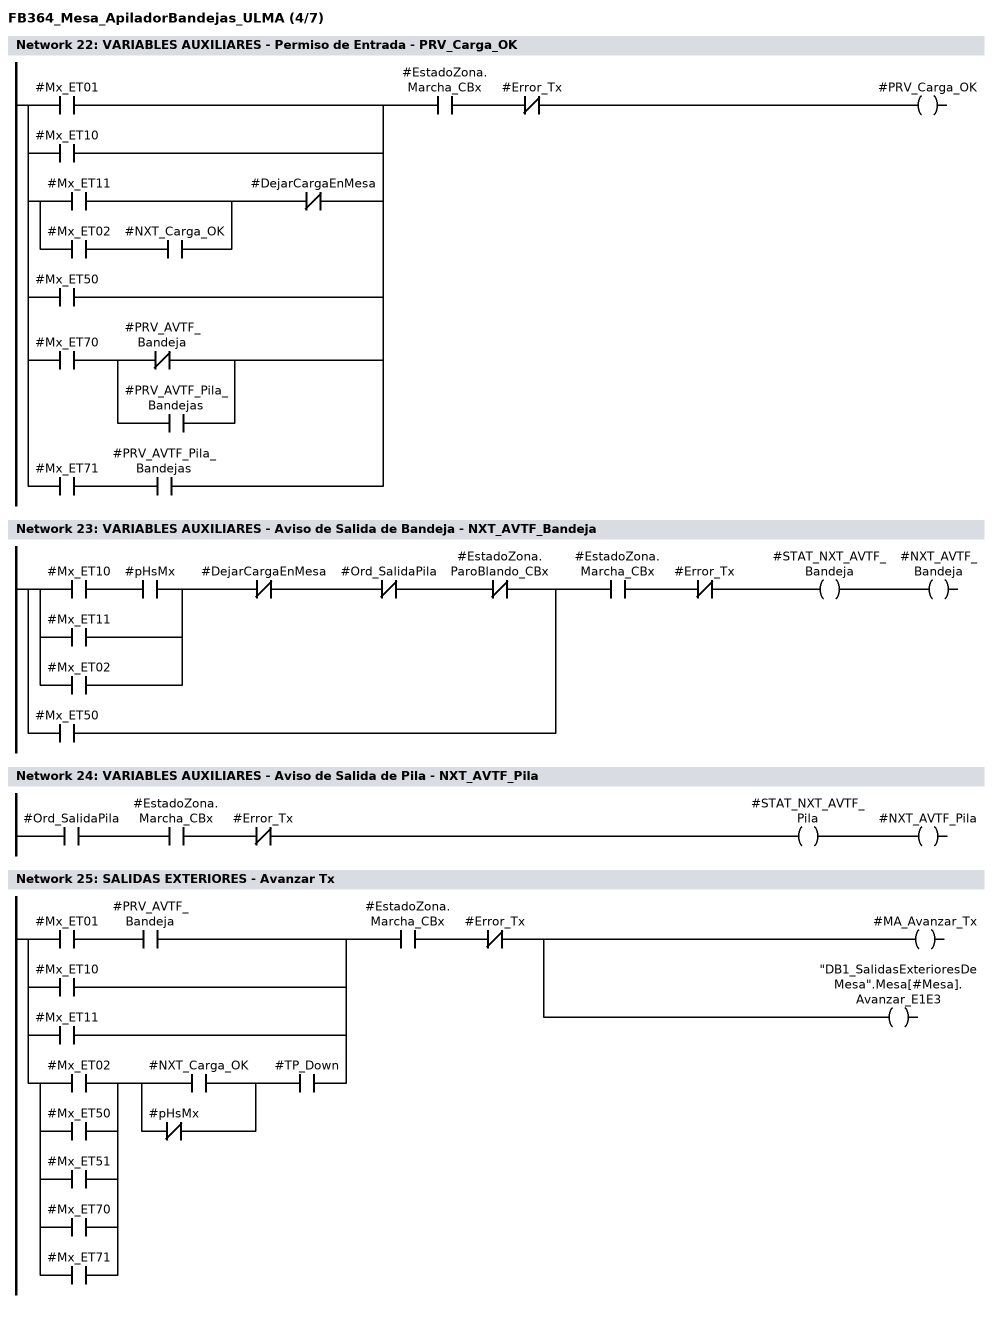
   RUNG wire#powerrail
      Contact( #Mx_ET01 )
      wire#w1
      Contact( #EstadoZona.Marcha_CBx )
      I_Contact( #Error_Tx )
      Coil( #PRV_Carga_OK )
   END_RUNG
   RUNG wire#powerrail
      Contact( #Mx_ET10 )
   END_RUNG wire#w1
   RUNG wire#powerrail
      Contact( #Mx_ET11 )
      wire#w2
      I_Contact( #DejarCargaEnMesa )
   END_RUNG wire#w1
   RUNG wire#powerrail
      Contact( #Mx_ET02 )
      Contact( #NXT_Carga_OK )
   END_RUNG wire#w2
   RUNG wire#powerrail
      Contact( #Mx_ET50 )
   END_RUNG wire#w1
   RUNG wire#powerrail
      Contact( #Mx_ET70 )
      wire#w3
      I_Contact( #PRV_AVTF_Bandeja )
   END_RUNG wire#w1
   RUNG wire#w3
      Contact( #PRV_AVTF_Pila_Bandejas )
   END_RUNG wire#w1
   RUNG wire#powerrail
      Contact( #Mx_ET71 )
      Contact( #PRV_AVTF_Pila_Bandejas )
   END_RUNG wire#w1
   // the same network as SCL:
   #PRV_Carga_OK := (#Mx_ET01 OR #Mx_ET10 OR ((#Mx_ET11 OR (#Mx_ET02 AND #NXT_Carga_OK)) AND NOT #DejarCargaEnMesa) OR #Mx_ET50 OR (#Mx_ET70 AND (NOT #PRV_AVTF_Bandeja OR #PRV_AVTF_Pila_Bandejas)) OR (#Mx_ET71 AND #PRV_AVTF_Pila_Bandejas)) AND #EstadoZona.Marcha_CBx AND NOT #Error_Tx;
END_REGION

REGION Network 23: VARIABLES AUXILIARES - Aviso de Salida de Bandeja - NXT_AVTF_Bandeja
   RUNG wire#powerrail
      Contact( #Mx_ET10 )
      Contact( #pHsMx )
      wire#w1
      I_Contact( #DejarCargaEnMesa )
      I_Contact( #Ord_SalidaPila )
      I_Contact( #EstadoZona.ParoBlando_CBx )
      wire#w2
      Contact( #EstadoZona.Marcha_CBx )
      I_Contact( #Error_Tx )
      Coil( #STAT_NXT_AVTF_Bandeja )
      Coil( #NXT_AVTF_Bandeja )
   END_RUNG
   RUNG wire#powerrail
      Contact( #Mx_ET11 )
   END_RUNG wire#w1
   RUNG wire#powerrail
      Contact( #Mx_ET02 )
   END_RUNG wire#w1
   RUNG wire#powerrail
      Contact( #Mx_ET50 )
   END_RUNG wire#w2
   // the same network as SCL:
   #STAT_NXT_AVTF_Bandeja := ((((#Mx_ET10 AND #pHsMx) OR #Mx_ET11 OR #Mx_ET02) AND NOT #DejarCargaEnMesa AND NOT #Ord_SalidaPila AND NOT #EstadoZona.ParoBlando_CBx) OR #Mx_ET50) AND #EstadoZona.Marcha_CBx AND NOT #Error_Tx;
   #NXT_AVTF_Bandeja := #STAT_NXT_AVTF_Bandeja;
END_REGION

REGION Network 24: VARIABLES AUXILIARES - Aviso de Salida de Pila - NXT_AVTF_Pila
   RUNG wire#powerrail
      Contact( #Ord_SalidaPila )
      Contact( #EstadoZona.Marcha_CBx )
      I_Contact( #Error_Tx )
      Coil( #STAT_NXT_AVTF_Pila )
      Coil( #NXT_AVTF_Pila )
   END_RUNG
   // the same network as SCL:
   #STAT_NXT_AVTF_Pila := #Ord_SalidaPila AND #EstadoZona.Marcha_CBx AND NOT #Error_Tx;
   #NXT_AVTF_Pila := #STAT_NXT_AVTF_Pila;
END_REGION

REGION Network 25: SALIDAS EXTERIORES - Avanzar Tx
   RUNG wire#powerrail
      Contact( #Mx_ET01 )
      Contact( #PRV_AVTF_Bandeja )
      wire#w1
      Contact( #EstadoZona.Marcha_CBx )
      I_Contact( #Error_Tx )
      wire#w4
      Coil( #MA_Avanzar_Tx )
   END_RUNG
   RUNG wire#powerrail
      Contact( #Mx_ET10 )
   END_RUNG wire#w1
   RUNG wire#powerrail
      Contact( #Mx_ET11 )
   END_RUNG wire#w1
   RUNG wire#powerrail
      Contact( #Mx_ET02 )
      wire#w2
      Contact( #NXT_Carga_OK )
      wire#w3
      Contact( #TP_Down )
   END_RUNG wire#w1
   RUNG wire#powerrail
      Contact( #Mx_ET50 )
   END_RUNG wire#w2
   RUNG wire#powerrail
      Contact( #Mx_ET51 )
   END_RUNG wire#w2
   RUNG wire#powerrail
      Contact( #Mx_ET70 )
   END_RUNG wire#w2
   RUNG wire#powerrail
      Contact( #Mx_ET71 )
   END_RUNG wire#w2
   RUNG wire#w2
      I_Contact( #pHsMx )
   END_RUNG wire#w3
   RUNG wire#w4
      Coil( "DB1_SalidasExterioresDeMesa".Mesa[#Mesa].Avanzar_E1E3 )
   END_RUNG
   // the same network as SCL:
   #MA_Avanzar_Tx := ((#Mx_ET01 AND #PRV_AVTF_Bandeja) OR #Mx_ET10 OR #Mx_ET11 OR ((#Mx_ET02 OR #Mx_ET50 OR #Mx_ET51 OR #Mx_ET70 OR #Mx_ET71) AND (#NXT_Carga_OK OR NOT #pHsMx) AND #TP_Down)) AND #EstadoZona.Marcha_CBx AND NOT #Error_Tx;
   "DB1_SalidasExterioresDeMesa".Mesa[#Mesa].Avanzar_E1E3 := #MA_Avanzar_Tx;
END_REGION

REGION Network 26: SALIDAS EXTERIORES - Parar Tx
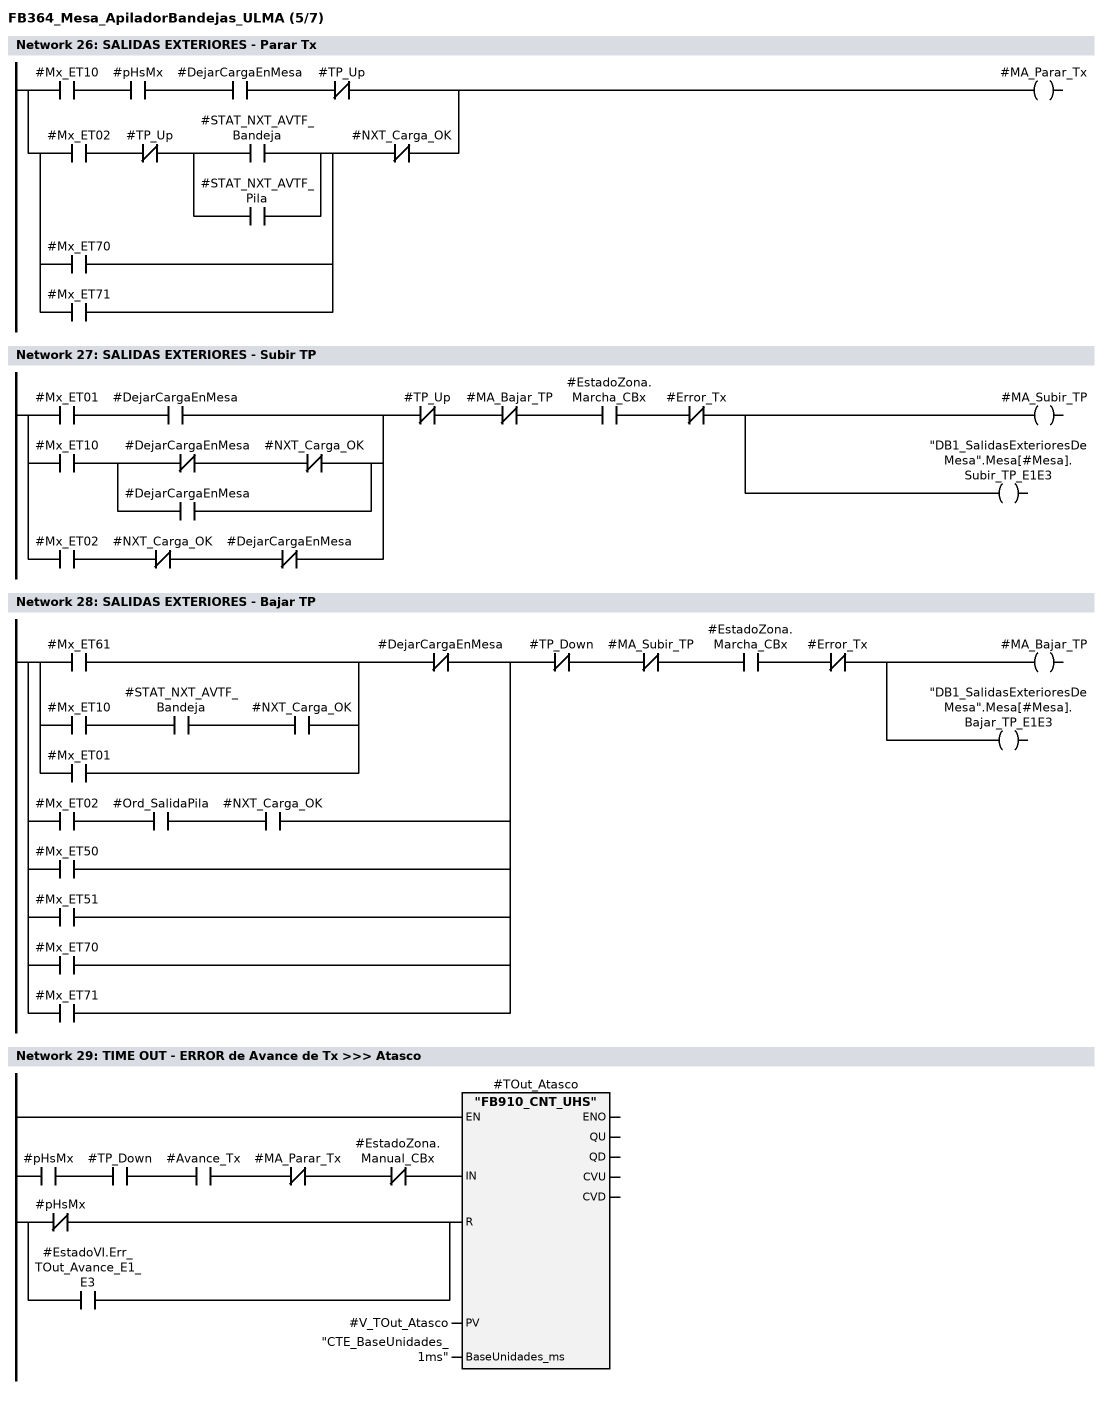
   RUNG wire#powerrail
      Contact( #Mx_ET10 )
      Contact( #pHsMx )
      Contact( #DejarCargaEnMesa )
      I_Contact( #TP_Up )
      wire#w1
      Coil( #MA_Parar_Tx )
   END_RUNG
   RUNG wire#powerrail
      Contact( #Mx_ET02 )
      I_Contact( #TP_Up )
      wire#w2
      Contact( #STAT_NXT_AVTF_Bandeja )
      wire#w3
      I_Contact( #NXT_Carga_OK )
   END_RUNG wire#w1
   RUNG wire#w2
      Contact( #STAT_NXT_AVTF_Pila )
   END_RUNG wire#w3
   RUNG wire#powerrail
      Contact( #Mx_ET70 )
   END_RUNG wire#w3
   RUNG wire#powerrail
      Contact( #Mx_ET71 )
   END_RUNG wire#w3
   // the same network as SCL:
   #MA_Parar_Tx := (#Mx_ET10 AND #pHsMx AND #DejarCargaEnMesa AND NOT #TP_Up) OR (((#Mx_ET02 AND NOT #TP_Up AND (#STAT_NXT_AVTF_Bandeja OR #STAT_NXT_AVTF_Pila)) OR #Mx_ET70 OR #Mx_ET71) AND NOT #NXT_Carga_OK);
END_REGION

REGION Network 27: SALIDAS EXTERIORES - Subir TP
   RUNG wire#powerrail
      Contact( #Mx_ET01 )
      Contact( #DejarCargaEnMesa )
      wire#w1
      I_Contact( #TP_Up )
      I_Contact( #MA_Bajar_TP )
      Contact( #EstadoZona.Marcha_CBx )
      I_Contact( #Error_Tx )
      wire#w3
      Coil( #MA_Subir_TP )
   END_RUNG
   RUNG wire#powerrail
      Contact( #Mx_ET10 )
      wire#w2
      I_Contact( #DejarCargaEnMesa )
      I_Contact( #NXT_Carga_OK )
   END_RUNG wire#w1
   RUNG wire#w2
      Contact( #DejarCargaEnMesa )
   END_RUNG wire#w1
   RUNG wire#powerrail
      Contact( #Mx_ET02 )
      I_Contact( #NXT_Carga_OK )
      I_Contact( #DejarCargaEnMesa )
   END_RUNG wire#w1
   RUNG wire#w3
      Coil( "DB1_SalidasExterioresDeMesa".Mesa[#Mesa].Subir_TP_E1E3 )
   END_RUNG
   // the same network as SCL:
   #MA_Subir_TP := ((#Mx_ET01 AND #DejarCargaEnMesa) OR (#Mx_ET10 AND ((NOT #DejarCargaEnMesa AND NOT #NXT_Carga_OK) OR #DejarCargaEnMesa)) OR (#Mx_ET02 AND NOT #NXT_Carga_OK AND NOT #DejarCargaEnMesa)) AND NOT #TP_Up AND NOT #MA_Bajar_TP AND #EstadoZona.Marcha_CBx AND NOT #Error_Tx;
   "DB1_SalidasExterioresDeMesa".Mesa[#Mesa].Subir_TP_E1E3 := #MA_Subir_TP;
END_REGION

REGION Network 28: SALIDAS EXTERIORES - Bajar TP
   RUNG wire#powerrail
      Contact( #Mx_ET61 )
      wire#w1
      I_Contact( #DejarCargaEnMesa )
      wire#w2
      I_Contact( #TP_Down )
      I_Contact( #MA_Subir_TP )
      Contact( #EstadoZona.Marcha_CBx )
      I_Contact( #Error_Tx )
      wire#w3
      Coil( #MA_Bajar_TP )
   END_RUNG
   RUNG wire#powerrail
      Contact( #Mx_ET10 )
      Contact( #STAT_NXT_AVTF_Bandeja )
      Contact( #NXT_Carga_OK )
   END_RUNG wire#w1
   RUNG wire#powerrail
      Contact( #Mx_ET01 )
   END_RUNG wire#w1
   RUNG wire#powerrail
      Contact( #Mx_ET02 )
      Contact( #Ord_SalidaPila )
      Contact( #NXT_Carga_OK )
   END_RUNG wire#w2
   RUNG wire#powerrail
      Contact( #Mx_ET50 )
   END_RUNG wire#w2
   RUNG wire#powerrail
      Contact( #Mx_ET51 )
   END_RUNG wire#w2
   RUNG wire#powerrail
      Contact( #Mx_ET70 )
   END_RUNG wire#w2
   RUNG wire#powerrail
      Contact( #Mx_ET71 )
   END_RUNG wire#w2
   RUNG wire#w3
      Coil( "DB1_SalidasExterioresDeMesa".Mesa[#Mesa].Bajar_TP_E1E3 )
   END_RUNG
   // the same network as SCL:
   #MA_Bajar_TP := (((#Mx_ET61 OR (#Mx_ET10 AND #STAT_NXT_AVTF_Bandeja AND #NXT_Carga_OK) OR #Mx_ET01) AND NOT #DejarCargaEnMesa) OR (#Mx_ET02 AND #Ord_SalidaPila AND #NXT_Carga_OK) OR #Mx_ET50 OR #Mx_ET51 OR #Mx_ET70 OR #Mx_ET71) AND NOT #TP_Down AND NOT #MA_Subir_TP AND #EstadoZona.Marcha_CBx AND NOT #Error_Tx;
   "DB1_SalidasExterioresDeMesa".Mesa[#Mesa].Bajar_TP_E1E3 := #MA_Bajar_TP;
END_REGION

REGION Network 29: TIME OUT - ERROR de Avance de Tx >>> Atasco
   RUNG wire#powerrail
      #TOut_Atasco(IN := wire#w1, R := wire#w2, PV := #V_TOut_Atasco, BaseUnidades_ms := "CTE_BaseUnidades_1ms", QU =>, QD =>, CVU =>, CVD =>)
   END_RUNG
   RUNG wire#powerrail
      Contact( #pHsMx )
      Contact( #TP_Down )
      Contact( #Avance_Tx )
      I_Contact( #MA_Parar_Tx )
      I_Contact( #EstadoZona.Manual_CBx )
   END_RUNG wire#w1
   RUNG wire#powerrail
      I_Contact( #pHsMx )
   END_RUNG wire#w2
   RUNG wire#powerrail
      Contact( #EstadoVI.Err_TOut_Avance_E1_E3 )
   END_RUNG wire#w2
   // the same network as SCL:
   #TOut_Atasco(IN := #pHsMx AND #TP_Down AND #Avance_Tx AND NOT #MA_Parar_Tx AND NOT #EstadoZona.Manual_CBx,   // "FB910_CNT_UHS"
                R := NOT #pHsMx OR #EstadoVI.Err_TOut_Avance_E1_E3,
                PV := #V_TOut_Atasco,
                BaseUnidades_ms := "CTE_BaseUnidades_1ms");
END_REGION

REGION Network 30: ERROR de Avance de Tx >>> Atasco
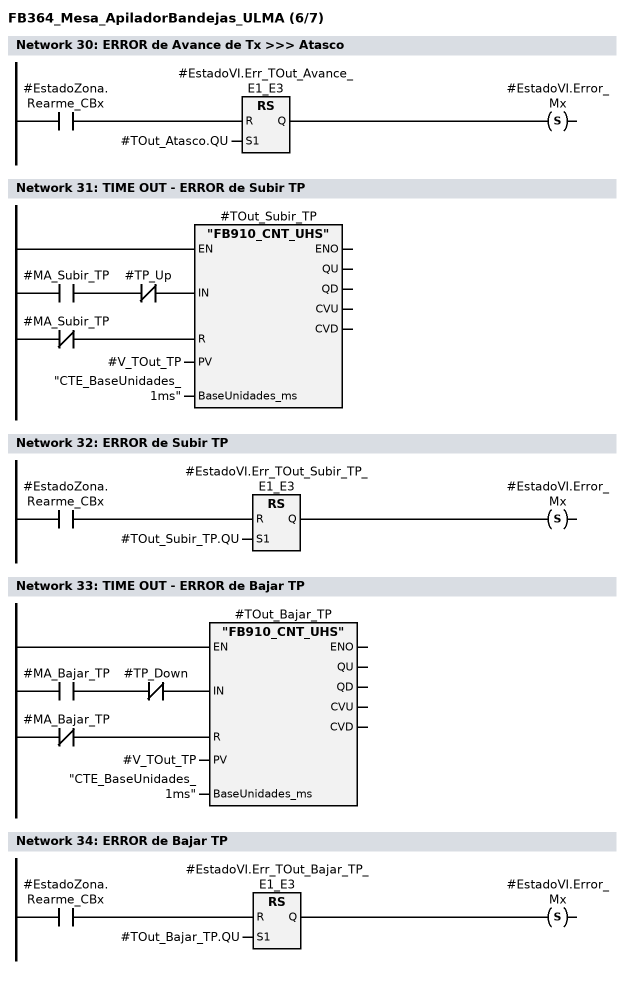
   RUNG wire#powerrail
      Contact( #EstadoZona.Rearme_CBx )
      S_RS(operand := #EstadoVI.Err_TOut_Avance_E1_E3, s1 := #TOut_Atasco.QU)
      S_Coil( #EstadoVI.Error_Mx )
   END_RUNG
   // the same network as SCL:
   IF #EstadoZona.Rearme_CBx THEN
       #EstadoVI.Err_TOut_Avance_E1_E3 := FALSE;   // RS flip-flop
   END_IF;
   IF #TOut_Atasco.QU THEN #EstadoVI.Err_TOut_Avance_E1_E3 := TRUE; END_IF;
   IF #EstadoVI.Err_TOut_Avance_E1_E3 THEN #EstadoVI.Error_Mx := TRUE; END_IF;
END_REGION

REGION Network 31: TIME OUT - ERROR de Subir TP
   RUNG wire#powerrail
      #TOut_Subir_TP(IN := wire#w1, R := wire#w2, PV := #V_TOut_TP, BaseUnidades_ms := "CTE_BaseUnidades_1ms", QU =>, QD =>, CVU =>, CVD =>)
   END_RUNG
   RUNG wire#powerrail
      Contact( #MA_Subir_TP )
      I_Contact( #TP_Up )
   END_RUNG wire#w1
   RUNG wire#powerrail
      I_Contact( #MA_Subir_TP )
   END_RUNG wire#w2
   // the same network as SCL:
   #TOut_Subir_TP(IN := #MA_Subir_TP AND NOT #TP_Up,   // "FB910_CNT_UHS"
                  R := NOT #MA_Subir_TP,
                  PV := #V_TOut_TP,
                  BaseUnidades_ms := "CTE_BaseUnidades_1ms");
END_REGION

REGION Network 32: ERROR de Subir TP
   RUNG wire#powerrail
      Contact( #EstadoZona.Rearme_CBx )
      S_RS(operand := #EstadoVI.Err_TOut_Subir_TP_E1_E3, s1 := #TOut_Subir_TP.QU)
      S_Coil( #EstadoVI.Error_Mx )
   END_RUNG
   // the same network as SCL:
   IF #EstadoZona.Rearme_CBx THEN
       #EstadoVI.Err_TOut_Subir_TP_E1_E3 := FALSE;   // RS flip-flop
   END_IF;
   IF #TOut_Subir_TP.QU THEN #EstadoVI.Err_TOut_Subir_TP_E1_E3 := TRUE; END_IF;
   IF #EstadoVI.Err_TOut_Subir_TP_E1_E3 THEN #EstadoVI.Error_Mx := TRUE; END_IF;
END_REGION

REGION Network 33: TIME OUT - ERROR de Bajar TP
   RUNG wire#powerrail
      #TOut_Bajar_TP(IN := wire#w1, R := wire#w2, PV := #V_TOut_TP, BaseUnidades_ms := "CTE_BaseUnidades_1ms", QU =>, QD =>, CVU =>, CVD =>)
   END_RUNG
   RUNG wire#powerrail
      Contact( #MA_Bajar_TP )
      I_Contact( #TP_Down )
   END_RUNG wire#w1
   RUNG wire#powerrail
      I_Contact( #MA_Bajar_TP )
   END_RUNG wire#w2
   // the same network as SCL:
   #TOut_Bajar_TP(IN := #MA_Bajar_TP AND NOT #TP_Down,   // "FB910_CNT_UHS"
                  R := NOT #MA_Bajar_TP,
                  PV := #V_TOut_TP,
                  BaseUnidades_ms := "CTE_BaseUnidades_1ms");
END_REGION

REGION Network 34: ERROR de Bajar TP
   RUNG wire#powerrail
      Contact( #EstadoZona.Rearme_CBx )
      S_RS(operand := #EstadoVI.Err_TOut_Bajar_TP_E1_E3, s1 := #TOut_Bajar_TP.QU)
      S_Coil( #EstadoVI.Error_Mx )
   END_RUNG
   // the same network as SCL:
   IF #EstadoZona.Rearme_CBx THEN
       #EstadoVI.Err_TOut_Bajar_TP_E1_E3 := FALSE;   // RS flip-flop
   END_IF;
   IF #TOut_Bajar_TP.QU THEN #EstadoVI.Err_TOut_Bajar_TP_E1_E3 := TRUE; END_IF;
   IF #EstadoVI.Err_TOut_Bajar_TP_E1_E3 THEN #EstadoVI.Error_Mx := TRUE; END_IF;
END_REGION

REGION Network 35: ESTADO DE LA MESA
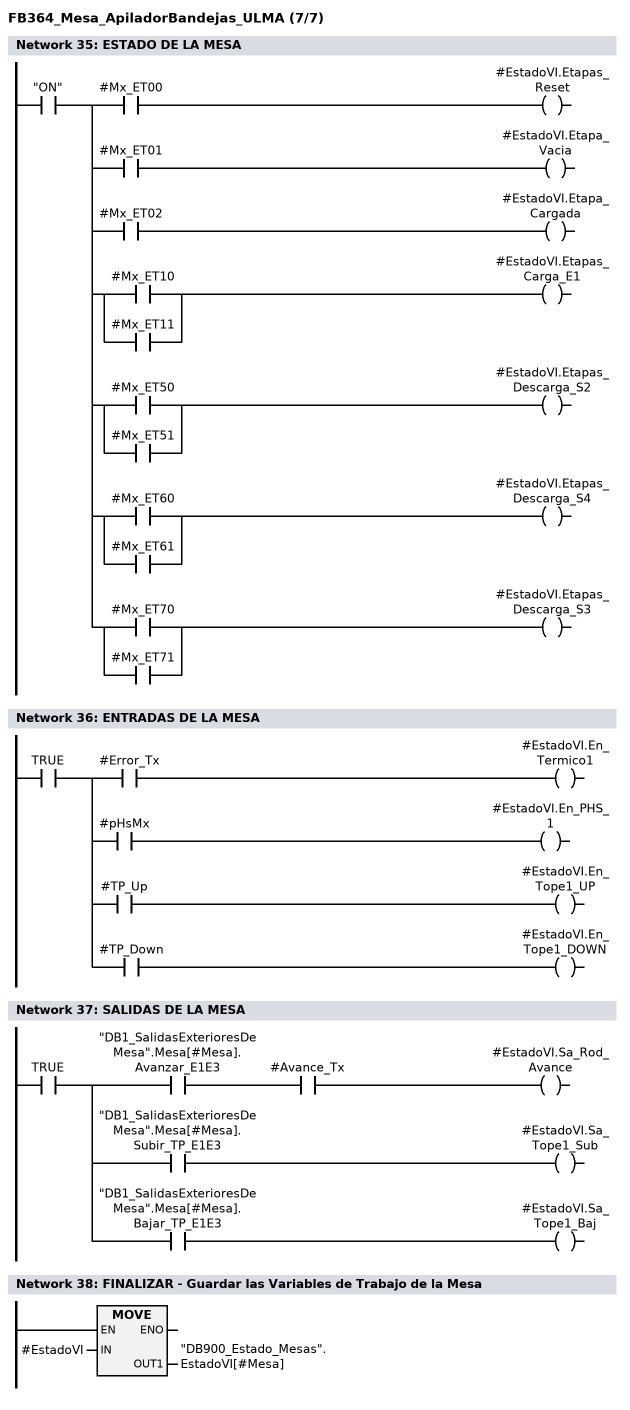
   RUNG wire#powerrail
      Contact( "ON" )
      wire#w1
      Contact( #Mx_ET00 )
      Coil( #EstadoVI.Etapas_Reset )
   END_RUNG
   RUNG wire#w1
      Contact( #Mx_ET01 )
      Coil( #EstadoVI.Etapa_Vacia )
   END_RUNG
   RUNG wire#w1
      Contact( #Mx_ET02 )
      Coil( #EstadoVI.Etapa_Cargada )
   END_RUNG
   RUNG wire#w1
      Contact( #Mx_ET10 )
      wire#w2
      Coil( #EstadoVI.Etapas_Carga_E1 )
   END_RUNG
   RUNG wire#w1
      Contact( #Mx_ET11 )
   END_RUNG wire#w2
   RUNG wire#w1
      Contact( #Mx_ET50 )
      wire#w3
      Coil( #EstadoVI.Etapas_Descarga_S2 )
   END_RUNG
   RUNG wire#w1
      Contact( #Mx_ET51 )
   END_RUNG wire#w3
   RUNG wire#w1
      Contact( #Mx_ET60 )
      wire#w4
      Coil( #EstadoVI.Etapas_Descarga_S4 )
   END_RUNG
   RUNG wire#w1
      Contact( #Mx_ET61 )
   END_RUNG wire#w4
   RUNG wire#w1
      Contact( #Mx_ET70 )
      wire#w5
      Coil( #EstadoVI.Etapas_Descarga_S3 )
   END_RUNG
   RUNG wire#w1
      Contact( #Mx_ET71 )
   END_RUNG wire#w5
   // the same network as SCL:
   #EstadoVI.Etapas_Reset := "ON" AND #Mx_ET00;
   #EstadoVI.Etapa_Vacia := "ON" AND #Mx_ET01;
   #EstadoVI.Etapa_Cargada := "ON" AND #Mx_ET02;
   #EstadoVI.Etapas_Carga_E1 := "ON" AND (#Mx_ET10 OR #Mx_ET11);
   #EstadoVI.Etapas_Descarga_S2 := "ON" AND (#Mx_ET50 OR #Mx_ET51);
   #EstadoVI.Etapas_Descarga_S4 := "ON" AND (#Mx_ET60 OR #Mx_ET61);
   #EstadoVI.Etapas_Descarga_S3 := "ON" AND (#Mx_ET70 OR #Mx_ET71);
END_REGION

REGION Network 36: ENTRADAS DE LA MESA
   RUNG wire#powerrail
      Contact( TRUE )
      wire#w1
      Contact( #Error_Tx )
      Coil( #EstadoVI.En_Termico1 )
   END_RUNG
   RUNG wire#w1
      Contact( #pHsMx )
      Coil( #EstadoVI.En_PHS_1 )
   END_RUNG
   RUNG wire#w1
      Contact( #TP_Up )
      Coil( #EstadoVI.En_Tope1_UP )
   END_RUNG
   RUNG wire#w1
      Contact( #TP_Down )
      Coil( #EstadoVI.En_Tope1_DOWN )
   END_RUNG
   // the same network as SCL:
   #EstadoVI.En_Termico1 := TRUE AND #Error_Tx;
   #EstadoVI.En_PHS_1 := TRUE AND #pHsMx;
   #EstadoVI.En_Tope1_UP := TRUE AND #TP_Up;
   #EstadoVI.En_Tope1_DOWN := TRUE AND #TP_Down;
END_REGION

REGION Network 37: SALIDAS DE LA MESA
   RUNG wire#powerrail
      Contact( TRUE )
      wire#w1
      Contact( "DB1_SalidasExterioresDeMesa".Mesa[#Mesa].Avanzar_E1E3 )
      Contact( #Avance_Tx )
      Coil( #EstadoVI.Sa_Rod_Avance )
   END_RUNG
   RUNG wire#w1
      Contact( "DB1_SalidasExterioresDeMesa".Mesa[#Mesa].Subir_TP_E1E3 )
      Coil( #EstadoVI.Sa_Tope1_Sub )
   END_RUNG
   RUNG wire#w1
      Contact( "DB1_SalidasExterioresDeMesa".Mesa[#Mesa].Bajar_TP_E1E3 )
      Coil( #EstadoVI.Sa_Tope1_Baj )
   END_RUNG
   // the same network as SCL:
   #EstadoVI.Sa_Rod_Avance := TRUE AND "DB1_SalidasExterioresDeMesa".Mesa[#Mesa].Avanzar_E1E3 AND #Avance_Tx;
   #EstadoVI.Sa_Tope1_Sub := TRUE AND "DB1_SalidasExterioresDeMesa".Mesa[#Mesa].Subir_TP_E1E3;
   #EstadoVI.Sa_Tope1_Baj := TRUE AND "DB1_SalidasExterioresDeMesa".Mesa[#Mesa].Bajar_TP_E1E3;
END_REGION

REGION Network 38: FINALIZAR - Guardar las Variables de Trabajo de la Mesa
   RUNG wire#powerrail
      Move(in := #EstadoVI, out1 => "DB900_Estado_Mesas".EstadoVI[#Mesa])
   END_RUNG
   // the same network as SCL:
   "DB900_Estado_Mesas".EstadoVI[#Mesa] := #EstadoVI;
END_REGION
END_FUNCTION_BLOCK

FUNCTION_BLOCK "FB365_ApiladorBandejas_ULMA_4Pilas"   // FB365, LAD
{ S7_Optimized_Access := 'FALSE' }
AUTHOR : TLigero
NAME : 20160211
VERSION : 0.2
// stored: AutoNumber false, SetENOAutomatically false
   VAR_INPUT
      Mesa : UInt;   // Mesa de la FB
      EnTension : Bool;   // Existe Tension en la Mesa
      Error_Tx : Bool;   // Error en el Tx
      Selector : "Selector";   // Selector Unidades
      Selector_AD : Bool;   // Selector de Adelante
      Selector_AT : Bool;   // Selector de Atras
      Termico_Tx : Bool;   // Proteccion de Tx
      pHs_M1 : Bool;   // pHs de la P01 de la Mesa
      pHs_M2 : Bool;   // pHs de laP02 de la Mesa
      pHs_M3 : Bool;   // pHs de la P03 de la Mesa
      pHs_M4 : Bool;   // pHs de la P04 de la Mesa
      pHs_SalidaApilador : Bool;   // pHs de Control a Salida del Apilador
      pHs_VacioApìlador : Bool;   // phs de Apilador Vacio
      pHs_LlenoApilador : Bool;   // pHs de Apilador Lleno
      Avance_Tx : Bool;   // Avance de Tx
      Termico_Apilador : Bool;   // Proteccion de Elevacion del Apilador
      Apilador_UP : Bool;   // Apilador en Posicion Up
      Apilador_DW : Bool;   // Apilador en Posicion Down
      EnMovimento_Apilador : Bool;   // Apilador en Movimiento
      TPM1_Up : Bool;   // TP de la P01 Arriba
      TPM1_Down : Bool;   // TP de la P01 Abajo
      TPM2_Up : Bool;   // TP de la P02 Arriba
      TPM2_Down : Bool;   // TP de la P02 Abajo
      TPM3_Up : Bool;   // TP de la P03 Arriba
      TPM3_Down : Bool;   // TP de la P03 Abajo
      TPM4_Up : Bool;   // TP de la P04 Arriba
      TPM4_Down : Bool;   // TP de la P04 Abajo
      PRV_AVTF : Bool;   // E1 >> Aviso de Entrada
      NXT_Carga_OK : Bool;   // S3 >> Permiso de Salida
      NumBandejasPorPila : Int;   // Numero de Bandejas por Pila
      V_TOut_Atasco : Int;   // Valor de Time Out de Atasco
      V_TOut_Elevacion : Int;   // Valor de TIme Out de Elevacion
   END_VAR
   VAR_OUTPUT
      PRV_Carga_OK : Bool;   // E1 >> Permiso de Entrada
      NXT_AVTF : Bool;   // S3 >> Aviso de Salida
   END_VAR
   VAR
      M01 { S7_SetPoint := 'True'} : "FB364_Mesa_ApiladorBandejas_ULMA";
      M02 { S7_SetPoint := 'True'} : "FB364_Mesa_ApiladorBandejas_ULMA";
      M03 { S7_SetPoint := 'True'} : "FB364_Mesa_ApiladorBandejas_ULMA";
      M04 { S7_SetPoint := 'True'} : "FB364_Mesa_ApiladorBandejas_ULMA";
      EstadoVI_M01 { S7_SetPoint := 'True'} : "EstadosMesa";
      EstadoVI_M02 { S7_SetPoint := 'True'} : "EstadosMesa";
      EstadoVI_M03 { S7_SetPoint := 'True'} : "EstadosMesa";
      EstadoVI_M04 { S7_SetPoint := 'True'} : "EstadosMesa";
      TMP_EnTension { S7_SetPoint := 'True'} : "FB910_CNT_UHS";
      TOut_Elevacion { S7_SetPoint := 'True'} : "FB910_CNT_UHS";
      ContadorBandejasEnPila : Int;   // Contador De Bandejas por Pila
      Ord_Vaciado : Bool;   // Interna >> Apilador esta Lleno
      Ord_Apilar : Bool;   // Interna >> Apilar Bandeja
      Ir_PosicionReposo : Bool;   // Operacion >> Ir a Posicion Reposo
      Ir_CogerBandeja : Bool;   // Operacion >> Ir a Coger Bandeja (Apilar)
      Ir_DejarPIla : Bool;   // Operacion >> Ir a Dejar Pila (Vaciado)
      EnPosicionReposo : Bool;   // Esta En Posicion de Reposo
      CogidaBandeja : Bool;   // Cogida Bandeja
      DejadaPila : Bool;   // Dejada la Pila
      MFP_ApiladorVaciado : Bool;   // Memoria FP de Apilador Vaciado
      MFP_ContadorBandejas : Bool;   // Memoria FP de Inc. de Bandeja en Pila
      MA_Avance_Tx : Bool;
      MA_Retroceder_Tx : Bool;
      MA_Subir : Bool;
      MA_Bajar : Bool;
      MA_Subir_TPM1 : Bool;
      MA_Bajar_TPM1 : Bool;
      MA_Subir_TPM2 : Bool;
      MA_Bajar_TPM2 : Bool;
      MA_Subir_TPM3 : Bool;
      MA_Bajar_TPM3 : Bool;
      MA_Subir_TPM4 : Bool;
      MA_Bajar_TPM4 : Bool;
   END_VAR
   VAR_TEMP
      EstadoZona : "EstadoZona";   // Estado de Zona de la Mesa
      EstadoVI : "EstadosMesa";   // Estado del Vehiculo Inteliguente de la Mesa
      EstadoMAQ : "EstadoMaquina";   // Estado del Vehiculo Inteliguente de la Maquina
      Aux_ET00 : Bool;
   END_VAR
   VAR_TEMP   // added for the SCL form of the ladder/FBD networks
      _w1 : Bool;
      _w2 : Bool;
   END_VAR
BEGIN

REGION Network 1: INICIALIZAR - Recoger las Variables de Estado de la Mesa
   // Se recoge - Estado_CBx
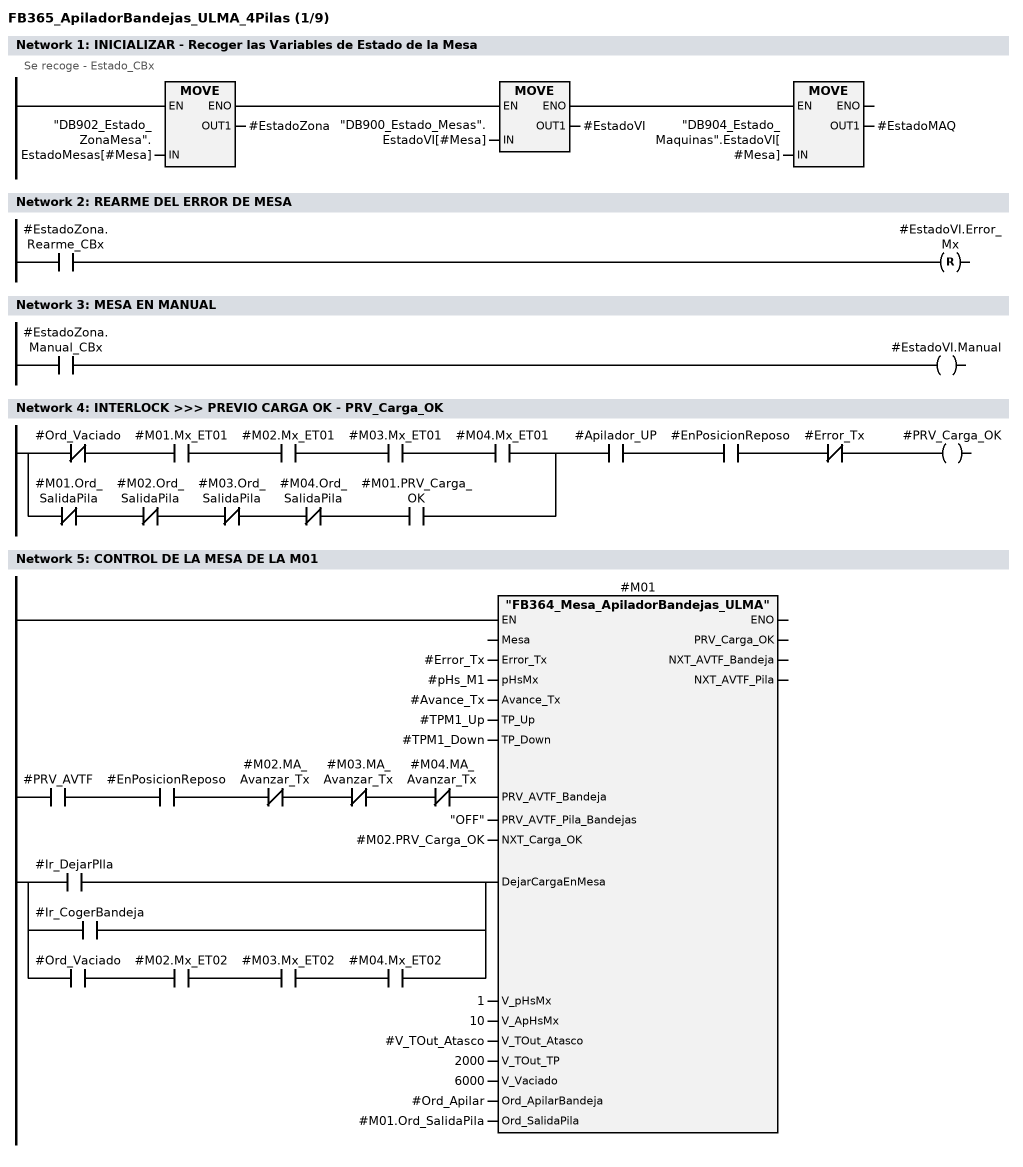
   RUNG wire#powerrail
      Move(in := "DB902_Estado_ZonaMesa".EstadoMesas[#Mesa], out1 => #EstadoZona)
      Move(in := "DB900_Estado_Mesas".EstadoVI[#Mesa], out1 => #EstadoVI)
      Move(in := "DB904_Estado_Maquinas".EstadoVI[#Mesa], out1 => #EstadoMAQ)
   END_RUNG
   // the same network as SCL:
   #EstadoZona := "DB902_Estado_ZonaMesa".EstadoMesas[#Mesa];
   #EstadoVI := "DB900_Estado_Mesas".EstadoVI[#Mesa];
   #EstadoMAQ := "DB904_Estado_Maquinas".EstadoVI[#Mesa];
END_REGION

REGION Network 2: REARME DEL ERROR DE MESA
   RUNG wire#powerrail
      Contact( #EstadoZona.Rearme_CBx )
      R_Coil( #EstadoVI.Error_Mx )
   END_RUNG
   // the same network as SCL:
   IF #EstadoZona.Rearme_CBx THEN #EstadoVI.Error_Mx := FALSE; END_IF;
END_REGION

REGION Network 3: MESA EN MANUAL
   RUNG wire#powerrail
      Contact( #EstadoZona.Manual_CBx )
      Coil( #EstadoVI.Manual )
   END_RUNG
   // the same network as SCL:
   #EstadoVI.Manual := #EstadoZona.Manual_CBx;
END_REGION

REGION Network 4: INTERLOCK >>> PREVIO CARGA OK - PRV_Carga_OK
   RUNG wire#powerrail
      I_Contact( #Ord_Vaciado )
      Contact( #M01.Mx_ET01 )
      Contact( #M02.Mx_ET01 )
      Contact( #M03.Mx_ET01 )
      Contact( #M04.Mx_ET01 )
      wire#w1
      Contact( #Apilador_UP )
      Contact( #EnPosicionReposo )
      I_Contact( #Error_Tx )
      Coil( #PRV_Carga_OK )
   END_RUNG
   RUNG wire#powerrail
      I_Contact( #M01.Ord_SalidaPila )
      I_Contact( #M02.Ord_SalidaPila )
      I_Contact( #M03.Ord_SalidaPila )
      I_Contact( #M04.Ord_SalidaPila )
      Contact( #M01.PRV_Carga_OK )
   END_RUNG wire#w1
   // the same network as SCL:
   #PRV_Carga_OK := ((NOT #Ord_Vaciado AND #M01.Mx_ET01 AND #M02.Mx_ET01 AND #M03.Mx_ET01 AND #M04.Mx_ET01) OR (NOT #M01.Ord_SalidaPila AND NOT #M02.Ord_SalidaPila AND NOT #M03.Ord_SalidaPila AND NOT #M04.Ord_SalidaPila AND #M01.PRV_Carga_OK)) AND #Apilador_UP AND #EnPosicionReposo AND NOT #Error_Tx;
END_REGION

REGION Network 5: CONTROL DE LA MESA DE LA M01
   RUNG wire#powerrail
      #M01(PRV_AVTF_Bandeja := wire#w1, DejarCargaEnMesa := wire#w2, Mesa :=, Error_Tx := #Error_Tx, pHsMx := #pHs_M1, Avance_Tx := #Avance_Tx, TP_Up := #TPM1_Up, TP_Down := #TPM1_Down, PRV_AVTF_Pila_Bandejas := "OFF", NXT_Carga_OK := #M02.PRV_Carga_OK, V_pHsMx := 1, V_ApHsMx := 10, V_TOut_Atasco := #V_TOut_Atasco, V_TOut_TP := 2000, V_Vaciado := 6000, Ord_ApilarBandeja := #Ord_Apilar, Ord_SalidaPila := #M01.Ord_SalidaPila, PRV_Carga_OK =>, NXT_AVTF_Bandeja =>, NXT_AVTF_Pila =>)
   END_RUNG
   RUNG wire#powerrail
      Contact( #PRV_AVTF )
      Contact( #EnPosicionReposo )
      I_Contact( #M02.MA_Avanzar_Tx )
      I_Contact( #M03.MA_Avanzar_Tx )
      I_Contact( #M04.MA_Avanzar_Tx )
   END_RUNG wire#w1
   RUNG wire#powerrail
      Contact( #Ir_DejarPIla )
   END_RUNG wire#w2
   RUNG wire#powerrail
      Contact( #Ir_CogerBandeja )
   END_RUNG wire#w2
   RUNG wire#powerrail
      Contact( #Ord_Vaciado )
      Contact( #M02.Mx_ET02 )
      Contact( #M03.Mx_ET02 )
      Contact( #M04.Mx_ET02 )
   END_RUNG wire#w2
   // the same network as SCL:
   #M01(Error_Tx := #Error_Tx,   // "FB364_Mesa_ApiladorBandejas_ULMA"
        pHsMx := #pHs_M1,
        Avance_Tx := #Avance_Tx,
        TP_Up := #TPM1_Up,
        TP_Down := #TPM1_Down,
        PRV_AVTF_Bandeja := #PRV_AVTF AND #EnPosicionReposo AND NOT #M02.MA_Avanzar_Tx AND NOT #M03.MA_Avanzar_Tx AND NOT #M04.MA_Avanzar_Tx,
        PRV_AVTF_Pila_Bandejas := "OFF",
        NXT_Carga_OK := #M02.PRV_Carga_OK,
        DejarCargaEnMesa := #Ir_DejarPIla OR #Ir_CogerBandeja OR (#Ord_Vaciado AND #M02.Mx_ET02 AND #M03.Mx_ET02 AND #M04.Mx_ET02),
        V_pHsMx := 1,
        V_ApHsMx := 10,
        V_TOut_Atasco := #V_TOut_Atasco,
        V_TOut_TP := 2000,
        V_Vaciado := 6000,
        Ord_ApilarBandeja := #Ord_Apilar,
        Ord_SalidaPila := #M01.Ord_SalidaPila);
END_REGION

REGION Network 6: CONTROL DE LA MESA DE LA M02
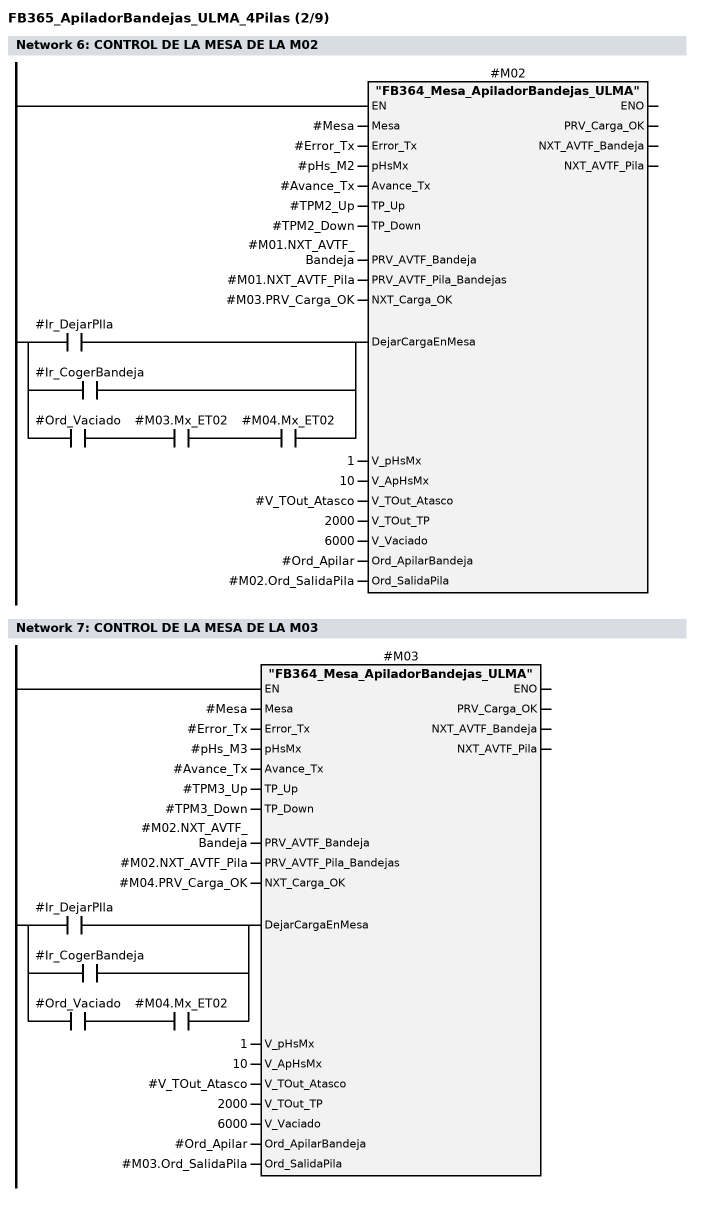
   RUNG wire#powerrail
      #M02(DejarCargaEnMesa := wire#w1, Mesa := #Mesa, Error_Tx := #Error_Tx, pHsMx := #pHs_M2, Avance_Tx := #Avance_Tx, TP_Up := #TPM2_Up, TP_Down := #TPM2_Down, PRV_AVTF_Bandeja := #M01.NXT_AVTF_Bandeja, PRV_AVTF_Pila_Bandejas := #M01.NXT_AVTF_Pila, NXT_Carga_OK := #M03.PRV_Carga_OK, V_pHsMx := 1, V_ApHsMx := 10, V_TOut_Atasco := #V_TOut_Atasco, V_TOut_TP := 2000, V_Vaciado := 6000, Ord_ApilarBandeja := #Ord_Apilar, Ord_SalidaPila := #M02.Ord_SalidaPila, PRV_Carga_OK =>, NXT_AVTF_Bandeja =>, NXT_AVTF_Pila =>)
   END_RUNG
   RUNG wire#powerrail
      Contact( #Ir_DejarPIla )
   END_RUNG wire#w1
   RUNG wire#powerrail
      Contact( #Ir_CogerBandeja )
   END_RUNG wire#w1
   RUNG wire#powerrail
      Contact( #Ord_Vaciado )
      Contact( #M03.Mx_ET02 )
      Contact( #M04.Mx_ET02 )
   END_RUNG wire#w1
   // the same network as SCL:
   #M02(Mesa := #Mesa,   // "FB364_Mesa_ApiladorBandejas_ULMA"
        Error_Tx := #Error_Tx,
        pHsMx := #pHs_M2,
        Avance_Tx := #Avance_Tx,
        TP_Up := #TPM2_Up,
        TP_Down := #TPM2_Down,
        PRV_AVTF_Bandeja := #M01.NXT_AVTF_Bandeja,
        PRV_AVTF_Pila_Bandejas := #M01.NXT_AVTF_Pila,
        NXT_Carga_OK := #M03.PRV_Carga_OK,
        DejarCargaEnMesa := #Ir_DejarPIla OR #Ir_CogerBandeja OR (#Ord_Vaciado AND #M03.Mx_ET02 AND #M04.Mx_ET02),
        V_pHsMx := 1,
        V_ApHsMx := 10,
        V_TOut_Atasco := #V_TOut_Atasco,
        V_TOut_TP := 2000,
        V_Vaciado := 6000,
        Ord_ApilarBandeja := #Ord_Apilar,
        Ord_SalidaPila := #M02.Ord_SalidaPila);
END_REGION

REGION Network 7: CONTROL DE LA MESA DE LA M03
   RUNG wire#powerrail
      #M03(DejarCargaEnMesa := wire#w1, Mesa := #Mesa, Error_Tx := #Error_Tx, pHsMx := #pHs_M3, Avance_Tx := #Avance_Tx, TP_Up := #TPM3_Up, TP_Down := #TPM3_Down, PRV_AVTF_Bandeja := #M02.NXT_AVTF_Bandeja, PRV_AVTF_Pila_Bandejas := #M02.NXT_AVTF_Pila, NXT_Carga_OK := #M04.PRV_Carga_OK, V_pHsMx := 1, V_ApHsMx := 10, V_TOut_Atasco := #V_TOut_Atasco, V_TOut_TP := 2000, V_Vaciado := 6000, Ord_ApilarBandeja := #Ord_Apilar, Ord_SalidaPila := #M03.Ord_SalidaPila, PRV_Carga_OK =>, NXT_AVTF_Bandeja =>, NXT_AVTF_Pila =>)
   END_RUNG
   RUNG wire#powerrail
      Contact( #Ir_DejarPIla )
   END_RUNG wire#w1
   RUNG wire#powerrail
      Contact( #Ir_CogerBandeja )
   END_RUNG wire#w1
   RUNG wire#powerrail
      Contact( #Ord_Vaciado )
      Contact( #M04.Mx_ET02 )
   END_RUNG wire#w1
   // the same network as SCL:
   #M03(Mesa := #Mesa,   // "FB364_Mesa_ApiladorBandejas_ULMA"
        Error_Tx := #Error_Tx,
        pHsMx := #pHs_M3,
        Avance_Tx := #Avance_Tx,
        TP_Up := #TPM3_Up,
        TP_Down := #TPM3_Down,
        PRV_AVTF_Bandeja := #M02.NXT_AVTF_Bandeja,
        PRV_AVTF_Pila_Bandejas := #M02.NXT_AVTF_Pila,
        NXT_Carga_OK := #M04.PRV_Carga_OK,
        DejarCargaEnMesa := #Ir_DejarPIla OR #Ir_CogerBandeja OR (#Ord_Vaciado AND #M04.Mx_ET02),
        V_pHsMx := 1,
        V_ApHsMx := 10,
        V_TOut_Atasco := #V_TOut_Atasco,
        V_TOut_TP := 2000,
        V_Vaciado := 6000,
        Ord_ApilarBandeja := #Ord_Apilar,
        Ord_SalidaPila := #M03.Ord_SalidaPila);
END_REGION

REGION Network 8: CONTROL DE LA MESA DE LA M04
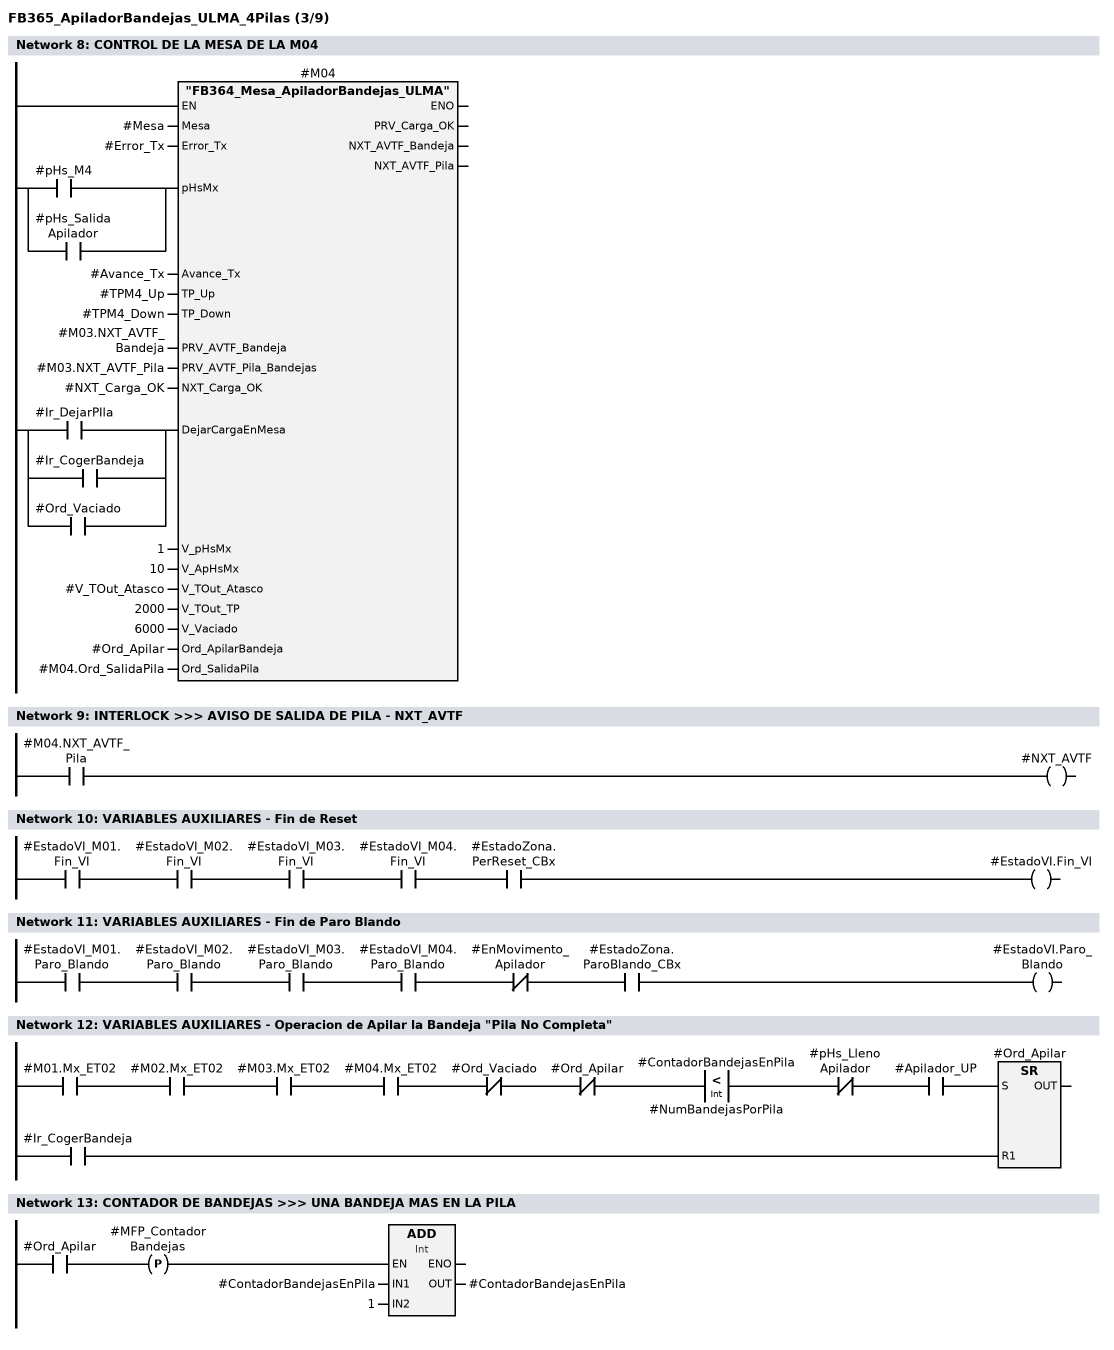
   RUNG wire#powerrail
      #M04(pHsMx := wire#w1, DejarCargaEnMesa := wire#w2, Mesa := #Mesa, Error_Tx := #Error_Tx, Avance_Tx := #Avance_Tx, TP_Up := #TPM4_Up, TP_Down := #TPM4_Down, PRV_AVTF_Bandeja := #M03.NXT_AVTF_Bandeja, PRV_AVTF_Pila_Bandejas := #M03.NXT_AVTF_Pila, NXT_Carga_OK := #NXT_Carga_OK, V_pHsMx := 1, V_ApHsMx := 10, V_TOut_Atasco := #V_TOut_Atasco, V_TOut_TP := 2000, V_Vaciado := 6000, Ord_ApilarBandeja := #Ord_Apilar, Ord_SalidaPila := #M04.Ord_SalidaPila, PRV_Carga_OK =>, NXT_AVTF_Bandeja =>, NXT_AVTF_Pila =>)
   END_RUNG
   RUNG wire#powerrail
      Contact( #pHs_M4 )
   END_RUNG wire#w1
   RUNG wire#powerrail
      Contact( #pHs_SalidaApilador )
   END_RUNG wire#w1
   RUNG wire#powerrail
      Contact( #Ir_DejarPIla )
   END_RUNG wire#w2
   RUNG wire#powerrail
      Contact( #Ir_CogerBandeja )
   END_RUNG wire#w2
   RUNG wire#powerrail
      Contact( #Ord_Vaciado )
   END_RUNG wire#w2
   // the same network as SCL:
   #M04(Mesa := #Mesa,   // "FB364_Mesa_ApiladorBandejas_ULMA"
        Error_Tx := #Error_Tx,
        pHsMx := #pHs_M4 OR #pHs_SalidaApilador,
        Avance_Tx := #Avance_Tx,
        TP_Up := #TPM4_Up,
        TP_Down := #TPM4_Down,
        PRV_AVTF_Bandeja := #M03.NXT_AVTF_Bandeja,
        PRV_AVTF_Pila_Bandejas := #M03.NXT_AVTF_Pila,
        NXT_Carga_OK := #NXT_Carga_OK,
        DejarCargaEnMesa := #Ir_DejarPIla OR #Ir_CogerBandeja OR #Ord_Vaciado,
        V_pHsMx := 1,
        V_ApHsMx := 10,
        V_TOut_Atasco := #V_TOut_Atasco,
        V_TOut_TP := 2000,
        V_Vaciado := 6000,
        Ord_ApilarBandeja := #Ord_Apilar,
        Ord_SalidaPila := #M04.Ord_SalidaPila);
END_REGION

REGION Network 9: INTERLOCK >>> AVISO DE SALIDA DE PILA - NXT_AVTF
   RUNG wire#powerrail
      Contact( #M04.NXT_AVTF_Pila )
      Coil( #NXT_AVTF )
   END_RUNG
   // the same network as SCL:
   #NXT_AVTF := #M04.NXT_AVTF_Pila;
END_REGION

REGION Network 10: VARIABLES AUXILIARES - Fin de Reset
   RUNG wire#powerrail
      Contact( #EstadoVI_M01.Fin_VI )
      Contact( #EstadoVI_M02.Fin_VI )
      Contact( #EstadoVI_M03.Fin_VI )
      Contact( #EstadoVI_M04.Fin_VI )
      Contact( #EstadoZona.PerReset_CBx )
      Coil( #EstadoVI.Fin_VI )
   END_RUNG
   // the same network as SCL:
   #EstadoVI.Fin_VI := #EstadoVI_M01.Fin_VI AND #EstadoVI_M02.Fin_VI AND #EstadoVI_M03.Fin_VI AND #EstadoVI_M04.Fin_VI AND #EstadoZona.PerReset_CBx;
END_REGION

REGION Network 11: VARIABLES AUXILIARES - Fin de Paro Blando
   RUNG wire#powerrail
      Contact( #EstadoVI_M01.Paro_Blando )
      Contact( #EstadoVI_M02.Paro_Blando )
      Contact( #EstadoVI_M03.Paro_Blando )
      Contact( #EstadoVI_M04.Paro_Blando )
      I_Contact( #EnMovimento_Apilador )
      Contact( #EstadoZona.ParoBlando_CBx )
      Coil( #EstadoVI.Paro_Blando )
   END_RUNG
   // the same network as SCL:
   #EstadoVI.Paro_Blando := #EstadoVI_M01.Paro_Blando AND #EstadoVI_M02.Paro_Blando AND #EstadoVI_M03.Paro_Blando AND #EstadoVI_M04.Paro_Blando AND NOT #EnMovimento_Apilador AND #EstadoZona.ParoBlando_CBx;
END_REGION

REGION Network 12: VARIABLES AUXILIARES - Operacion de Apilar la Bandeja "Pila No Completa"
   RUNG wire#powerrail
      Contact( #M01.Mx_ET02 )
      Contact( #M02.Mx_ET02 )
      Contact( #M03.Mx_ET02 )
      Contact( #M04.Mx_ET02 )
      I_Contact( #Ord_Vaciado )
      I_Contact( #Ord_Apilar )
      { S7_Templates := "SrcType := Int" } LT_Contact(in1 := #ContadorBandejasEnPila, in2 := #NumBandejasPorPila)
      I_Contact( #pHs_LlenoApilador )
      Contact( #Apilador_UP )
      S_SR(operand := #Ord_Apilar, r1 := wire#w1)
   END_RUNG
   RUNG wire#powerrail
      Contact( #Ir_CogerBandeja )
   END_RUNG wire#w1
   // the same network as SCL:
   IF #M01.Mx_ET02 AND #M02.Mx_ET02 AND #M03.Mx_ET02 AND #M04.Mx_ET02 AND NOT #Ord_Vaciado AND NOT #Ord_Apilar AND (#ContadorBandejasEnPila < #NumBandejasPorPila) AND NOT #pHs_LlenoApilador AND #Apilador_UP THEN
       #Ord_Apilar := TRUE;   // SR flip-flop
   END_IF;
   IF #Ir_CogerBandeja THEN #Ord_Apilar := FALSE; END_IF;
END_REGION

REGION Network 13: CONTADOR DE BANDEJAS >>> UNA BANDEJA MAS EN LA PILA
   RUNG wire#powerrail
      Contact( #Ord_Apilar )
      P_Trig( #MFP_ContadorBandejas )
      { S7_Templates := "SrcType := Int"; S7_GenerateENO := "TRUE" } Add(in1 := #ContadorBandejasEnPila, in2 := 1, out => #ContadorBandejasEnPila)
   END_RUNG
   // the same network as SCL:
   #_w1 := #Ord_Apilar AND NOT #MFP_ContadorBandejas;   // rising edge
   #MFP_ContadorBandejas := #Ord_Apilar;
   IF #_w1 THEN #ContadorBandejasEnPila := #ContadorBandejasEnPila + 1; END_IF;
END_REGION

REGION Network 14: CONTADOR DE BANDEJAS >>> RESET DE BANDEJAS EN LA PILA
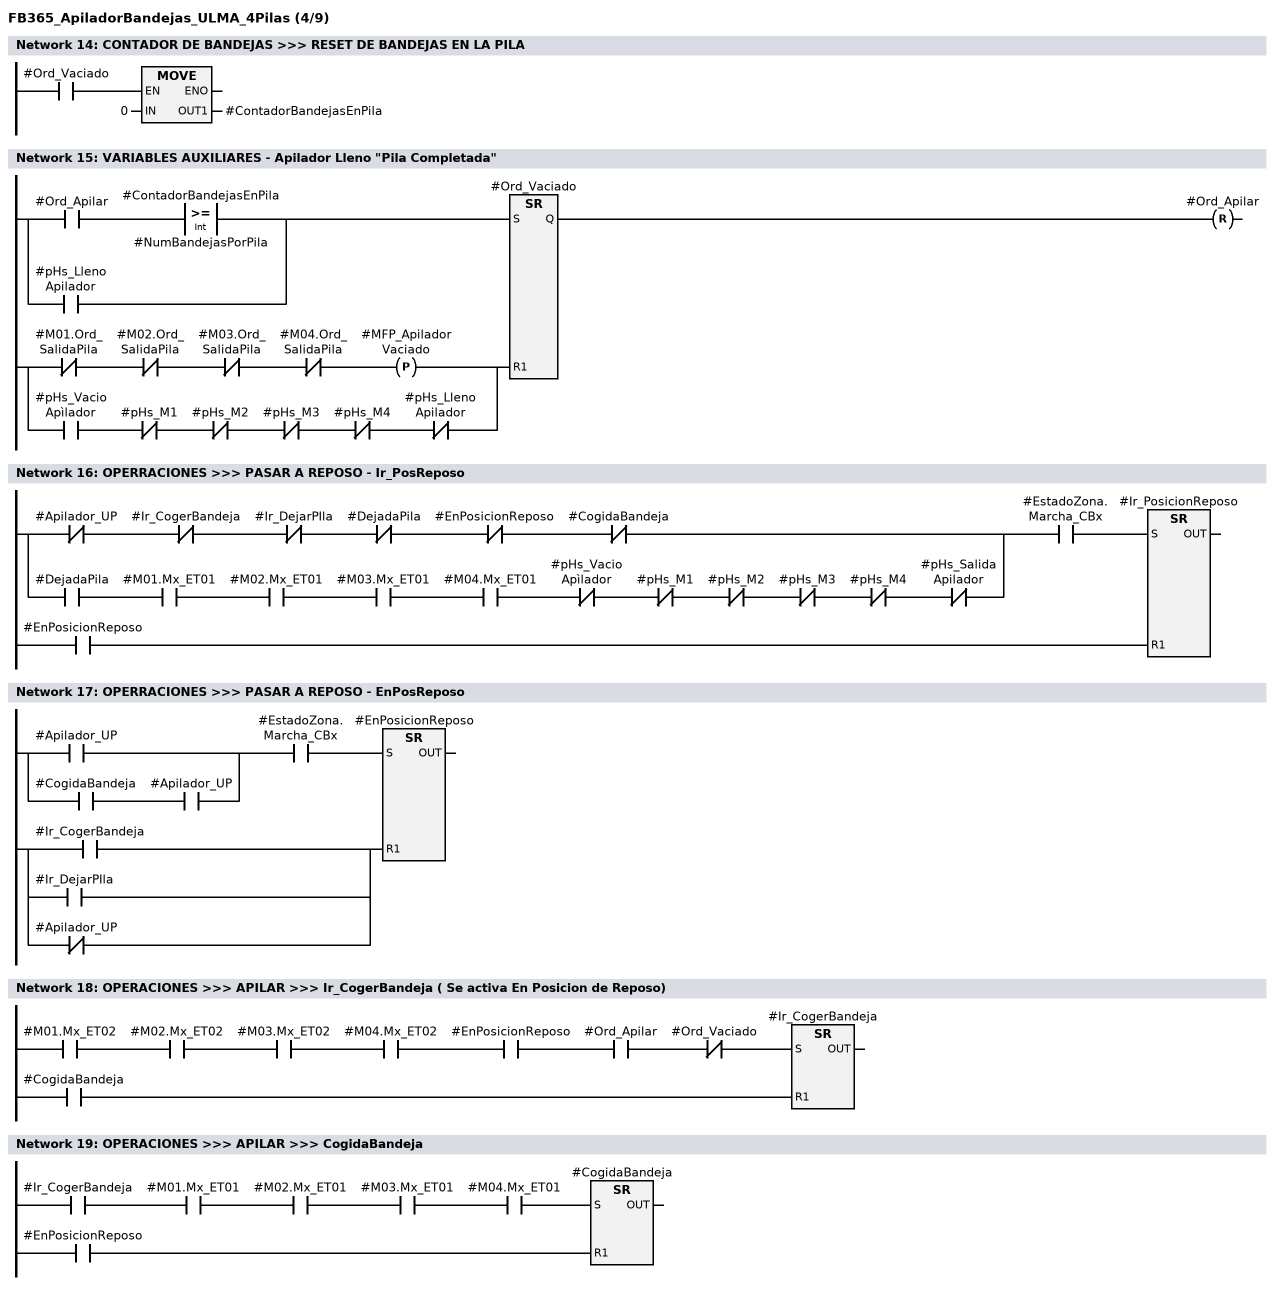
   RUNG wire#powerrail
      Contact( #Ord_Vaciado )
      { S7_GenerateENO := "TRUE" } Move(in := 0, out1 => #ContadorBandejasEnPila)
   END_RUNG
   // the same network as SCL:
   IF #Ord_Vaciado THEN #ContadorBandejasEnPila := 0; END_IF;
END_REGION

REGION Network 15: VARIABLES AUXILIARES - Apilador Lleno "Pila Completada"
   RUNG wire#powerrail
      Contact( #Ord_Apilar )
      { S7_Templates := "SrcType := Int" } GE_Contact(in1 := #ContadorBandejasEnPila, in2 := #NumBandejasPorPila)
      wire#w1
      S_SR(operand := #Ord_Vaciado, r1 := wire#w2)
      R_Coil( #Ord_Apilar )
   END_RUNG
   RUNG wire#powerrail
      Contact( #pHs_LlenoApilador )
   END_RUNG wire#w1
   RUNG wire#powerrail
      I_Contact( #M01.Ord_SalidaPila )
      I_Contact( #M02.Ord_SalidaPila )
      I_Contact( #M03.Ord_SalidaPila )
      I_Contact( #M04.Ord_SalidaPila )
      P_Trig( #MFP_ApiladorVaciado )
   END_RUNG wire#w2
   RUNG wire#powerrail
      Contact( #pHs_VacioApìlador )
      I_Contact( #pHs_M1 )
      I_Contact( #pHs_M2 )
      I_Contact( #pHs_M3 )
      I_Contact( #pHs_M4 )
      I_Contact( #pHs_LlenoApilador )
   END_RUNG wire#w2
   // the same network as SCL:
   #_w1 := NOT #M01.Ord_SalidaPila AND NOT #M02.Ord_SalidaPila AND NOT #M03.Ord_SalidaPila AND NOT #M04.Ord_SalidaPila;
   #_w2 := #_w1 AND NOT #MFP_ApiladorVaciado;   // rising edge
   #MFP_ApiladorVaciado := #_w1;
   IF (#Ord_Apilar AND (#ContadorBandejasEnPila >= #NumBandejasPorPila)) OR #pHs_LlenoApilador THEN
       #Ord_Vaciado := TRUE;   // SR flip-flop
   END_IF;
   IF #_w2 OR (#pHs_VacioApìlador AND NOT #pHs_M1 AND NOT #pHs_M2 AND NOT #pHs_M3 AND NOT #pHs_M4 AND NOT #pHs_LlenoApilador) THEN
       #Ord_Vaciado := FALSE;
   END_IF;
   IF #Ord_Vaciado THEN #Ord_Apilar := FALSE; END_IF;
END_REGION

REGION Network 16: OPERRACIONES >>> PASAR A REPOSO - Ir_PosReposo
   RUNG wire#powerrail
      I_Contact( #Apilador_UP )
      I_Contact( #Ir_CogerBandeja )
      I_Contact( #Ir_DejarPIla )
      I_Contact( #DejadaPila )
      I_Contact( #EnPosicionReposo )
      I_Contact( #CogidaBandeja )
      wire#w1
      Contact( #EstadoZona.Marcha_CBx )
      S_SR(operand := #Ir_PosicionReposo, r1 := wire#w2)
   END_RUNG
   RUNG wire#powerrail
      Contact( #DejadaPila )
      Contact( #M01.Mx_ET01 )
      Contact( #M02.Mx_ET01 )
      Contact( #M03.Mx_ET01 )
      Contact( #M04.Mx_ET01 )
      I_Contact( #pHs_VacioApìlador )
      I_Contact( #pHs_M1 )
      I_Contact( #pHs_M2 )
      I_Contact( #pHs_M3 )
      I_Contact( #pHs_M4 )
      I_Contact( #pHs_SalidaApilador )
   END_RUNG wire#w1
   RUNG wire#powerrail
      Contact( #EnPosicionReposo )
   END_RUNG wire#w2
   // the same network as SCL:
   IF ((NOT #Apilador_UP AND NOT #Ir_CogerBandeja AND NOT #Ir_DejarPIla AND NOT #DejadaPila AND NOT #EnPosicionReposo AND NOT #CogidaBandeja) OR (#DejadaPila AND #M01.Mx_ET01 AND #M02.Mx_ET01 AND #M03.Mx_ET01 AND #M04.Mx_ET01 AND NOT #pHs_VacioApìlador AND NOT #pHs_M1 AND NOT #pHs_M2 AND NOT #pHs_M3 AND NOT #pHs_M4 AND NOT #pHs_SalidaApilador)) AND #EstadoZona.Marcha_CBx THEN
       #Ir_PosicionReposo := TRUE;   // SR flip-flop
   END_IF;
   IF #EnPosicionReposo THEN #Ir_PosicionReposo := FALSE; END_IF;
END_REGION

REGION Network 17: OPERRACIONES >>> PASAR A REPOSO - EnPosReposo
   RUNG wire#powerrail
      Contact( #Apilador_UP )
      wire#w1
      Contact( #EstadoZona.Marcha_CBx )
      S_SR(operand := #EnPosicionReposo, r1 := wire#w2)
   END_RUNG
   RUNG wire#powerrail
      Contact( #CogidaBandeja )
      Contact( #Apilador_UP )
   END_RUNG wire#w1
   RUNG wire#powerrail
      Contact( #Ir_CogerBandeja )
   END_RUNG wire#w2
   RUNG wire#powerrail
      Contact( #Ir_DejarPIla )
   END_RUNG wire#w2
   RUNG wire#powerrail
      I_Contact( #Apilador_UP )
   END_RUNG wire#w2
   // the same network as SCL:
   IF (#Apilador_UP OR (#CogidaBandeja AND #Apilador_UP)) AND #EstadoZona.Marcha_CBx THEN
       #EnPosicionReposo := TRUE;   // SR flip-flop
   END_IF;
   IF #Ir_CogerBandeja OR #Ir_DejarPIla OR NOT #Apilador_UP THEN #EnPosicionReposo := FALSE; END_IF;
END_REGION

REGION Network 18: OPERACIONES >>> APILAR >>> Ir_CogerBandeja ( Se activa En Posicion de Reposo)
   RUNG wire#powerrail
      Contact( #M01.Mx_ET02 )
      Contact( #M02.Mx_ET02 )
      Contact( #M03.Mx_ET02 )
      Contact( #M04.Mx_ET02 )
      Contact( #EnPosicionReposo )
      Contact( #Ord_Apilar )
      I_Contact( #Ord_Vaciado )
      S_SR(operand := #Ir_CogerBandeja, r1 := wire#w1)
   END_RUNG
   RUNG wire#powerrail
      Contact( #CogidaBandeja )
   END_RUNG wire#w1
   // the same network as SCL:
   IF #M01.Mx_ET02 AND #M02.Mx_ET02 AND #M03.Mx_ET02 AND #M04.Mx_ET02 AND #EnPosicionReposo AND #Ord_Apilar AND NOT #Ord_Vaciado THEN
       #Ir_CogerBandeja := TRUE;   // SR flip-flop
   END_IF;
   IF #CogidaBandeja THEN #Ir_CogerBandeja := FALSE; END_IF;
END_REGION

REGION Network 19: OPERACIONES >>> APILAR >>> CogidaBandeja
   RUNG wire#powerrail
      Contact( #Ir_CogerBandeja )
      Contact( #M01.Mx_ET01 )
      Contact( #M02.Mx_ET01 )
      Contact( #M03.Mx_ET01 )
      Contact( #M04.Mx_ET01 )
      S_SR(operand := #CogidaBandeja, r1 := wire#w1)
   END_RUNG
   RUNG wire#powerrail
      Contact( #EnPosicionReposo )
   END_RUNG wire#w1
   // the same network as SCL:
   IF #Ir_CogerBandeja AND #M01.Mx_ET01 AND #M02.Mx_ET01 AND #M03.Mx_ET01 AND #M04.Mx_ET01 THEN
       #CogidaBandeja := TRUE;   // SR flip-flop
   END_IF;
   IF #EnPosicionReposo THEN #CogidaBandeja := FALSE; END_IF;
END_REGION

REGION Network 20: OPERACIONES >>> VACIAR PILAS >>> Ir_DejarPila ( Se activa En Posicion de Reposo)
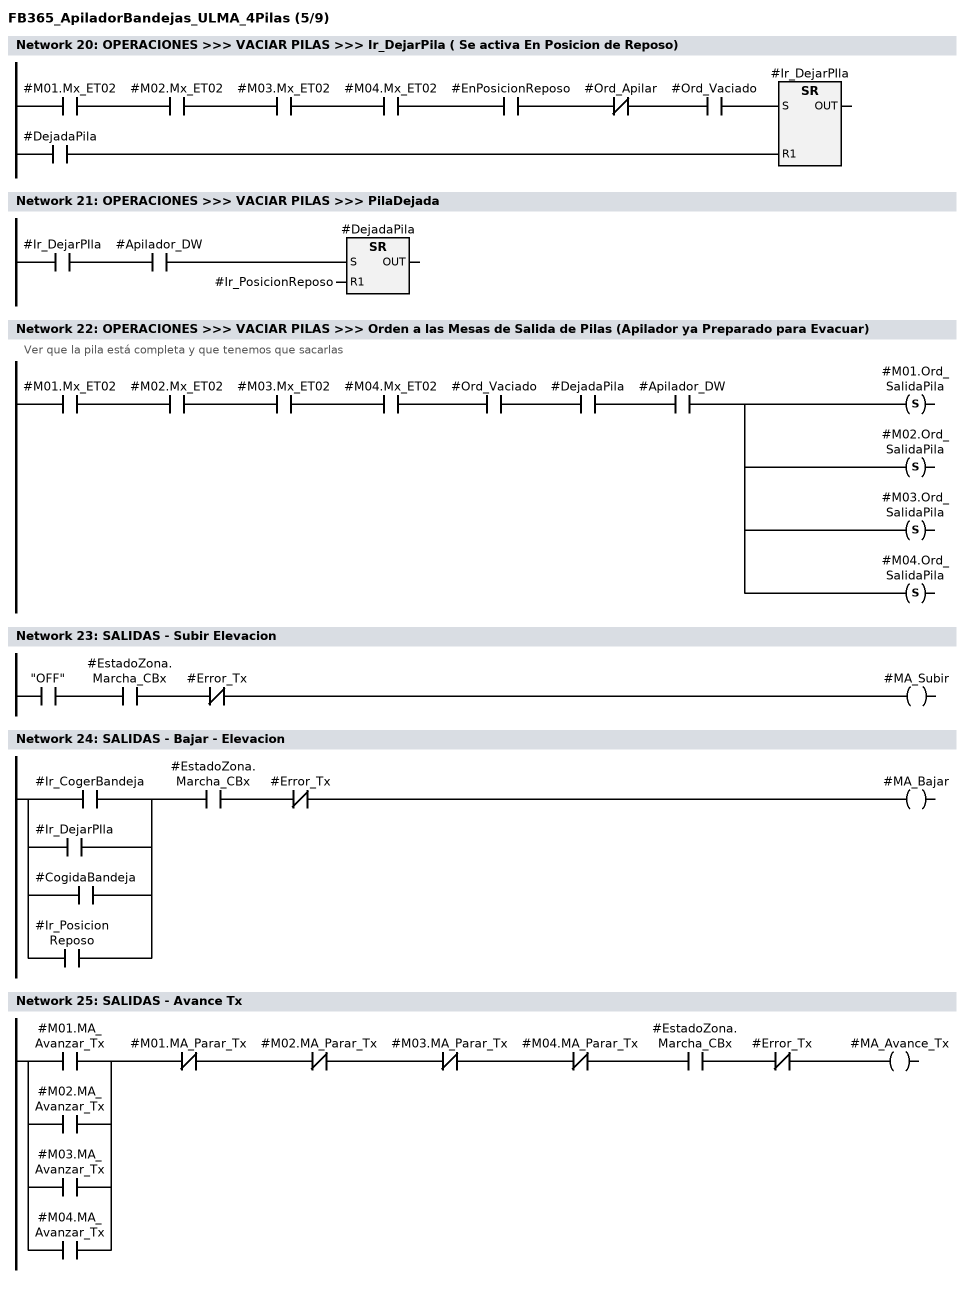
   RUNG wire#powerrail
      Contact( #M01.Mx_ET02 )
      Contact( #M02.Mx_ET02 )
      Contact( #M03.Mx_ET02 )
      Contact( #M04.Mx_ET02 )
      Contact( #EnPosicionReposo )
      I_Contact( #Ord_Apilar )
      Contact( #Ord_Vaciado )
      S_SR(operand := #Ir_DejarPIla, r1 := wire#w1)
   END_RUNG
   RUNG wire#powerrail
      Contact( #DejadaPila )
   END_RUNG wire#w1
   // the same network as SCL:
   IF #M01.Mx_ET02 AND #M02.Mx_ET02 AND #M03.Mx_ET02 AND #M04.Mx_ET02 AND #EnPosicionReposo AND NOT #Ord_Apilar AND #Ord_Vaciado THEN
       #Ir_DejarPIla := TRUE;   // SR flip-flop
   END_IF;
   IF #DejadaPila THEN #Ir_DejarPIla := FALSE; END_IF;
END_REGION

REGION Network 21: OPERACIONES >>> VACIAR PILAS >>> PilaDejada
   RUNG wire#powerrail
      Contact( #Ir_DejarPIla )
      Contact( #Apilador_DW )
      S_SR(operand := #DejadaPila, r1 := #Ir_PosicionReposo)
   END_RUNG
   // the same network as SCL:
   IF #Ir_DejarPIla AND #Apilador_DW THEN
       #DejadaPila := TRUE;   // SR flip-flop
   END_IF;
   IF #Ir_PosicionReposo THEN #DejadaPila := FALSE; END_IF;
END_REGION

REGION Network 22: OPERACIONES >>> VACIAR PILAS >>> Orden a las Mesas de Salida de Pilas (Apilador ya Preparado para Evacuar)
   // Ver que la pila está completa y que tenemos que sacarlas
   RUNG wire#powerrail
      Contact( #M01.Mx_ET02 )
      Contact( #M02.Mx_ET02 )
      Contact( #M03.Mx_ET02 )
      Contact( #M04.Mx_ET02 )
      Contact( #Ord_Vaciado )
      Contact( #DejadaPila )
      Contact( #Apilador_DW )
      wire#w1
      S_Coil( #M01.Ord_SalidaPila )
   END_RUNG
   RUNG wire#w1
      S_Coil( #M02.Ord_SalidaPila )
   END_RUNG
   RUNG wire#w1
      S_Coil( #M03.Ord_SalidaPila )
   END_RUNG
   RUNG wire#w1
      S_Coil( #M04.Ord_SalidaPila )
   END_RUNG
   // the same network as SCL:
   IF #M01.Mx_ET02 AND #M02.Mx_ET02 AND #M03.Mx_ET02 AND #M04.Mx_ET02 AND #Ord_Vaciado AND #DejadaPila AND #Apilador_DW THEN
       #M01.Ord_SalidaPila := TRUE;
       #M02.Ord_SalidaPila := TRUE;
       #M03.Ord_SalidaPila := TRUE;
       #M04.Ord_SalidaPila := TRUE;
   END_IF;
END_REGION

REGION Network 23: SALIDAS - Subir Elevacion
   RUNG wire#powerrail
      Contact( "OFF" )
      Contact( #EstadoZona.Marcha_CBx )
      I_Contact( #Error_Tx )
      Coil( #MA_Subir )
   END_RUNG
   // the same network as SCL:
   #MA_Subir := "OFF" AND #EstadoZona.Marcha_CBx AND NOT #Error_Tx;
END_REGION

REGION Network 24: SALIDAS - Bajar - Elevacion
   RUNG wire#powerrail
      Contact( #Ir_CogerBandeja )
      wire#w1
      Contact( #EstadoZona.Marcha_CBx )
      I_Contact( #Error_Tx )
      Coil( #MA_Bajar )
   END_RUNG
   RUNG wire#powerrail
      Contact( #Ir_DejarPIla )
   END_RUNG wire#w1
   RUNG wire#powerrail
      Contact( #CogidaBandeja )
   END_RUNG wire#w1
   RUNG wire#powerrail
      Contact( #Ir_PosicionReposo )
   END_RUNG wire#w1
   // the same network as SCL:
   #MA_Bajar := (#Ir_CogerBandeja OR #Ir_DejarPIla OR #CogidaBandeja OR #Ir_PosicionReposo) AND #EstadoZona.Marcha_CBx AND NOT #Error_Tx;
END_REGION

REGION Network 25: SALIDAS - Avance Tx
   RUNG wire#powerrail
      Contact( #M01.MA_Avanzar_Tx )
      wire#w1
      I_Contact( #M01.MA_Parar_Tx )
      I_Contact( #M02.MA_Parar_Tx )
      I_Contact( #M03.MA_Parar_Tx )
      I_Contact( #M04.MA_Parar_Tx )
      Contact( #EstadoZona.Marcha_CBx )
      I_Contact( #Error_Tx )
      Coil( #MA_Avance_Tx )
   END_RUNG
   RUNG wire#powerrail
      Contact( #M02.MA_Avanzar_Tx )
   END_RUNG wire#w1
   RUNG wire#powerrail
      Contact( #M03.MA_Avanzar_Tx )
   END_RUNG wire#w1
   RUNG wire#powerrail
      Contact( #M04.MA_Avanzar_Tx )
   END_RUNG wire#w1
   // the same network as SCL:
   #MA_Avance_Tx := (#M01.MA_Avanzar_Tx OR #M02.MA_Avanzar_Tx OR #M03.MA_Avanzar_Tx OR #M04.MA_Avanzar_Tx) AND NOT #M01.MA_Parar_Tx AND NOT #M02.MA_Parar_Tx AND NOT #M03.MA_Parar_Tx AND NOT #M04.MA_Parar_Tx AND #EstadoZona.Marcha_CBx AND NOT #Error_Tx;
END_REGION

REGION Network 26: SALIDAS - Retroceder Tx
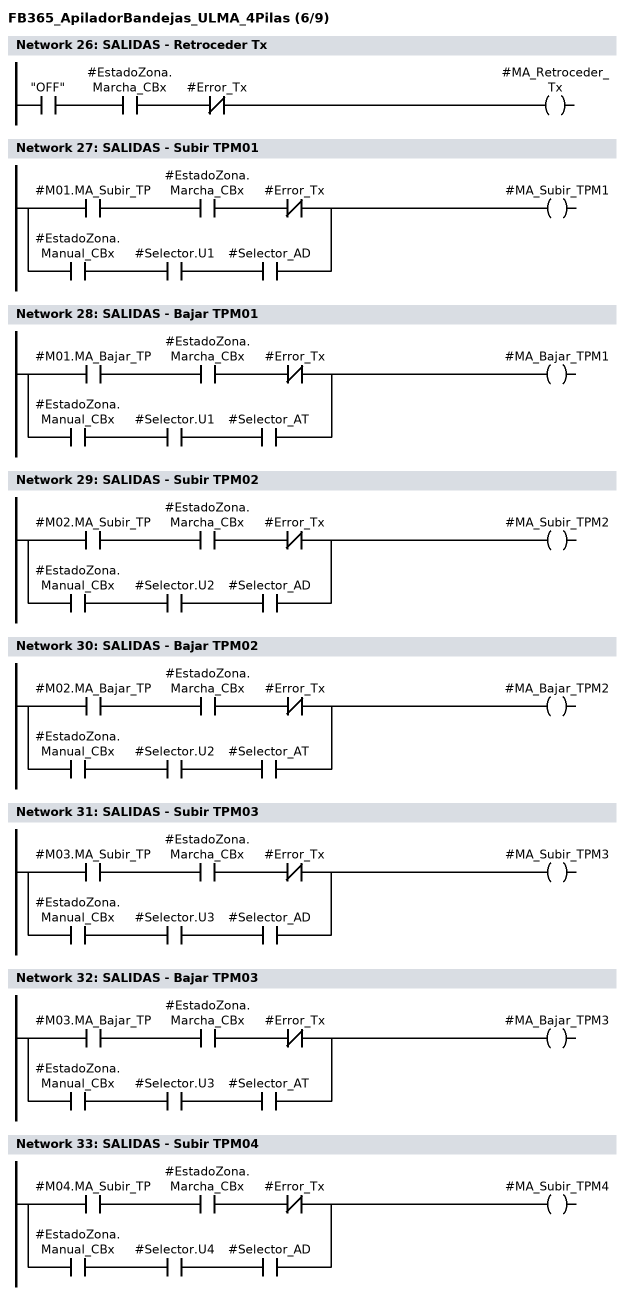
   RUNG wire#powerrail
      Contact( "OFF" )
      Contact( #EstadoZona.Marcha_CBx )
      I_Contact( #Error_Tx )
      Coil( #MA_Retroceder_Tx )
   END_RUNG
   // the same network as SCL:
   #MA_Retroceder_Tx := "OFF" AND #EstadoZona.Marcha_CBx AND NOT #Error_Tx;
END_REGION

REGION Network 27: SALIDAS - Subir TPM01
   RUNG wire#powerrail
      Contact( #M01.MA_Subir_TP )
      Contact( #EstadoZona.Marcha_CBx )
      I_Contact( #Error_Tx )
      wire#w1
      Coil( #MA_Subir_TPM1 )
   END_RUNG
   RUNG wire#powerrail
      Contact( #EstadoZona.Manual_CBx )
      Contact( #Selector.U1 )
      Contact( #Selector_AD )
   END_RUNG wire#w1
   // the same network as SCL:
   #MA_Subir_TPM1 := (#M01.MA_Subir_TP AND #EstadoZona.Marcha_CBx AND NOT #Error_Tx) OR (#EstadoZona.Manual_CBx AND #Selector.U1 AND #Selector_AD);
END_REGION

REGION Network 28: SALIDAS - Bajar TPM01
   RUNG wire#powerrail
      Contact( #M01.MA_Bajar_TP )
      Contact( #EstadoZona.Marcha_CBx )
      I_Contact( #Error_Tx )
      wire#w1
      Coil( #MA_Bajar_TPM1 )
   END_RUNG
   RUNG wire#powerrail
      Contact( #EstadoZona.Manual_CBx )
      Contact( #Selector.U1 )
      Contact( #Selector_AT )
   END_RUNG wire#w1
   // the same network as SCL:
   #MA_Bajar_TPM1 := (#M01.MA_Bajar_TP AND #EstadoZona.Marcha_CBx AND NOT #Error_Tx) OR (#EstadoZona.Manual_CBx AND #Selector.U1 AND #Selector_AT);
END_REGION

REGION Network 29: SALIDAS - Subir TPM02
   RUNG wire#powerrail
      Contact( #M02.MA_Subir_TP )
      Contact( #EstadoZona.Marcha_CBx )
      I_Contact( #Error_Tx )
      wire#w1
      Coil( #MA_Subir_TPM2 )
   END_RUNG
   RUNG wire#powerrail
      Contact( #EstadoZona.Manual_CBx )
      Contact( #Selector.U2 )
      Contact( #Selector_AD )
   END_RUNG wire#w1
   // the same network as SCL:
   #MA_Subir_TPM2 := (#M02.MA_Subir_TP AND #EstadoZona.Marcha_CBx AND NOT #Error_Tx) OR (#EstadoZona.Manual_CBx AND #Selector.U2 AND #Selector_AD);
END_REGION

REGION Network 30: SALIDAS - Bajar TPM02
   RUNG wire#powerrail
      Contact( #M02.MA_Bajar_TP )
      Contact( #EstadoZona.Marcha_CBx )
      I_Contact( #Error_Tx )
      wire#w1
      Coil( #MA_Bajar_TPM2 )
   END_RUNG
   RUNG wire#powerrail
      Contact( #EstadoZona.Manual_CBx )
      Contact( #Selector.U2 )
      Contact( #Selector_AT )
   END_RUNG wire#w1
   // the same network as SCL:
   #MA_Bajar_TPM2 := (#M02.MA_Bajar_TP AND #EstadoZona.Marcha_CBx AND NOT #Error_Tx) OR (#EstadoZona.Manual_CBx AND #Selector.U2 AND #Selector_AT);
END_REGION

REGION Network 31: SALIDAS - Subir TPM03
   RUNG wire#powerrail
      Contact( #M03.MA_Subir_TP )
      Contact( #EstadoZona.Marcha_CBx )
      I_Contact( #Error_Tx )
      wire#w1
      Coil( #MA_Subir_TPM3 )
   END_RUNG
   RUNG wire#powerrail
      Contact( #EstadoZona.Manual_CBx )
      Contact( #Selector.U3 )
      Contact( #Selector_AD )
   END_RUNG wire#w1
   // the same network as SCL:
   #MA_Subir_TPM3 := (#M03.MA_Subir_TP AND #EstadoZona.Marcha_CBx AND NOT #Error_Tx) OR (#EstadoZona.Manual_CBx AND #Selector.U3 AND #Selector_AD);
END_REGION

REGION Network 32: SALIDAS - Bajar TPM03
   RUNG wire#powerrail
      Contact( #M03.MA_Bajar_TP )
      Contact( #EstadoZona.Marcha_CBx )
      I_Contact( #Error_Tx )
      wire#w1
      Coil( #MA_Bajar_TPM3 )
   END_RUNG
   RUNG wire#powerrail
      Contact( #EstadoZona.Manual_CBx )
      Contact( #Selector.U3 )
      Contact( #Selector_AT )
   END_RUNG wire#w1
   // the same network as SCL:
   #MA_Bajar_TPM3 := (#M03.MA_Bajar_TP AND #EstadoZona.Marcha_CBx AND NOT #Error_Tx) OR (#EstadoZona.Manual_CBx AND #Selector.U3 AND #Selector_AT);
END_REGION

REGION Network 33: SALIDAS - Subir TPM04
   RUNG wire#powerrail
      Contact( #M04.MA_Subir_TP )
      Contact( #EstadoZona.Marcha_CBx )
      I_Contact( #Error_Tx )
      wire#w1
      Coil( #MA_Subir_TPM4 )
   END_RUNG
   RUNG wire#powerrail
      Contact( #EstadoZona.Manual_CBx )
      Contact( #Selector.U4 )
      Contact( #Selector_AD )
   END_RUNG wire#w1
   // the same network as SCL:
   #MA_Subir_TPM4 := (#M04.MA_Subir_TP AND #EstadoZona.Marcha_CBx AND NOT #Error_Tx) OR (#EstadoZona.Manual_CBx AND #Selector.U4 AND #Selector_AD);
END_REGION

REGION Network 34: SALIDAS - Bajar TPM04
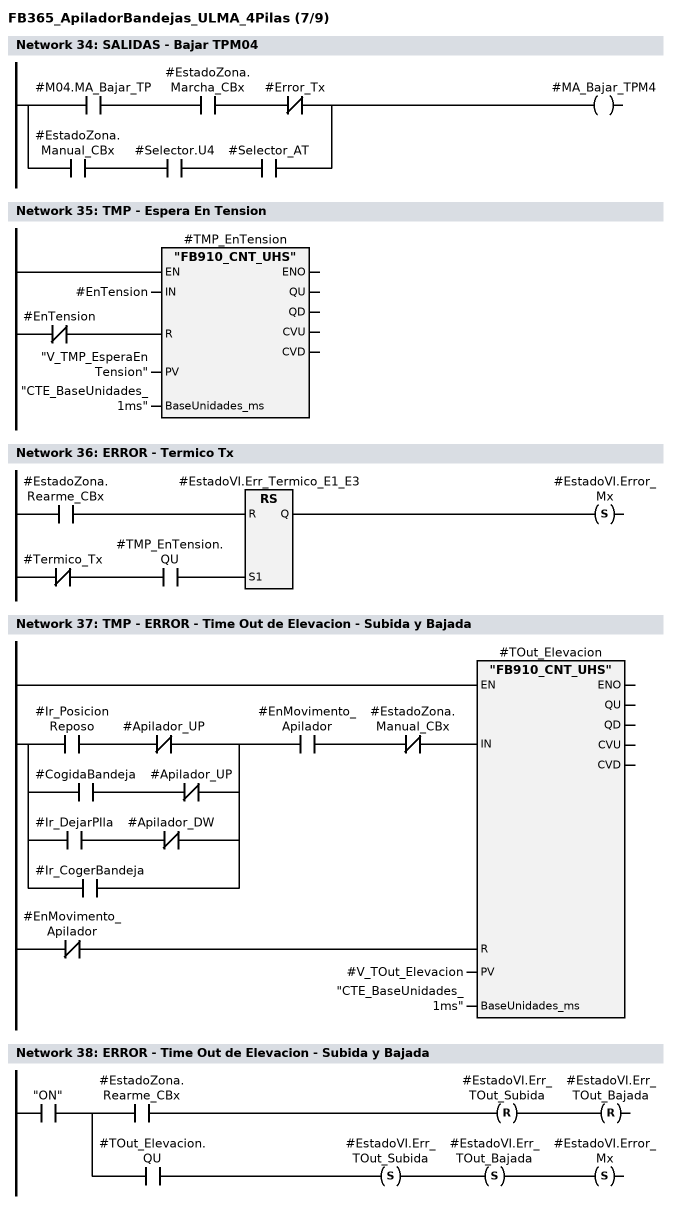
   RUNG wire#powerrail
      Contact( #M04.MA_Bajar_TP )
      Contact( #EstadoZona.Marcha_CBx )
      I_Contact( #Error_Tx )
      wire#w1
      Coil( #MA_Bajar_TPM4 )
   END_RUNG
   RUNG wire#powerrail
      Contact( #EstadoZona.Manual_CBx )
      Contact( #Selector.U4 )
      Contact( #Selector_AT )
   END_RUNG wire#w1
   // the same network as SCL:
   #MA_Bajar_TPM4 := (#M04.MA_Bajar_TP AND #EstadoZona.Marcha_CBx AND NOT #Error_Tx) OR (#EstadoZona.Manual_CBx AND #Selector.U4 AND #Selector_AT);
END_REGION

REGION Network 35: TMP - Espera En Tension
   RUNG wire#powerrail
      #TMP_EnTension(R := wire#w1, IN := #EnTension, PV := "V_TMP_EsperaEnTension", BaseUnidades_ms := "CTE_BaseUnidades_1ms", QU =>, QD =>, CVU =>, CVD =>)
   END_RUNG
   RUNG wire#powerrail
      I_Contact( #EnTension )
   END_RUNG wire#w1
   // the same network as SCL:
   #TMP_EnTension(IN := #EnTension,   // "FB910_CNT_UHS"
                  R := NOT #EnTension,
                  PV := "V_TMP_EsperaEnTension",
                  BaseUnidades_ms := "CTE_BaseUnidades_1ms");
END_REGION

REGION Network 36: ERROR - Termico Tx
   RUNG wire#powerrail
      Contact( #EstadoZona.Rearme_CBx )
      S_RS(operand := #EstadoVI.Err_Termico_E1_E3, s1 := wire#w1)
      S_Coil( #EstadoVI.Error_Mx )
   END_RUNG
   RUNG wire#powerrail
      I_Contact( #Termico_Tx )
      Contact( #TMP_EnTension.QU )
   END_RUNG wire#w1
   // the same network as SCL:
   IF #EstadoZona.Rearme_CBx THEN
       #EstadoVI.Err_Termico_E1_E3 := FALSE;   // RS flip-flop
   END_IF;
   IF NOT #Termico_Tx AND #TMP_EnTension.QU THEN #EstadoVI.Err_Termico_E1_E3 := TRUE; END_IF;
   IF #EstadoVI.Err_Termico_E1_E3 THEN #EstadoVI.Error_Mx := TRUE; END_IF;
END_REGION

REGION Network 37: TMP - ERROR - Time Out de Elevacion - Subida y Bajada
   RUNG wire#powerrail
      #TOut_Elevacion(IN := wire#w2, R := wire#w3, PV := #V_TOut_Elevacion, BaseUnidades_ms := "CTE_BaseUnidades_1ms", QU =>, QD =>, CVU =>, CVD =>)
   END_RUNG
   RUNG wire#powerrail
      Contact( #Ir_PosicionReposo )
      I_Contact( #Apilador_UP )
      wire#w1
      Contact( #EnMovimento_Apilador )
      I_Contact( #EstadoZona.Manual_CBx )
   END_RUNG wire#w2
   RUNG wire#powerrail
      Contact( #CogidaBandeja )
      I_Contact( #Apilador_UP )
   END_RUNG wire#w1
   RUNG wire#powerrail
      Contact( #Ir_DejarPIla )
      I_Contact( #Apilador_DW )
   END_RUNG wire#w1
   RUNG wire#powerrail
      Contact( #Ir_CogerBandeja )
   END_RUNG wire#w1
   RUNG wire#powerrail
      I_Contact( #EnMovimento_Apilador )
   END_RUNG wire#w3
   // the same network as SCL:
   #TOut_Elevacion(IN := ((#Ir_PosicionReposo AND NOT #Apilador_UP) OR (#CogidaBandeja AND NOT #Apilador_UP) OR (#Ir_DejarPIla AND NOT #Apilador_DW) OR #Ir_CogerBandeja) AND #EnMovimento_Apilador AND NOT #EstadoZona.Manual_CBx,   // "FB910_CNT_UHS"
                   R := NOT #EnMovimento_Apilador,
                   PV := #V_TOut_Elevacion,
                   BaseUnidades_ms := "CTE_BaseUnidades_1ms");
END_REGION

REGION Network 38: ERROR - Time Out de Elevacion - Subida y Bajada
   RUNG wire#powerrail
      Contact( "ON" )
      wire#w1
      Contact( #EstadoZona.Rearme_CBx )
      R_Coil( #EstadoVI.Err_TOut_Subida )
      R_Coil( #EstadoVI.Err_TOut_Bajada )
   END_RUNG
   RUNG wire#w1
      Contact( #TOut_Elevacion.QU )
      S_Coil( #EstadoVI.Err_TOut_Subida )
      S_Coil( #EstadoVI.Err_TOut_Bajada )
      S_Coil( #EstadoVI.Error_Mx )
   END_RUNG
   // the same network as SCL:
   IF "ON" AND #EstadoZona.Rearme_CBx THEN
       #EstadoVI.Err_TOut_Subida := FALSE;
       #EstadoVI.Err_TOut_Bajada := FALSE;
   END_IF;
   IF "ON" AND #TOut_Elevacion.QU THEN
       #EstadoVI.Err_TOut_Subida := TRUE;
       #EstadoVI.Err_TOut_Bajada := TRUE;
       #EstadoVI.Error_Mx := TRUE;
   END_IF;
END_REGION

REGION Network 39: ERROR - TimeOut de Atasco
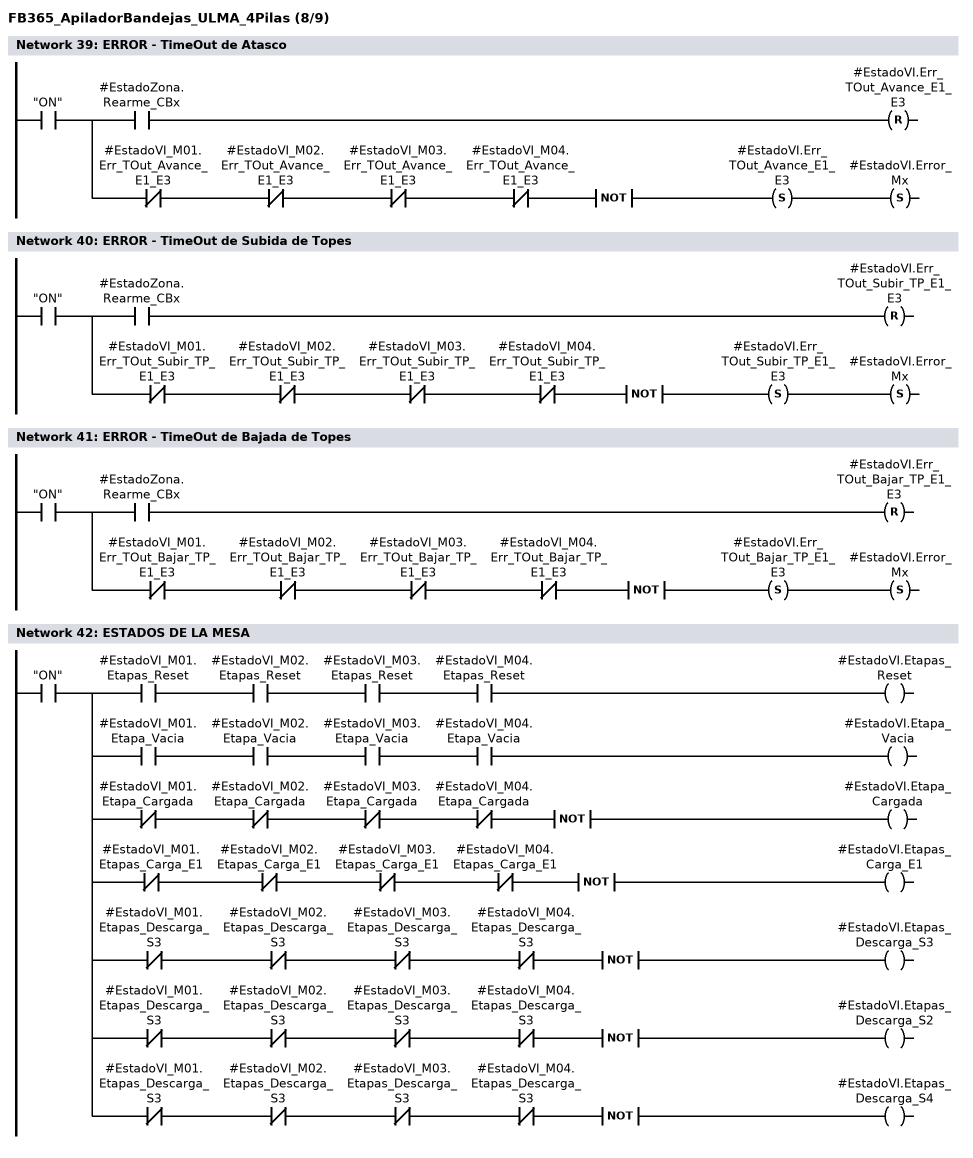
   RUNG wire#powerrail
      Contact( "ON" )
      wire#w1
      Contact( #EstadoZona.Rearme_CBx )
      R_Coil( #EstadoVI.Err_TOut_Avance_E1_E3 )
   END_RUNG
   RUNG wire#w1
      I_Contact( #EstadoVI_M01.Err_TOut_Avance_E1_E3 )
      I_Contact( #EstadoVI_M02.Err_TOut_Avance_E1_E3 )
      I_Contact( #EstadoVI_M03.Err_TOut_Avance_E1_E3 )
      I_Contact( #EstadoVI_M04.Err_TOut_Avance_E1_E3 )
      Not()
      S_Coil( #EstadoVI.Err_TOut_Avance_E1_E3 )
      S_Coil( #EstadoVI.Error_Mx )
   END_RUNG
   // the same network as SCL:
   IF "ON" AND #EstadoZona.Rearme_CBx THEN #EstadoVI.Err_TOut_Avance_E1_E3 := FALSE; END_IF;
   IF NOT ("ON" AND NOT #EstadoVI_M01.Err_TOut_Avance_E1_E3 AND NOT #EstadoVI_M02.Err_TOut_Avance_E1_E3 AND NOT #EstadoVI_M03.Err_TOut_Avance_E1_E3 AND NOT #EstadoVI_M04.Err_TOut_Avance_E1_E3) THEN
       #EstadoVI.Err_TOut_Avance_E1_E3 := TRUE;
       #EstadoVI.Error_Mx := TRUE;
   END_IF;
END_REGION

REGION Network 40: ERROR - TimeOut de Subida de Topes
   RUNG wire#powerrail
      Contact( "ON" )
      wire#w1
      Contact( #EstadoZona.Rearme_CBx )
      R_Coil( #EstadoVI.Err_TOut_Subir_TP_E1_E3 )
   END_RUNG
   RUNG wire#w1
      I_Contact( #EstadoVI_M01.Err_TOut_Subir_TP_E1_E3 )
      I_Contact( #EstadoVI_M02.Err_TOut_Subir_TP_E1_E3 )
      I_Contact( #EstadoVI_M03.Err_TOut_Subir_TP_E1_E3 )
      I_Contact( #EstadoVI_M04.Err_TOut_Subir_TP_E1_E3 )
      Not()
      S_Coil( #EstadoVI.Err_TOut_Subir_TP_E1_E3 )
      S_Coil( #EstadoVI.Error_Mx )
   END_RUNG
   // the same network as SCL:
   IF "ON" AND #EstadoZona.Rearme_CBx THEN #EstadoVI.Err_TOut_Subir_TP_E1_E3 := FALSE; END_IF;
   IF NOT ("ON" AND NOT #EstadoVI_M01.Err_TOut_Subir_TP_E1_E3 AND NOT #EstadoVI_M02.Err_TOut_Subir_TP_E1_E3 AND NOT #EstadoVI_M03.Err_TOut_Subir_TP_E1_E3 AND NOT #EstadoVI_M04.Err_TOut_Subir_TP_E1_E3) THEN
       #EstadoVI.Err_TOut_Subir_TP_E1_E3 := TRUE;
       #EstadoVI.Error_Mx := TRUE;
   END_IF;
END_REGION

REGION Network 41: ERROR - TimeOut de Bajada de Topes
   RUNG wire#powerrail
      Contact( "ON" )
      wire#w1
      Contact( #EstadoZona.Rearme_CBx )
      R_Coil( #EstadoVI.Err_TOut_Bajar_TP_E1_E3 )
   END_RUNG
   RUNG wire#w1
      I_Contact( #EstadoVI_M01.Err_TOut_Bajar_TP_E1_E3 )
      I_Contact( #EstadoVI_M02.Err_TOut_Bajar_TP_E1_E3 )
      I_Contact( #EstadoVI_M03.Err_TOut_Bajar_TP_E1_E3 )
      I_Contact( #EstadoVI_M04.Err_TOut_Bajar_TP_E1_E3 )
      Not()
      S_Coil( #EstadoVI.Err_TOut_Bajar_TP_E1_E3 )
      S_Coil( #EstadoVI.Error_Mx )
   END_RUNG
   // the same network as SCL:
   IF "ON" AND #EstadoZona.Rearme_CBx THEN #EstadoVI.Err_TOut_Bajar_TP_E1_E3 := FALSE; END_IF;
   IF NOT ("ON" AND NOT #EstadoVI_M01.Err_TOut_Bajar_TP_E1_E3 AND NOT #EstadoVI_M02.Err_TOut_Bajar_TP_E1_E3 AND NOT #EstadoVI_M03.Err_TOut_Bajar_TP_E1_E3 AND NOT #EstadoVI_M04.Err_TOut_Bajar_TP_E1_E3) THEN
       #EstadoVI.Err_TOut_Bajar_TP_E1_E3 := TRUE;
       #EstadoVI.Error_Mx := TRUE;
   END_IF;
END_REGION

REGION Network 42: ESTADOS DE LA MESA
   RUNG wire#powerrail
      Contact( "ON" )
      wire#w1
      Contact( #EstadoVI_M01.Etapas_Reset )
      Contact( #EstadoVI_M02.Etapas_Reset )
      Contact( #EstadoVI_M03.Etapas_Reset )
      Contact( #EstadoVI_M04.Etapas_Reset )
      Coil( #EstadoVI.Etapas_Reset )
   END_RUNG
   RUNG wire#w1
      Contact( #EstadoVI_M01.Etapa_Vacia )
      Contact( #EstadoVI_M02.Etapa_Vacia )
      Contact( #EstadoVI_M03.Etapa_Vacia )
      Contact( #EstadoVI_M04.Etapa_Vacia )
      Coil( #EstadoVI.Etapa_Vacia )
   END_RUNG
   RUNG wire#w1
      I_Contact( #EstadoVI_M01.Etapa_Cargada )
      I_Contact( #EstadoVI_M02.Etapa_Cargada )
      I_Contact( #EstadoVI_M03.Etapa_Cargada )
      I_Contact( #EstadoVI_M04.Etapa_Cargada )
      Not()
      Coil( #EstadoVI.Etapa_Cargada )
   END_RUNG
   RUNG wire#w1
      I_Contact( #EstadoVI_M01.Etapas_Carga_E1 )
      I_Contact( #EstadoVI_M02.Etapas_Carga_E1 )
      I_Contact( #EstadoVI_M03.Etapas_Carga_E1 )
      I_Contact( #EstadoVI_M04.Etapas_Carga_E1 )
      Not()
      Coil( #EstadoVI.Etapas_Carga_E1 )
   END_RUNG
   RUNG wire#w1
      I_Contact( #EstadoVI_M01.Etapas_Descarga_S3 )
      I_Contact( #EstadoVI_M02.Etapas_Descarga_S3 )
      I_Contact( #EstadoVI_M03.Etapas_Descarga_S3 )
      I_Contact( #EstadoVI_M04.Etapas_Descarga_S3 )
      Not()
      Coil( #EstadoVI.Etapas_Descarga_S3 )
   END_RUNG
   RUNG wire#w1
      I_Contact( #EstadoVI_M01.Etapas_Descarga_S3 )
      I_Contact( #EstadoVI_M02.Etapas_Descarga_S3 )
      I_Contact( #EstadoVI_M03.Etapas_Descarga_S3 )
      I_Contact( #EstadoVI_M04.Etapas_Descarga_S3 )
      Not()
      Coil( #EstadoVI.Etapas_Descarga_S2 )
   END_RUNG
   RUNG wire#w1
      I_Contact( #EstadoVI_M01.Etapas_Descarga_S3 )
      I_Contact( #EstadoVI_M02.Etapas_Descarga_S3 )
      I_Contact( #EstadoVI_M03.Etapas_Descarga_S3 )
      I_Contact( #EstadoVI_M04.Etapas_Descarga_S3 )
      Not()
      Coil( #EstadoVI.Etapas_Descarga_S4 )
   END_RUNG
   // the same network as SCL:
   #EstadoVI.Etapas_Reset := "ON" AND #EstadoVI_M01.Etapas_Reset AND #EstadoVI_M02.Etapas_Reset AND #EstadoVI_M03.Etapas_Reset AND #EstadoVI_M04.Etapas_Reset;
   #EstadoVI.Etapa_Vacia := "ON" AND #EstadoVI_M01.Etapa_Vacia AND #EstadoVI_M02.Etapa_Vacia AND #EstadoVI_M03.Etapa_Vacia AND #EstadoVI_M04.Etapa_Vacia;
   #EstadoVI.Etapa_Cargada := NOT ("ON" AND NOT #EstadoVI_M01.Etapa_Cargada AND NOT #EstadoVI_M02.Etapa_Cargada AND NOT #EstadoVI_M03.Etapa_Cargada AND NOT #EstadoVI_M04.Etapa_Cargada);
   #EstadoVI.Etapas_Carga_E1 := NOT ("ON" AND NOT #EstadoVI_M01.Etapas_Carga_E1 AND NOT #EstadoVI_M02.Etapas_Carga_E1 AND NOT #EstadoVI_M03.Etapas_Carga_E1 AND NOT #EstadoVI_M04.Etapas_Carga_E1);
   #EstadoVI.Etapas_Descarga_S3 := NOT ("ON" AND NOT #EstadoVI_M01.Etapas_Descarga_S3 AND NOT #EstadoVI_M02.Etapas_Descarga_S3 AND NOT #EstadoVI_M03.Etapas_Descarga_S3 AND NOT #EstadoVI_M04.Etapas_Descarga_S3);
   #EstadoVI.Etapas_Descarga_S2 := NOT ("ON" AND NOT #EstadoVI_M01.Etapas_Descarga_S3 AND NOT #EstadoVI_M02.Etapas_Descarga_S3 AND NOT #EstadoVI_M03.Etapas_Descarga_S3 AND NOT #EstadoVI_M04.Etapas_Descarga_S3);
   #EstadoVI.Etapas_Descarga_S4 := NOT ("ON" AND NOT #EstadoVI_M01.Etapas_Descarga_S3 AND NOT #EstadoVI_M02.Etapas_Descarga_S3 AND NOT #EstadoVI_M03.Etapas_Descarga_S3 AND NOT #EstadoVI_M04.Etapas_Descarga_S3);
END_REGION

REGION Network 43: ENTRADAS DE LA MESA
   // Estados de las mesas
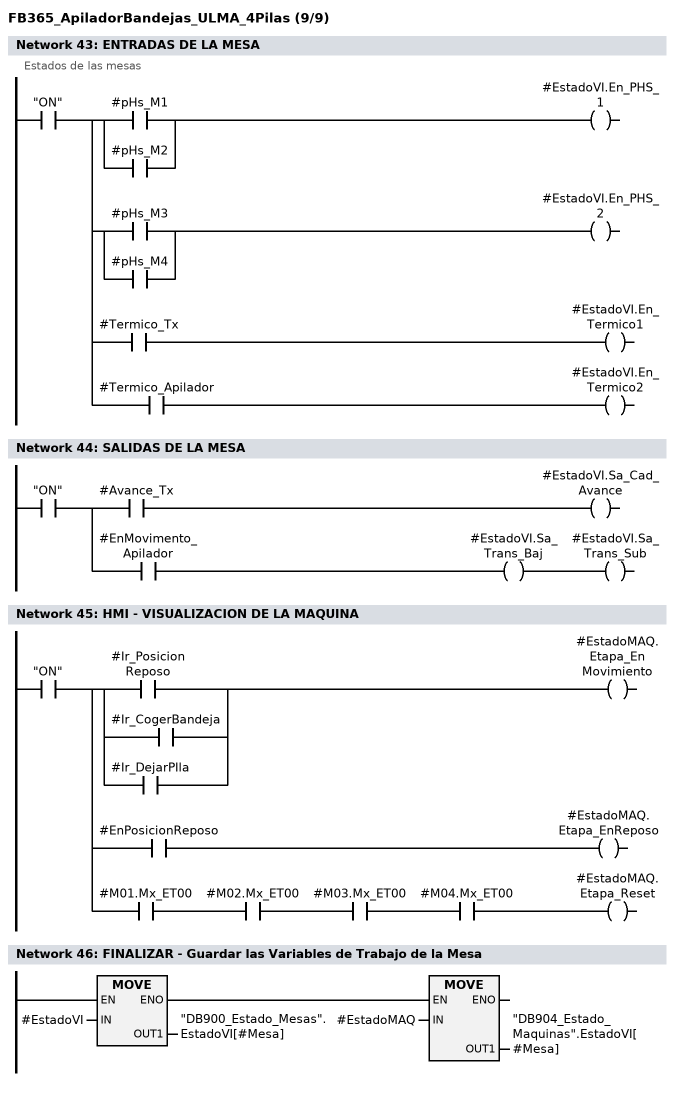
   RUNG wire#powerrail
      Contact( "ON" )
      wire#w1
      Contact( #pHs_M1 )
      wire#w2
      Coil( #EstadoVI.En_PHS_1 )
   END_RUNG
   RUNG wire#w1
      Contact( #pHs_M2 )
   END_RUNG wire#w2
   RUNG wire#w1
      Contact( #pHs_M3 )
      wire#w3
      Coil( #EstadoVI.En_PHS_2 )
   END_RUNG
   RUNG wire#w1
      Contact( #pHs_M4 )
   END_RUNG wire#w3
   RUNG wire#w1
      Contact( #Termico_Tx )
      Coil( #EstadoVI.En_Termico1 )
   END_RUNG
   RUNG wire#w1
      Contact( #Termico_Apilador )
      Coil( #EstadoVI.En_Termico2 )
   END_RUNG
   // the same network as SCL:
   #EstadoVI.En_PHS_1 := "ON" AND (#pHs_M1 OR #pHs_M2);
   #EstadoVI.En_PHS_2 := "ON" AND (#pHs_M3 OR #pHs_M4);
   #EstadoVI.En_Termico1 := "ON" AND #Termico_Tx;
   #EstadoVI.En_Termico2 := "ON" AND #Termico_Apilador;
END_REGION

REGION Network 44: SALIDAS DE LA MESA
   RUNG wire#powerrail
      Contact( "ON" )
      wire#w1
      Contact( #Avance_Tx )
      Coil( #EstadoVI.Sa_Cad_Avance )
   END_RUNG
   RUNG wire#w1
      Contact( #EnMovimento_Apilador )
      Coil( #EstadoVI.Sa_Trans_Baj )
      Coil( #EstadoVI.Sa_Trans_Sub )
   END_RUNG
   // the same network as SCL:
   #EstadoVI.Sa_Cad_Avance := "ON" AND #Avance_Tx;
   #EstadoVI.Sa_Trans_Baj := "ON" AND #EnMovimento_Apilador;
   #EstadoVI.Sa_Trans_Sub := #EstadoVI.Sa_Trans_Baj;
END_REGION

REGION Network 45: HMI - VISUALIZACION DE LA MAQUINA
   RUNG wire#powerrail
      Contact( "ON" )
      wire#w1
      Contact( #Ir_PosicionReposo )
      wire#w2
      Coil( #EstadoMAQ.Etapa_EnMovimiento )
   END_RUNG
   RUNG wire#w1
      Contact( #Ir_CogerBandeja )
   END_RUNG wire#w2
   RUNG wire#w1
      Contact( #Ir_DejarPIla )
   END_RUNG wire#w2
   RUNG wire#w1
      Contact( #EnPosicionReposo )
      Coil( #EstadoMAQ.Etapa_EnReposo )
   END_RUNG
   RUNG wire#w1
      Contact( #M01.Mx_ET00 )
      Contact( #M02.Mx_ET00 )
      Contact( #M03.Mx_ET00 )
      Contact( #M04.Mx_ET00 )
      Coil( #EstadoMAQ.Etapa_Reset )
   END_RUNG
   // the same network as SCL:
   #EstadoMAQ.Etapa_EnMovimiento := "ON" AND (#Ir_PosicionReposo OR #Ir_CogerBandeja OR #Ir_DejarPIla);
   #EstadoMAQ.Etapa_EnReposo := "ON" AND #EnPosicionReposo;
   #EstadoMAQ.Etapa_Reset := "ON" AND #M01.Mx_ET00 AND #M02.Mx_ET00 AND #M03.Mx_ET00 AND #M04.Mx_ET00;
END_REGION

REGION Network 46: FINALIZAR - Guardar las Variables de Trabajo de la Mesa
   RUNG wire#powerrail
      Move(in := #EstadoVI, out1 => "DB900_Estado_Mesas".EstadoVI[#Mesa])
      Move(in := #EstadoMAQ, out1 => "DB904_Estado_Maquinas".EstadoVI[#Mesa])
   END_RUNG
   // the same network as SCL:
   "DB900_Estado_Mesas".EstadoVI[#Mesa] := #EstadoVI;
   "DB904_Estado_Maquinas".EstadoVI[#Mesa] := #EstadoMAQ;
END_REGION
END_FUNCTION_BLOCK

FUNCTION_BLOCK "FB366_ApiladorBandejas_ULMA_2Pilas"   // FB366, LAD
{ S7_Optimized_Access := 'FALSE' }
AUTHOR : TLigero
NAME : 20160211
VERSION : 0.2
// stored: AutoNumber false, SetENOAutomatically false
   VAR_INPUT
      Mesa : UInt;   // Mesa de la FB
      EnTension : Bool;   // Existe Tension en la Mesa
      Error_Tx : Bool;   // Error en el Tx
      Selector : "Selector";   // Selector Unidades
      Selector_AD : Bool;   // Selector de Adelante
      Selector_AT : Bool;   // Selector de Atras
      Termico_Tx : Bool;   // Proteccion de Tx
      pHs_M1 : Bool;   // pHs de la P01 de la Mesa
      pHs_M2 : Bool;   // pHs de la P04 de la Mesa
      pHs_SalidaApilador : Bool;   // pHs de Control a Salida del Apilador
      pHs_VacioApìlador : Bool;   // phs de Apilador Vacio
      pHs_LlenoApilador : Bool;   // pHs de Apilador Lleno
      Avance_Tx : Bool;   // Avance de Tx
      Termico_Apilador : Bool;   // Proteccion de Elevacion del Apilador
      Apilador_UP : Bool;   // Apilador en Posicion Up
      Apilador_DW : Bool;   // Apilador en Posicion Down
      EnMovimento_Apilador : Bool;   // Apilador en Movimiento
      TPM1_Up : Bool;   // TP de la P01 Arriba
      TPM1_Down : Bool;   // TP de la P01 Abajo
      TPM2_Up : Bool;   // TP de la P04 Arriba
      TPM2_Down : Bool;   // TP de la P04 Abajo
      PRV_AVTF : Bool;   // E1 >> Aviso de Entrada
      NXT_Carga_OK : Bool;   // S3 >> Permiso de Salida
      NumBandejasPorPila : Int;   // Numero de Bandejas por Pila
      V_TOut_Atasco : Int;   // Valor de Time Out de Atasco
      V_TOut_Elevacion : Int;   // Valor de TIme Out de Elevacion
   END_VAR
   VAR_OUTPUT
      PRV_Carga_OK : Bool;   // E1 >> Permiso de Entrada
      NXT_AVTF : Bool;   // S3 >> Aviso de Salida
   END_VAR
   VAR
      M01 { S7_SetPoint := 'True'} : "FB364_Mesa_ApiladorBandejas_ULMA";
      M02 { S7_SetPoint := 'True'} : "FB364_Mesa_ApiladorBandejas_ULMA";
      EstadoVI_M01 { S7_SetPoint := 'True'} : "EstadosMesa";
      EstadoVI_M02 { S7_SetPoint := 'True'} : "EstadosMesa";
      TMP_EnTension { S7_SetPoint := 'True'} : "FB910_CNT_UHS";
      TOut_Elevacion { S7_SetPoint := 'True'} : "FB910_CNT_UHS";
      ContadorBandejasEnPila : Int;   // Contador De Bandejas por Pila
      Ord_Vaciado : Bool;   // Interna >> Apilador esta Lleno
      Ord_Apilar : Bool;   // Interna >> Apilar Bandeja
      Ir_PosicionReposo : Bool;   // Operacion >> Ir a Posicion Reposo
      Ir_CogerBandeja : Bool;   // Operacion >> Ir a Coger Bandeja (Apilar)
      Ir_DejarPIla : Bool;   // Operacion >> Ir a Dejar Pila (Vaciado)
      EnPosicionReposo : Bool;   // Esta En Posicion de Reposo
      CogidaBandeja : Bool;   // Cogida Bandeja
      DejadaPila : Bool;   // Dejada la Pila
      MFP_ApiladorVaciado : Bool;   // Memoria FP de Apilador Vaciado
      MFP_ContadorBandejas : Bool;   // Memoria FP de Inc. de Bandeja en Pila
      MA_Avance_Tx : Bool;
      MA_Retroceder_Tx : Bool;
      MA_Subir : Bool;
      MA_Bajar : Bool;
      MA_Subir_TPM1 : Bool;
      MA_Bajar_TPM1 : Bool;
      MA_Subir_TPM2 : Bool;
      MA_Bajar_TPM2 : Bool;
   END_VAR
   VAR_TEMP
      EstadoZona : "EstadoZona";   // Estado de Zona de la Mesa
      EstadoVI : "EstadosMesa";   // Estado del Vehiculo Inteliguente de la Mesa
      EstadoMAQ : "EstadoMaquina";   // Estado del Vehiculo Inteliguente de la Maquina
      Aux_ET00 : Bool;
   END_VAR
   VAR_TEMP   // added for the SCL form of the ladder/FBD networks
      _w1 : Bool;
      _w2 : Bool;
   END_VAR
BEGIN

REGION Network 1: INICIALIZAR - Recoger las Variables de Estado de la Mesa
   // Se recoge - Estado_CBx
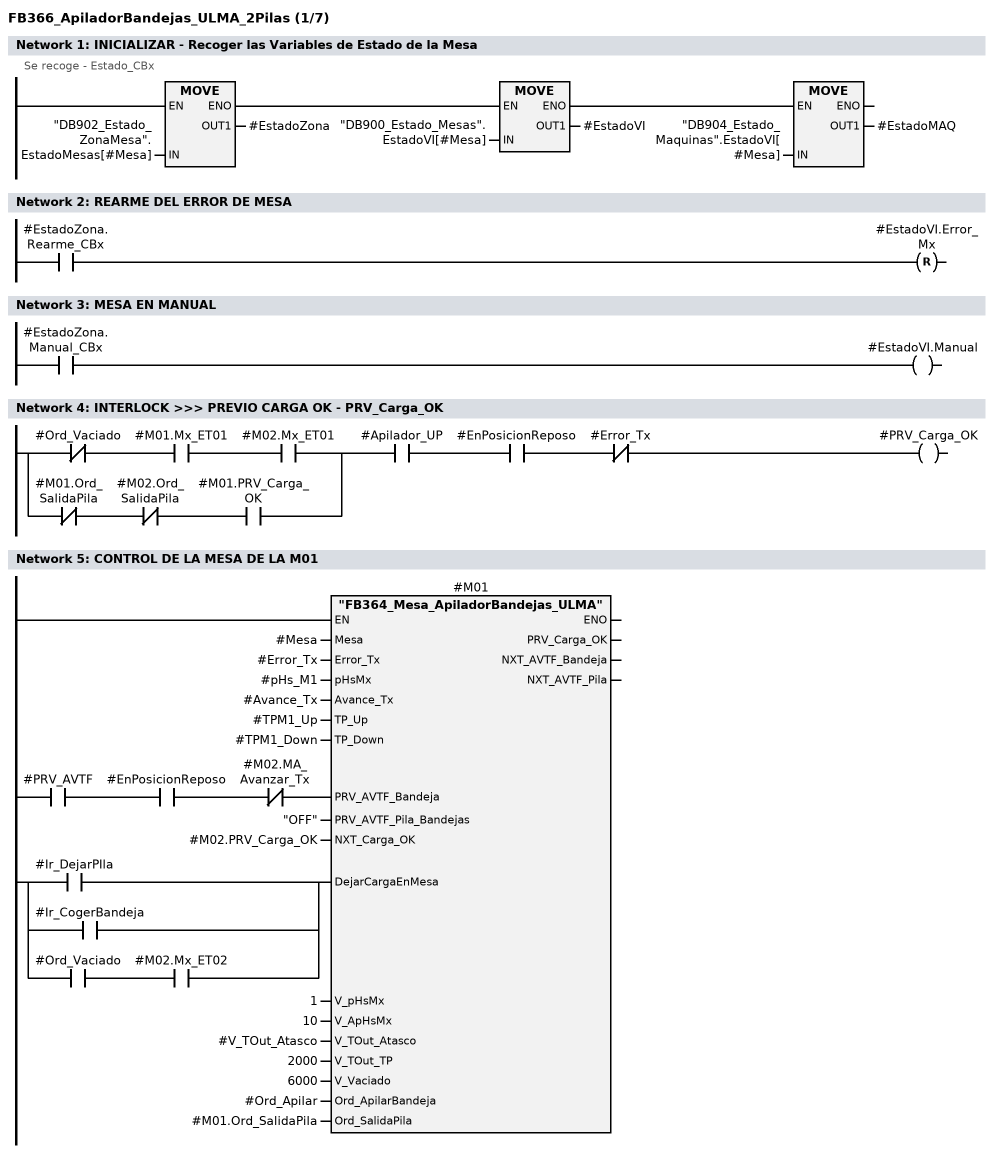
   RUNG wire#powerrail
      Move(in := "DB902_Estado_ZonaMesa".EstadoMesas[#Mesa], out1 => #EstadoZona)
      Move(in := "DB900_Estado_Mesas".EstadoVI[#Mesa], out1 => #EstadoVI)
      Move(in := "DB904_Estado_Maquinas".EstadoVI[#Mesa], out1 => #EstadoMAQ)
   END_RUNG
   // the same network as SCL:
   #EstadoZona := "DB902_Estado_ZonaMesa".EstadoMesas[#Mesa];
   #EstadoVI := "DB900_Estado_Mesas".EstadoVI[#Mesa];
   #EstadoMAQ := "DB904_Estado_Maquinas".EstadoVI[#Mesa];
END_REGION

REGION Network 2: REARME DEL ERROR DE MESA
   RUNG wire#powerrail
      Contact( #EstadoZona.Rearme_CBx )
      R_Coil( #EstadoVI.Error_Mx )
   END_RUNG
   // the same network as SCL:
   IF #EstadoZona.Rearme_CBx THEN #EstadoVI.Error_Mx := FALSE; END_IF;
END_REGION

REGION Network 3: MESA EN MANUAL
   RUNG wire#powerrail
      Contact( #EstadoZona.Manual_CBx )
      Coil( #EstadoVI.Manual )
   END_RUNG
   // the same network as SCL:
   #EstadoVI.Manual := #EstadoZona.Manual_CBx;
END_REGION

REGION Network 4: INTERLOCK >>> PREVIO CARGA OK - PRV_Carga_OK
   RUNG wire#powerrail
      I_Contact( #Ord_Vaciado )
      Contact( #M01.Mx_ET01 )
      Contact( #M02.Mx_ET01 )
      wire#w1
      Contact( #Apilador_UP )
      Contact( #EnPosicionReposo )
      I_Contact( #Error_Tx )
      Coil( #PRV_Carga_OK )
   END_RUNG
   RUNG wire#powerrail
      I_Contact( #M01.Ord_SalidaPila )
      I_Contact( #M02.Ord_SalidaPila )
      Contact( #M01.PRV_Carga_OK )
   END_RUNG wire#w1
   // the same network as SCL:
   #PRV_Carga_OK := ((NOT #Ord_Vaciado AND #M01.Mx_ET01 AND #M02.Mx_ET01) OR (NOT #M01.Ord_SalidaPila AND NOT #M02.Ord_SalidaPila AND #M01.PRV_Carga_OK)) AND #Apilador_UP AND #EnPosicionReposo AND NOT #Error_Tx;
END_REGION

REGION Network 5: CONTROL DE LA MESA DE LA M01
   RUNG wire#powerrail
      #M01(PRV_AVTF_Bandeja := wire#w1, DejarCargaEnMesa := wire#w2, Mesa := #Mesa, Error_Tx := #Error_Tx, pHsMx := #pHs_M1, Avance_Tx := #Avance_Tx, TP_Up := #TPM1_Up, TP_Down := #TPM1_Down, PRV_AVTF_Pila_Bandejas := "OFF", NXT_Carga_OK := #M02.PRV_Carga_OK, V_pHsMx := 1, V_ApHsMx := 10, V_TOut_Atasco := #V_TOut_Atasco, V_TOut_TP := 2000, V_Vaciado := 6000, Ord_ApilarBandeja := #Ord_Apilar, Ord_SalidaPila := #M01.Ord_SalidaPila, PRV_Carga_OK =>, NXT_AVTF_Bandeja =>, NXT_AVTF_Pila =>)
   END_RUNG
   RUNG wire#powerrail
      Contact( #PRV_AVTF )
      Contact( #EnPosicionReposo )
      I_Contact( #M02.MA_Avanzar_Tx )
   END_RUNG wire#w1
   RUNG wire#powerrail
      Contact( #Ir_DejarPIla )
   END_RUNG wire#w2
   RUNG wire#powerrail
      Contact( #Ir_CogerBandeja )
   END_RUNG wire#w2
   RUNG wire#powerrail
      Contact( #Ord_Vaciado )
      Contact( #M02.Mx_ET02 )
   END_RUNG wire#w2
   // the same network as SCL:
   #M01(Mesa := #Mesa,   // "FB364_Mesa_ApiladorBandejas_ULMA"
        Error_Tx := #Error_Tx,
        pHsMx := #pHs_M1,
        Avance_Tx := #Avance_Tx,
        TP_Up := #TPM1_Up,
        TP_Down := #TPM1_Down,
        PRV_AVTF_Bandeja := #PRV_AVTF AND #EnPosicionReposo AND NOT #M02.MA_Avanzar_Tx,
        PRV_AVTF_Pila_Bandejas := "OFF",
        NXT_Carga_OK := #M02.PRV_Carga_OK,
        DejarCargaEnMesa := #Ir_DejarPIla OR #Ir_CogerBandeja OR (#Ord_Vaciado AND #M02.Mx_ET02),
        V_pHsMx := 1,
        V_ApHsMx := 10,
        V_TOut_Atasco := #V_TOut_Atasco,
        V_TOut_TP := 2000,
        V_Vaciado := 6000,
        Ord_ApilarBandeja := #Ord_Apilar,
        Ord_SalidaPila := #M01.Ord_SalidaPila);
END_REGION

REGION Network 6: CONTROL DE LA MESA DE LA M02
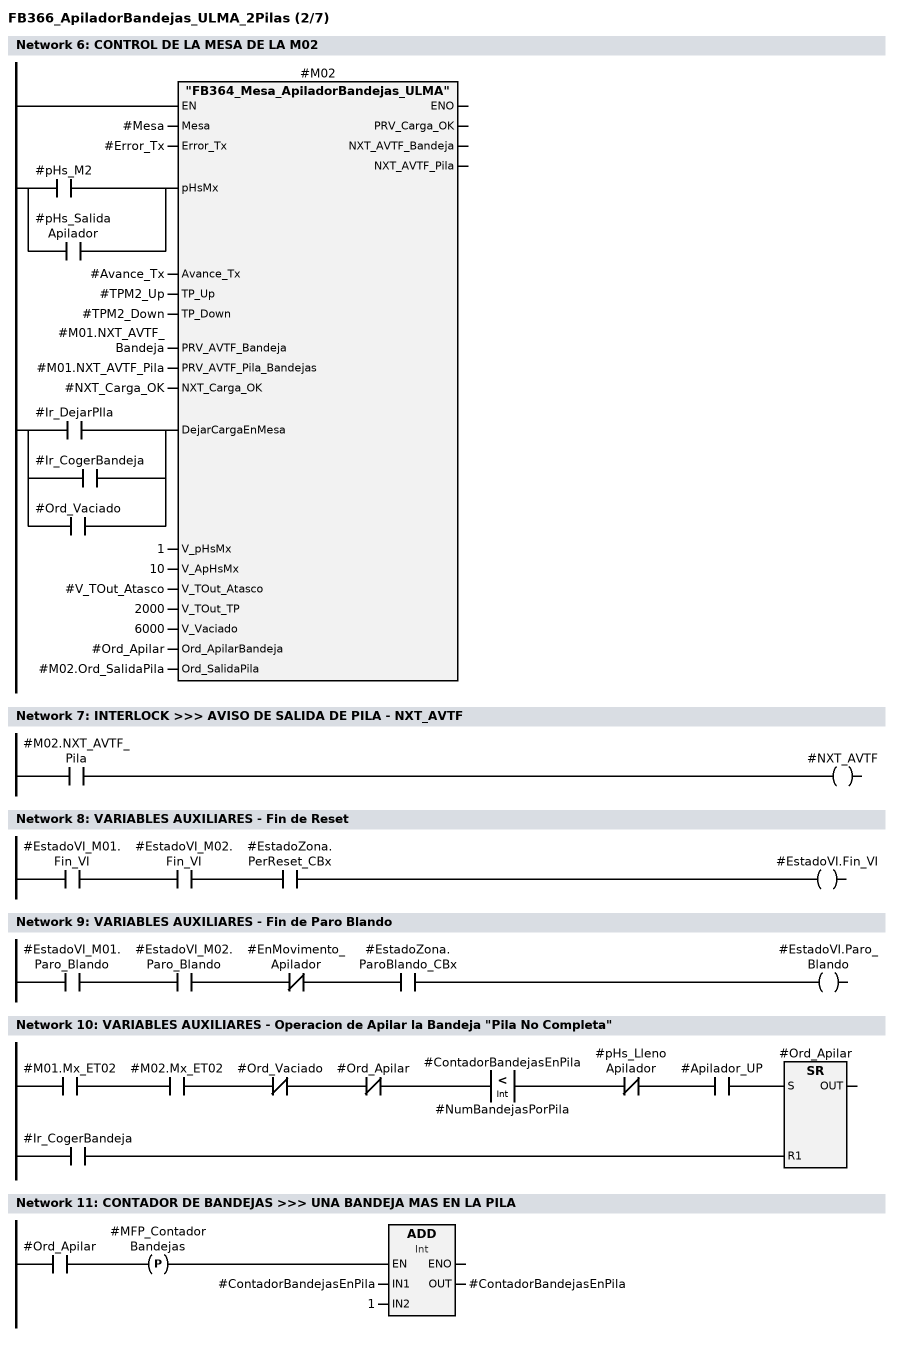
   RUNG wire#powerrail
      #M02(pHsMx := wire#w1, DejarCargaEnMesa := wire#w2, Mesa := #Mesa, Error_Tx := #Error_Tx, Avance_Tx := #Avance_Tx, TP_Up := #TPM2_Up, TP_Down := #TPM2_Down, PRV_AVTF_Bandeja := #M01.NXT_AVTF_Bandeja, PRV_AVTF_Pila_Bandejas := #M01.NXT_AVTF_Pila, NXT_Carga_OK := #NXT_Carga_OK, V_pHsMx := 1, V_ApHsMx := 10, V_TOut_Atasco := #V_TOut_Atasco, V_TOut_TP := 2000, V_Vaciado := 6000, Ord_ApilarBandeja := #Ord_Apilar, Ord_SalidaPila := #M02.Ord_SalidaPila, PRV_Carga_OK =>, NXT_AVTF_Bandeja =>, NXT_AVTF_Pila =>)
   END_RUNG
   RUNG wire#powerrail
      Contact( #pHs_M2 )
   END_RUNG wire#w1
   RUNG wire#powerrail
      Contact( #pHs_SalidaApilador )
   END_RUNG wire#w1
   RUNG wire#powerrail
      Contact( #Ir_DejarPIla )
   END_RUNG wire#w2
   RUNG wire#powerrail
      Contact( #Ir_CogerBandeja )
   END_RUNG wire#w2
   RUNG wire#powerrail
      Contact( #Ord_Vaciado )
   END_RUNG wire#w2
   // the same network as SCL:
   #M02(Mesa := #Mesa,   // "FB364_Mesa_ApiladorBandejas_ULMA"
        Error_Tx := #Error_Tx,
        pHsMx := #pHs_M2 OR #pHs_SalidaApilador,
        Avance_Tx := #Avance_Tx,
        TP_Up := #TPM2_Up,
        TP_Down := #TPM2_Down,
        PRV_AVTF_Bandeja := #M01.NXT_AVTF_Bandeja,
        PRV_AVTF_Pila_Bandejas := #M01.NXT_AVTF_Pila,
        NXT_Carga_OK := #NXT_Carga_OK,
        DejarCargaEnMesa := #Ir_DejarPIla OR #Ir_CogerBandeja OR #Ord_Vaciado,
        V_pHsMx := 1,
        V_ApHsMx := 10,
        V_TOut_Atasco := #V_TOut_Atasco,
        V_TOut_TP := 2000,
        V_Vaciado := 6000,
        Ord_ApilarBandeja := #Ord_Apilar,
        Ord_SalidaPila := #M02.Ord_SalidaPila);
END_REGION

REGION Network 7: INTERLOCK >>> AVISO DE SALIDA DE PILA - NXT_AVTF
   RUNG wire#powerrail
      Contact( #M02.NXT_AVTF_Pila )
      Coil( #NXT_AVTF )
   END_RUNG
   // the same network as SCL:
   #NXT_AVTF := #M02.NXT_AVTF_Pila;
END_REGION

REGION Network 8: VARIABLES AUXILIARES - Fin de Reset
   RUNG wire#powerrail
      Contact( #EstadoVI_M01.Fin_VI )
      Contact( #EstadoVI_M02.Fin_VI )
      Contact( #EstadoZona.PerReset_CBx )
      Coil( #EstadoVI.Fin_VI )
   END_RUNG
   // the same network as SCL:
   #EstadoVI.Fin_VI := #EstadoVI_M01.Fin_VI AND #EstadoVI_M02.Fin_VI AND #EstadoZona.PerReset_CBx;
END_REGION

REGION Network 9: VARIABLES AUXILIARES - Fin de Paro Blando
   RUNG wire#powerrail
      Contact( #EstadoVI_M01.Paro_Blando )
      Contact( #EstadoVI_M02.Paro_Blando )
      I_Contact( #EnMovimento_Apilador )
      Contact( #EstadoZona.ParoBlando_CBx )
      Coil( #EstadoVI.Paro_Blando )
   END_RUNG
   // the same network as SCL:
   #EstadoVI.Paro_Blando := #EstadoVI_M01.Paro_Blando AND #EstadoVI_M02.Paro_Blando AND NOT #EnMovimento_Apilador AND #EstadoZona.ParoBlando_CBx;
END_REGION

REGION Network 10: VARIABLES AUXILIARES - Operacion de Apilar la Bandeja "Pila No Completa"
   RUNG wire#powerrail
      Contact( #M01.Mx_ET02 )
      Contact( #M02.Mx_ET02 )
      I_Contact( #Ord_Vaciado )
      I_Contact( #Ord_Apilar )
      { S7_Templates := "SrcType := Int" } LT_Contact(in1 := #ContadorBandejasEnPila, in2 := #NumBandejasPorPila)
      I_Contact( #pHs_LlenoApilador )
      Contact( #Apilador_UP )
      S_SR(operand := #Ord_Apilar, r1 := wire#w1)
   END_RUNG
   RUNG wire#powerrail
      Contact( #Ir_CogerBandeja )
   END_RUNG wire#w1
   // the same network as SCL:
   IF #M01.Mx_ET02 AND #M02.Mx_ET02 AND NOT #Ord_Vaciado AND NOT #Ord_Apilar AND (#ContadorBandejasEnPila < #NumBandejasPorPila) AND NOT #pHs_LlenoApilador AND #Apilador_UP THEN
       #Ord_Apilar := TRUE;   // SR flip-flop
   END_IF;
   IF #Ir_CogerBandeja THEN #Ord_Apilar := FALSE; END_IF;
END_REGION

REGION Network 11: CONTADOR DE BANDEJAS >>> UNA BANDEJA MAS EN LA PILA
   RUNG wire#powerrail
      Contact( #Ord_Apilar )
      P_Trig( #MFP_ContadorBandejas )
      { S7_Templates := "SrcType := Int"; S7_GenerateENO := "TRUE" } Add(in1 := #ContadorBandejasEnPila, in2 := 1, out => #ContadorBandejasEnPila)
   END_RUNG
   // the same network as SCL:
   #_w1 := #Ord_Apilar AND NOT #MFP_ContadorBandejas;   // rising edge
   #MFP_ContadorBandejas := #Ord_Apilar;
   IF #_w1 THEN #ContadorBandejasEnPila := #ContadorBandejasEnPila + 1; END_IF;
END_REGION

REGION Network 12: CONTADOR DE BANDEJAS >>> RESET DE BANDEJAS EN LA PILA
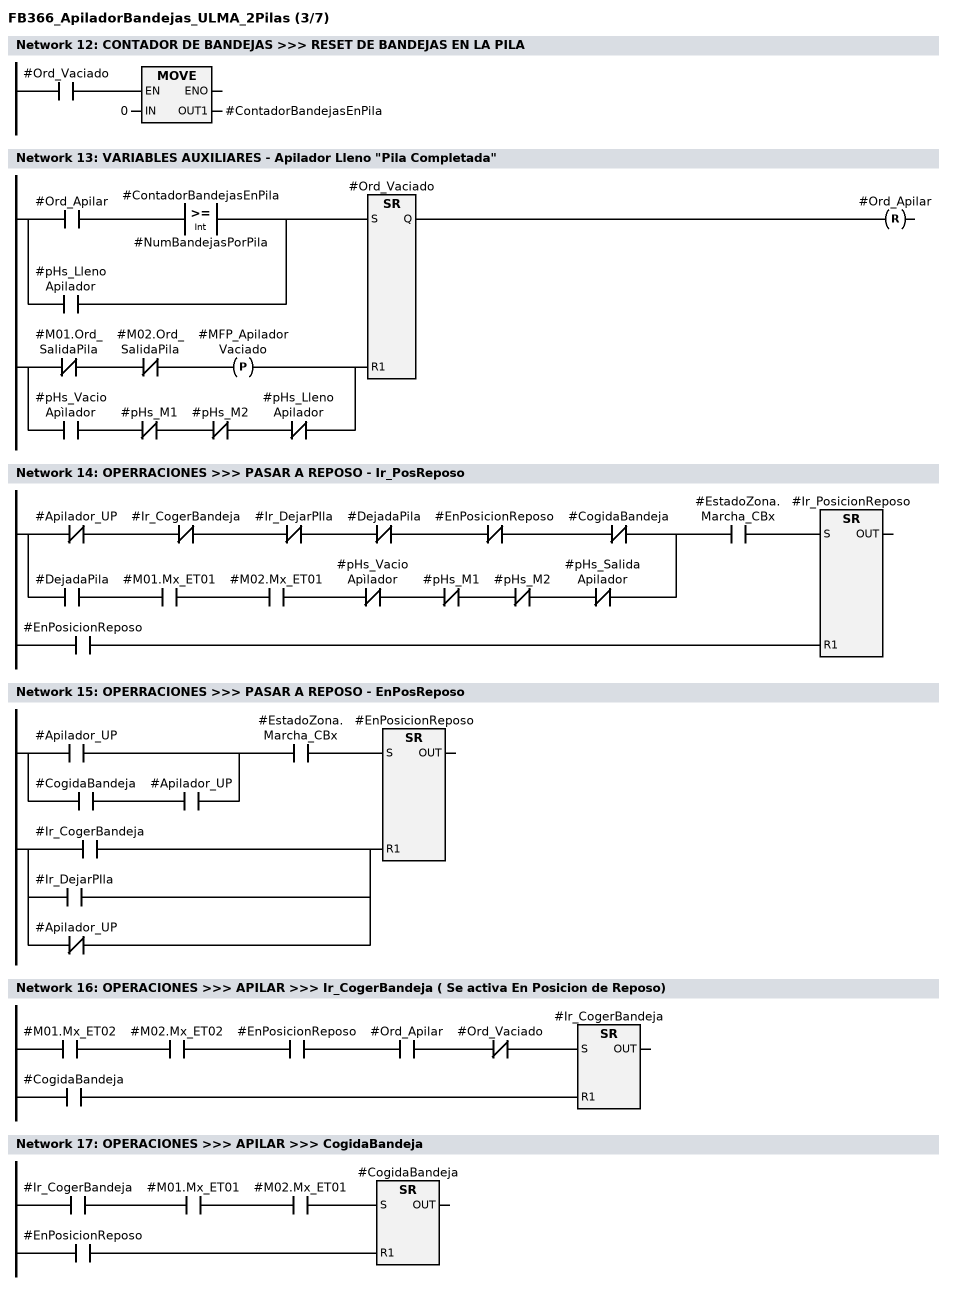
   RUNG wire#powerrail
      Contact( #Ord_Vaciado )
      { S7_GenerateENO := "TRUE" } Move(in := 0, out1 => #ContadorBandejasEnPila)
   END_RUNG
   // the same network as SCL:
   IF #Ord_Vaciado THEN #ContadorBandejasEnPila := 0; END_IF;
END_REGION

REGION Network 13: VARIABLES AUXILIARES - Apilador Lleno "Pila Completada"
   RUNG wire#powerrail
      Contact( #Ord_Apilar )
      { S7_Templates := "SrcType := Int" } GE_Contact(in1 := #ContadorBandejasEnPila, in2 := #NumBandejasPorPila)
      wire#w1
      S_SR(operand := #Ord_Vaciado, r1 := wire#w2)
      R_Coil( #Ord_Apilar )
   END_RUNG
   RUNG wire#powerrail
      Contact( #pHs_LlenoApilador )
   END_RUNG wire#w1
   RUNG wire#powerrail
      I_Contact( #M01.Ord_SalidaPila )
      I_Contact( #M02.Ord_SalidaPila )
      P_Trig( #MFP_ApiladorVaciado )
   END_RUNG wire#w2
   RUNG wire#powerrail
      Contact( #pHs_VacioApìlador )
      I_Contact( #pHs_M1 )
      I_Contact( #pHs_M2 )
      I_Contact( #pHs_LlenoApilador )
   END_RUNG wire#w2
   // the same network as SCL:
   #_w1 := NOT #M01.Ord_SalidaPila AND NOT #M02.Ord_SalidaPila;
   #_w2 := #_w1 AND NOT #MFP_ApiladorVaciado;   // rising edge
   #MFP_ApiladorVaciado := #_w1;
   IF (#Ord_Apilar AND (#ContadorBandejasEnPila >= #NumBandejasPorPila)) OR #pHs_LlenoApilador THEN
       #Ord_Vaciado := TRUE;   // SR flip-flop
   END_IF;
   IF #_w2 OR (#pHs_VacioApìlador AND NOT #pHs_M1 AND NOT #pHs_M2 AND NOT #pHs_LlenoApilador) THEN
       #Ord_Vaciado := FALSE;
   END_IF;
   IF #Ord_Vaciado THEN #Ord_Apilar := FALSE; END_IF;
END_REGION

REGION Network 14: OPERRACIONES >>> PASAR A REPOSO - Ir_PosReposo
   RUNG wire#powerrail
      I_Contact( #Apilador_UP )
      I_Contact( #Ir_CogerBandeja )
      I_Contact( #Ir_DejarPIla )
      I_Contact( #DejadaPila )
      I_Contact( #EnPosicionReposo )
      I_Contact( #CogidaBandeja )
      wire#w1
      Contact( #EstadoZona.Marcha_CBx )
      S_SR(operand := #Ir_PosicionReposo, r1 := wire#w2)
   END_RUNG
   RUNG wire#powerrail
      Contact( #DejadaPila )
      Contact( #M01.Mx_ET01 )
      Contact( #M02.Mx_ET01 )
      I_Contact( #pHs_VacioApìlador )
      I_Contact( #pHs_M1 )
      I_Contact( #pHs_M2 )
      I_Contact( #pHs_SalidaApilador )
   END_RUNG wire#w1
   RUNG wire#powerrail
      Contact( #EnPosicionReposo )
   END_RUNG wire#w2
   // the same network as SCL:
   IF ((NOT #Apilador_UP AND NOT #Ir_CogerBandeja AND NOT #Ir_DejarPIla AND NOT #DejadaPila AND NOT #EnPosicionReposo AND NOT #CogidaBandeja) OR (#DejadaPila AND #M01.Mx_ET01 AND #M02.Mx_ET01 AND NOT #pHs_VacioApìlador AND NOT #pHs_M1 AND NOT #pHs_M2 AND NOT #pHs_SalidaApilador)) AND #EstadoZona.Marcha_CBx THEN
       #Ir_PosicionReposo := TRUE;   // SR flip-flop
   END_IF;
   IF #EnPosicionReposo THEN #Ir_PosicionReposo := FALSE; END_IF;
END_REGION

REGION Network 15: OPERRACIONES >>> PASAR A REPOSO - EnPosReposo
   RUNG wire#powerrail
      Contact( #Apilador_UP )
      wire#w1
      Contact( #EstadoZona.Marcha_CBx )
      S_SR(operand := #EnPosicionReposo, r1 := wire#w2)
   END_RUNG
   RUNG wire#powerrail
      Contact( #CogidaBandeja )
      Contact( #Apilador_UP )
   END_RUNG wire#w1
   RUNG wire#powerrail
      Contact( #Ir_CogerBandeja )
   END_RUNG wire#w2
   RUNG wire#powerrail
      Contact( #Ir_DejarPIla )
   END_RUNG wire#w2
   RUNG wire#powerrail
      I_Contact( #Apilador_UP )
   END_RUNG wire#w2
   // the same network as SCL:
   IF (#Apilador_UP OR (#CogidaBandeja AND #Apilador_UP)) AND #EstadoZona.Marcha_CBx THEN
       #EnPosicionReposo := TRUE;   // SR flip-flop
   END_IF;
   IF #Ir_CogerBandeja OR #Ir_DejarPIla OR NOT #Apilador_UP THEN #EnPosicionReposo := FALSE; END_IF;
END_REGION

REGION Network 16: OPERACIONES >>> APILAR >>> Ir_CogerBandeja ( Se activa En Posicion de Reposo)
   RUNG wire#powerrail
      Contact( #M01.Mx_ET02 )
      Contact( #M02.Mx_ET02 )
      Contact( #EnPosicionReposo )
      Contact( #Ord_Apilar )
      I_Contact( #Ord_Vaciado )
      S_SR(operand := #Ir_CogerBandeja, r1 := wire#w1)
   END_RUNG
   RUNG wire#powerrail
      Contact( #CogidaBandeja )
   END_RUNG wire#w1
   // the same network as SCL:
   IF #M01.Mx_ET02 AND #M02.Mx_ET02 AND #EnPosicionReposo AND #Ord_Apilar AND NOT #Ord_Vaciado THEN
       #Ir_CogerBandeja := TRUE;   // SR flip-flop
   END_IF;
   IF #CogidaBandeja THEN #Ir_CogerBandeja := FALSE; END_IF;
END_REGION

REGION Network 17: OPERACIONES >>> APILAR >>> CogidaBandeja
   RUNG wire#powerrail
      Contact( #Ir_CogerBandeja )
      Contact( #M01.Mx_ET01 )
      Contact( #M02.Mx_ET01 )
      S_SR(operand := #CogidaBandeja, r1 := wire#w1)
   END_RUNG
   RUNG wire#powerrail
      Contact( #EnPosicionReposo )
   END_RUNG wire#w1
   // the same network as SCL:
   IF #Ir_CogerBandeja AND #M01.Mx_ET01 AND #M02.Mx_ET01 THEN
       #CogidaBandeja := TRUE;   // SR flip-flop
   END_IF;
   IF #EnPosicionReposo THEN #CogidaBandeja := FALSE; END_IF;
END_REGION

REGION Network 18: OPERACIONES >>> VACIAR PILAS >>> Ir_DejarPila ( Se activa En Posicion de Reposo)
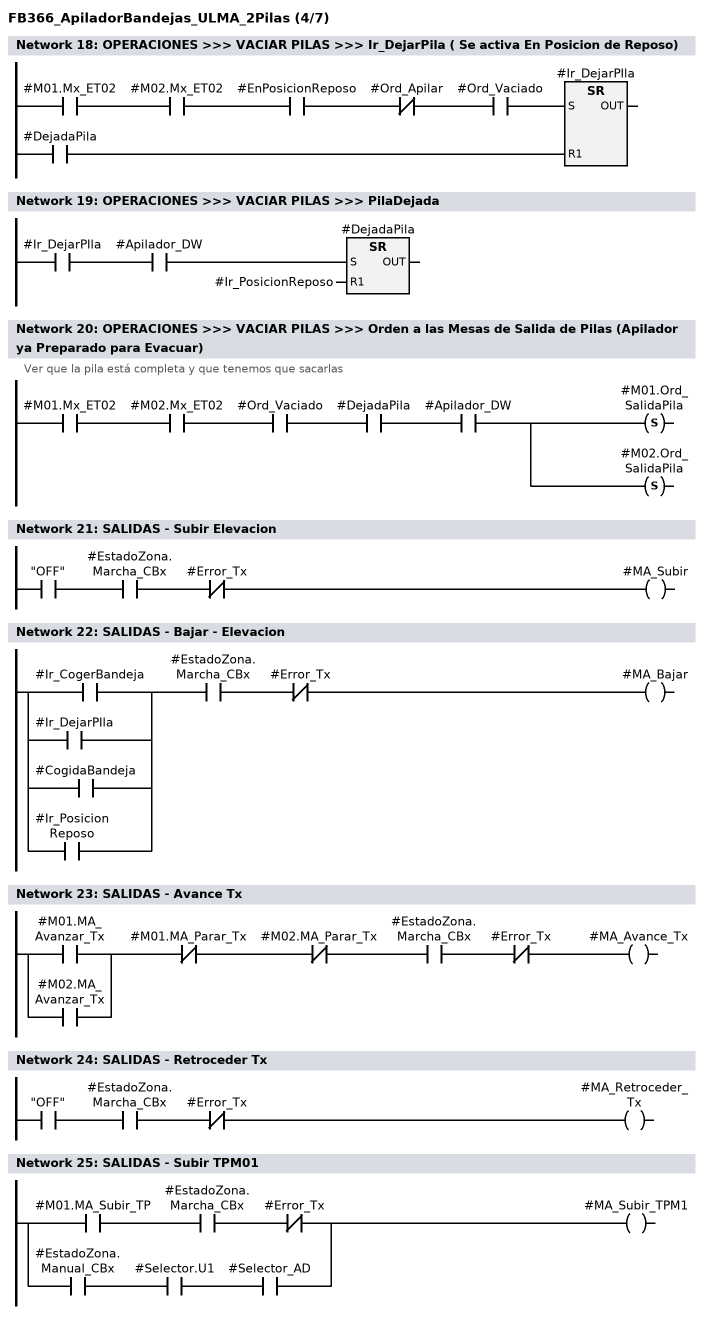
   RUNG wire#powerrail
      Contact( #M01.Mx_ET02 )
      Contact( #M02.Mx_ET02 )
      Contact( #EnPosicionReposo )
      I_Contact( #Ord_Apilar )
      Contact( #Ord_Vaciado )
      S_SR(operand := #Ir_DejarPIla, r1 := wire#w1)
   END_RUNG
   RUNG wire#powerrail
      Contact( #DejadaPila )
   END_RUNG wire#w1
   // the same network as SCL:
   IF #M01.Mx_ET02 AND #M02.Mx_ET02 AND #EnPosicionReposo AND NOT #Ord_Apilar AND #Ord_Vaciado THEN
       #Ir_DejarPIla := TRUE;   // SR flip-flop
   END_IF;
   IF #DejadaPila THEN #Ir_DejarPIla := FALSE; END_IF;
END_REGION

REGION Network 19: OPERACIONES >>> VACIAR PILAS >>> PilaDejada
   RUNG wire#powerrail
      Contact( #Ir_DejarPIla )
      Contact( #Apilador_DW )
      S_SR(operand := #DejadaPila, r1 := #Ir_PosicionReposo)
   END_RUNG
   // the same network as SCL:
   IF #Ir_DejarPIla AND #Apilador_DW THEN
       #DejadaPila := TRUE;   // SR flip-flop
   END_IF;
   IF #Ir_PosicionReposo THEN #DejadaPila := FALSE; END_IF;
END_REGION

REGION Network 20: OPERACIONES >>> VACIAR PILAS >>> Orden a las Mesas de Salida de Pilas (Apilador ya Preparado para Evacuar)
   // Ver que la pila está completa y que tenemos que sacarlas
   RUNG wire#powerrail
      Contact( #M01.Mx_ET02 )
      Contact( #M02.Mx_ET02 )
      Contact( #Ord_Vaciado )
      Contact( #DejadaPila )
      Contact( #Apilador_DW )
      wire#w1
      S_Coil( #M01.Ord_SalidaPila )
   END_RUNG
   RUNG wire#w1
      S_Coil( #M02.Ord_SalidaPila )
   END_RUNG
   // the same network as SCL:
   IF #M01.Mx_ET02 AND #M02.Mx_ET02 AND #Ord_Vaciado AND #DejadaPila AND #Apilador_DW THEN
       #M01.Ord_SalidaPila := TRUE;
       #M02.Ord_SalidaPila := TRUE;
   END_IF;
END_REGION

REGION Network 21: SALIDAS - Subir Elevacion
   RUNG wire#powerrail
      Contact( "OFF" )
      Contact( #EstadoZona.Marcha_CBx )
      I_Contact( #Error_Tx )
      Coil( #MA_Subir )
   END_RUNG
   // the same network as SCL:
   #MA_Subir := "OFF" AND #EstadoZona.Marcha_CBx AND NOT #Error_Tx;
END_REGION

REGION Network 22: SALIDAS - Bajar - Elevacion
   RUNG wire#powerrail
      Contact( #Ir_CogerBandeja )
      wire#w1
      Contact( #EstadoZona.Marcha_CBx )
      I_Contact( #Error_Tx )
      Coil( #MA_Bajar )
   END_RUNG
   RUNG wire#powerrail
      Contact( #Ir_DejarPIla )
   END_RUNG wire#w1
   RUNG wire#powerrail
      Contact( #CogidaBandeja )
   END_RUNG wire#w1
   RUNG wire#powerrail
      Contact( #Ir_PosicionReposo )
   END_RUNG wire#w1
   // the same network as SCL:
   #MA_Bajar := (#Ir_CogerBandeja OR #Ir_DejarPIla OR #CogidaBandeja OR #Ir_PosicionReposo) AND #EstadoZona.Marcha_CBx AND NOT #Error_Tx;
END_REGION

REGION Network 23: SALIDAS - Avance Tx
   RUNG wire#powerrail
      Contact( #M01.MA_Avanzar_Tx )
      wire#w1
      I_Contact( #M01.MA_Parar_Tx )
      I_Contact( #M02.MA_Parar_Tx )
      Contact( #EstadoZona.Marcha_CBx )
      I_Contact( #Error_Tx )
      Coil( #MA_Avance_Tx )
   END_RUNG
   RUNG wire#powerrail
      Contact( #M02.MA_Avanzar_Tx )
   END_RUNG wire#w1
   // the same network as SCL:
   #MA_Avance_Tx := (#M01.MA_Avanzar_Tx OR #M02.MA_Avanzar_Tx) AND NOT #M01.MA_Parar_Tx AND NOT #M02.MA_Parar_Tx AND #EstadoZona.Marcha_CBx AND NOT #Error_Tx;
END_REGION

REGION Network 24: SALIDAS - Retroceder Tx
   RUNG wire#powerrail
      Contact( "OFF" )
      Contact( #EstadoZona.Marcha_CBx )
      I_Contact( #Error_Tx )
      Coil( #MA_Retroceder_Tx )
   END_RUNG
   // the same network as SCL:
   #MA_Retroceder_Tx := "OFF" AND #EstadoZona.Marcha_CBx AND NOT #Error_Tx;
END_REGION

REGION Network 25: SALIDAS - Subir TPM01
   RUNG wire#powerrail
      Contact( #M01.MA_Subir_TP )
      Contact( #EstadoZona.Marcha_CBx )
      I_Contact( #Error_Tx )
      wire#w1
      Coil( #MA_Subir_TPM1 )
   END_RUNG
   RUNG wire#powerrail
      Contact( #EstadoZona.Manual_CBx )
      Contact( #Selector.U1 )
      Contact( #Selector_AD )
   END_RUNG wire#w1
   // the same network as SCL:
   #MA_Subir_TPM1 := (#M01.MA_Subir_TP AND #EstadoZona.Marcha_CBx AND NOT #Error_Tx) OR (#EstadoZona.Manual_CBx AND #Selector.U1 AND #Selector_AD);
END_REGION

REGION Network 26: SALIDAS - Bajar TPM01
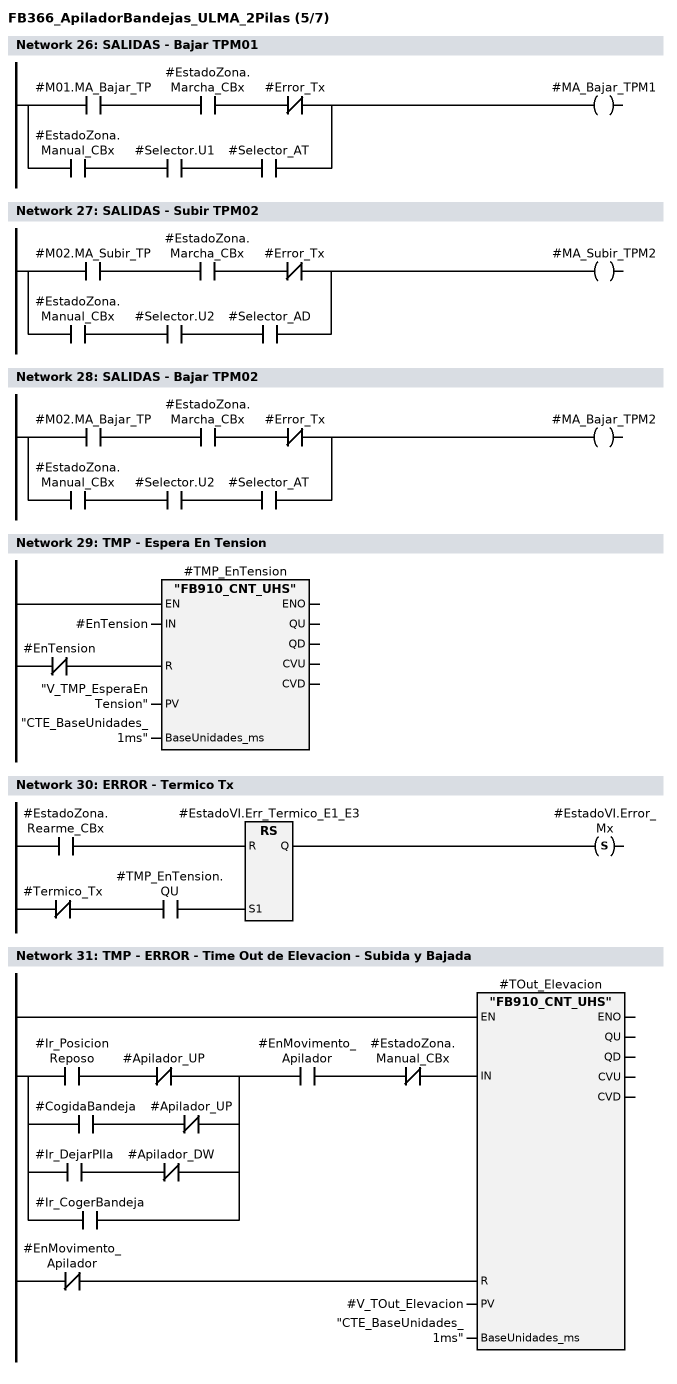
   RUNG wire#powerrail
      Contact( #M01.MA_Bajar_TP )
      Contact( #EstadoZona.Marcha_CBx )
      I_Contact( #Error_Tx )
      wire#w1
      Coil( #MA_Bajar_TPM1 )
   END_RUNG
   RUNG wire#powerrail
      Contact( #EstadoZona.Manual_CBx )
      Contact( #Selector.U1 )
      Contact( #Selector_AT )
   END_RUNG wire#w1
   // the same network as SCL:
   #MA_Bajar_TPM1 := (#M01.MA_Bajar_TP AND #EstadoZona.Marcha_CBx AND NOT #Error_Tx) OR (#EstadoZona.Manual_CBx AND #Selector.U1 AND #Selector_AT);
END_REGION

REGION Network 27: SALIDAS - Subir TPM02
   RUNG wire#powerrail
      Contact( #M02.MA_Subir_TP )
      Contact( #EstadoZona.Marcha_CBx )
      I_Contact( #Error_Tx )
      wire#w1
      Coil( #MA_Subir_TPM2 )
   END_RUNG
   RUNG wire#powerrail
      Contact( #EstadoZona.Manual_CBx )
      Contact( #Selector.U2 )
      Contact( #Selector_AD )
   END_RUNG wire#w1
   // the same network as SCL:
   #MA_Subir_TPM2 := (#M02.MA_Subir_TP AND #EstadoZona.Marcha_CBx AND NOT #Error_Tx) OR (#EstadoZona.Manual_CBx AND #Selector.U2 AND #Selector_AD);
END_REGION

REGION Network 28: SALIDAS - Bajar TPM02
   RUNG wire#powerrail
      Contact( #M02.MA_Bajar_TP )
      Contact( #EstadoZona.Marcha_CBx )
      I_Contact( #Error_Tx )
      wire#w1
      Coil( #MA_Bajar_TPM2 )
   END_RUNG
   RUNG wire#powerrail
      Contact( #EstadoZona.Manual_CBx )
      Contact( #Selector.U2 )
      Contact( #Selector_AT )
   END_RUNG wire#w1
   // the same network as SCL:
   #MA_Bajar_TPM2 := (#M02.MA_Bajar_TP AND #EstadoZona.Marcha_CBx AND NOT #Error_Tx) OR (#EstadoZona.Manual_CBx AND #Selector.U2 AND #Selector_AT);
END_REGION

REGION Network 29: TMP - Espera En Tension
   RUNG wire#powerrail
      #TMP_EnTension(R := wire#w1, IN := #EnTension, PV := "V_TMP_EsperaEnTension", BaseUnidades_ms := "CTE_BaseUnidades_1ms", QU =>, QD =>, CVU =>, CVD =>)
   END_RUNG
   RUNG wire#powerrail
      I_Contact( #EnTension )
   END_RUNG wire#w1
   // the same network as SCL:
   #TMP_EnTension(IN := #EnTension,   // "FB910_CNT_UHS"
                  R := NOT #EnTension,
                  PV := "V_TMP_EsperaEnTension",
                  BaseUnidades_ms := "CTE_BaseUnidades_1ms");
END_REGION

REGION Network 30: ERROR - Termico Tx
   RUNG wire#powerrail
      Contact( #EstadoZona.Rearme_CBx )
      S_RS(operand := #EstadoVI.Err_Termico_E1_E3, s1 := wire#w1)
      S_Coil( #EstadoVI.Error_Mx )
   END_RUNG
   RUNG wire#powerrail
      I_Contact( #Termico_Tx )
      Contact( #TMP_EnTension.QU )
   END_RUNG wire#w1
   // the same network as SCL:
   IF #EstadoZona.Rearme_CBx THEN
       #EstadoVI.Err_Termico_E1_E3 := FALSE;   // RS flip-flop
   END_IF;
   IF NOT #Termico_Tx AND #TMP_EnTension.QU THEN #EstadoVI.Err_Termico_E1_E3 := TRUE; END_IF;
   IF #EstadoVI.Err_Termico_E1_E3 THEN #EstadoVI.Error_Mx := TRUE; END_IF;
END_REGION

REGION Network 31: TMP - ERROR - Time Out de Elevacion - Subida y Bajada
   RUNG wire#powerrail
      #TOut_Elevacion(IN := wire#w2, R := wire#w3, PV := #V_TOut_Elevacion, BaseUnidades_ms := "CTE_BaseUnidades_1ms", QU =>, QD =>, CVU =>, CVD =>)
   END_RUNG
   RUNG wire#powerrail
      Contact( #Ir_PosicionReposo )
      I_Contact( #Apilador_UP )
      wire#w1
      Contact( #EnMovimento_Apilador )
      I_Contact( #EstadoZona.Manual_CBx )
   END_RUNG wire#w2
   RUNG wire#powerrail
      Contact( #CogidaBandeja )
      I_Contact( #Apilador_UP )
   END_RUNG wire#w1
   RUNG wire#powerrail
      Contact( #Ir_DejarPIla )
      I_Contact( #Apilador_DW )
   END_RUNG wire#w1
   RUNG wire#powerrail
      Contact( #Ir_CogerBandeja )
   END_RUNG wire#w1
   RUNG wire#powerrail
      I_Contact( #EnMovimento_Apilador )
   END_RUNG wire#w3
   // the same network as SCL:
   #TOut_Elevacion(IN := ((#Ir_PosicionReposo AND NOT #Apilador_UP) OR (#CogidaBandeja AND NOT #Apilador_UP) OR (#Ir_DejarPIla AND NOT #Apilador_DW) OR #Ir_CogerBandeja) AND #EnMovimento_Apilador AND NOT #EstadoZona.Manual_CBx,   // "FB910_CNT_UHS"
                   R := NOT #EnMovimento_Apilador,
                   PV := #V_TOut_Elevacion,
                   BaseUnidades_ms := "CTE_BaseUnidades_1ms");
END_REGION

REGION Network 32: ERROR - Time Out de Elevacion - Subida y Bajada
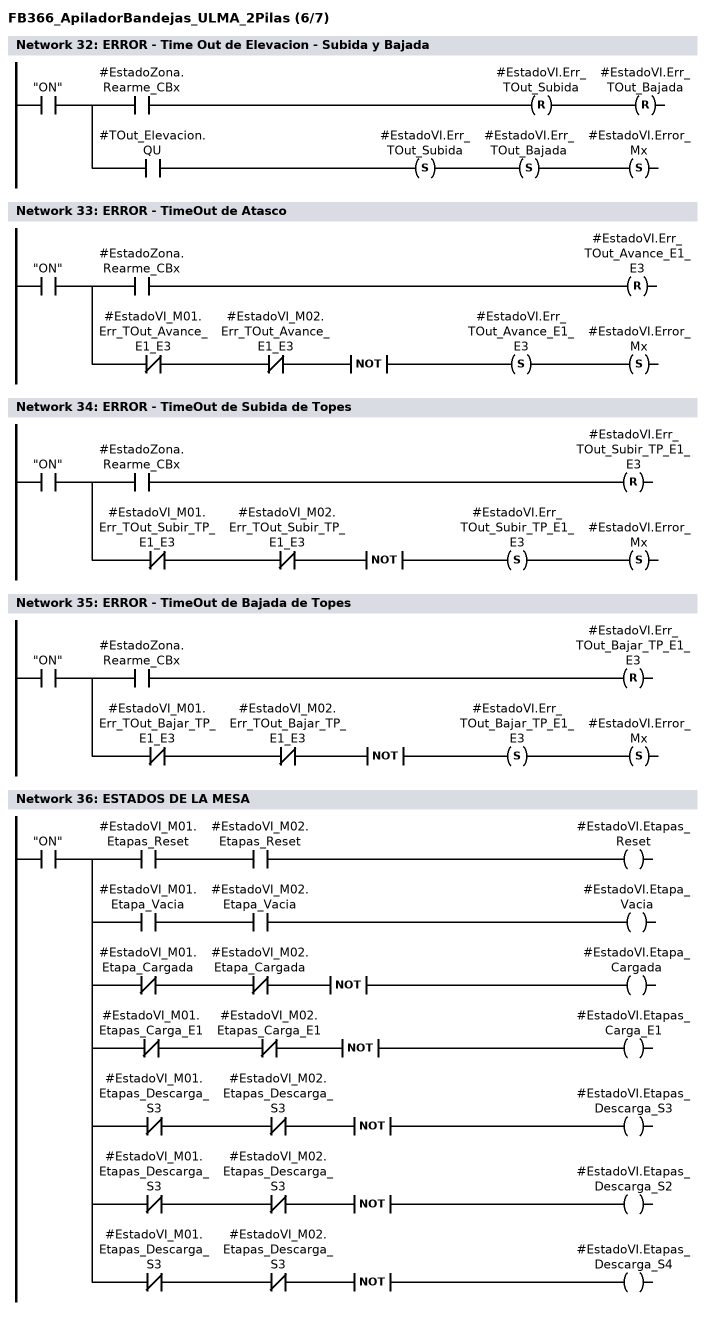
   RUNG wire#powerrail
      Contact( "ON" )
      wire#w1
      Contact( #EstadoZona.Rearme_CBx )
      R_Coil( #EstadoVI.Err_TOut_Subida )
      R_Coil( #EstadoVI.Err_TOut_Bajada )
   END_RUNG
   RUNG wire#w1
      Contact( #TOut_Elevacion.QU )
      S_Coil( #EstadoVI.Err_TOut_Subida )
      S_Coil( #EstadoVI.Err_TOut_Bajada )
      S_Coil( #EstadoVI.Error_Mx )
   END_RUNG
   // the same network as SCL:
   IF "ON" AND #EstadoZona.Rearme_CBx THEN
       #EstadoVI.Err_TOut_Subida := FALSE;
       #EstadoVI.Err_TOut_Bajada := FALSE;
   END_IF;
   IF "ON" AND #TOut_Elevacion.QU THEN
       #EstadoVI.Err_TOut_Subida := TRUE;
       #EstadoVI.Err_TOut_Bajada := TRUE;
       #EstadoVI.Error_Mx := TRUE;
   END_IF;
END_REGION

REGION Network 33: ERROR - TimeOut de Atasco
   RUNG wire#powerrail
      Contact( "ON" )
      wire#w1
      Contact( #EstadoZona.Rearme_CBx )
      R_Coil( #EstadoVI.Err_TOut_Avance_E1_E3 )
   END_RUNG
   RUNG wire#w1
      I_Contact( #EstadoVI_M01.Err_TOut_Avance_E1_E3 )
      I_Contact( #EstadoVI_M02.Err_TOut_Avance_E1_E3 )
      Not()
      S_Coil( #EstadoVI.Err_TOut_Avance_E1_E3 )
      S_Coil( #EstadoVI.Error_Mx )
   END_RUNG
   // the same network as SCL:
   IF "ON" AND #EstadoZona.Rearme_CBx THEN #EstadoVI.Err_TOut_Avance_E1_E3 := FALSE; END_IF;
   IF NOT ("ON" AND NOT #EstadoVI_M01.Err_TOut_Avance_E1_E3 AND NOT #EstadoVI_M02.Err_TOut_Avance_E1_E3) THEN
       #EstadoVI.Err_TOut_Avance_E1_E3 := TRUE;
       #EstadoVI.Error_Mx := TRUE;
   END_IF;
END_REGION

REGION Network 34: ERROR - TimeOut de Subida de Topes
   RUNG wire#powerrail
      Contact( "ON" )
      wire#w1
      Contact( #EstadoZona.Rearme_CBx )
      R_Coil( #EstadoVI.Err_TOut_Subir_TP_E1_E3 )
   END_RUNG
   RUNG wire#w1
      I_Contact( #EstadoVI_M01.Err_TOut_Subir_TP_E1_E3 )
      I_Contact( #EstadoVI_M02.Err_TOut_Subir_TP_E1_E3 )
      Not()
      S_Coil( #EstadoVI.Err_TOut_Subir_TP_E1_E3 )
      S_Coil( #EstadoVI.Error_Mx )
   END_RUNG
   // the same network as SCL:
   IF "ON" AND #EstadoZona.Rearme_CBx THEN #EstadoVI.Err_TOut_Subir_TP_E1_E3 := FALSE; END_IF;
   IF NOT ("ON" AND NOT #EstadoVI_M01.Err_TOut_Subir_TP_E1_E3 AND NOT #EstadoVI_M02.Err_TOut_Subir_TP_E1_E3) THEN
       #EstadoVI.Err_TOut_Subir_TP_E1_E3 := TRUE;
       #EstadoVI.Error_Mx := TRUE;
   END_IF;
END_REGION

REGION Network 35: ERROR - TimeOut de Bajada de Topes
   RUNG wire#powerrail
      Contact( "ON" )
      wire#w1
      Contact( #EstadoZona.Rearme_CBx )
      R_Coil( #EstadoVI.Err_TOut_Bajar_TP_E1_E3 )
   END_RUNG
   RUNG wire#w1
      I_Contact( #EstadoVI_M01.Err_TOut_Bajar_TP_E1_E3 )
      I_Contact( #EstadoVI_M02.Err_TOut_Bajar_TP_E1_E3 )
      Not()
      S_Coil( #EstadoVI.Err_TOut_Bajar_TP_E1_E3 )
      S_Coil( #EstadoVI.Error_Mx )
   END_RUNG
   // the same network as SCL:
   IF "ON" AND #EstadoZona.Rearme_CBx THEN #EstadoVI.Err_TOut_Bajar_TP_E1_E3 := FALSE; END_IF;
   IF NOT ("ON" AND NOT #EstadoVI_M01.Err_TOut_Bajar_TP_E1_E3 AND NOT #EstadoVI_M02.Err_TOut_Bajar_TP_E1_E3) THEN
       #EstadoVI.Err_TOut_Bajar_TP_E1_E3 := TRUE;
       #EstadoVI.Error_Mx := TRUE;
   END_IF;
END_REGION

REGION Network 36: ESTADOS DE LA MESA
   RUNG wire#powerrail
      Contact( "ON" )
      wire#w1
      Contact( #EstadoVI_M01.Etapas_Reset )
      Contact( #EstadoVI_M02.Etapas_Reset )
      Coil( #EstadoVI.Etapas_Reset )
   END_RUNG
   RUNG wire#w1
      Contact( #EstadoVI_M01.Etapa_Vacia )
      Contact( #EstadoVI_M02.Etapa_Vacia )
      Coil( #EstadoVI.Etapa_Vacia )
   END_RUNG
   RUNG wire#w1
      I_Contact( #EstadoVI_M01.Etapa_Cargada )
      I_Contact( #EstadoVI_M02.Etapa_Cargada )
      Not()
      Coil( #EstadoVI.Etapa_Cargada )
   END_RUNG
   RUNG wire#w1
      I_Contact( #EstadoVI_M01.Etapas_Carga_E1 )
      I_Contact( #EstadoVI_M02.Etapas_Carga_E1 )
      Not()
      Coil( #EstadoVI.Etapas_Carga_E1 )
   END_RUNG
   RUNG wire#w1
      I_Contact( #EstadoVI_M01.Etapas_Descarga_S3 )
      I_Contact( #EstadoVI_M02.Etapas_Descarga_S3 )
      Not()
      Coil( #EstadoVI.Etapas_Descarga_S3 )
   END_RUNG
   RUNG wire#w1
      I_Contact( #EstadoVI_M01.Etapas_Descarga_S3 )
      I_Contact( #EstadoVI_M02.Etapas_Descarga_S3 )
      Not()
      Coil( #EstadoVI.Etapas_Descarga_S2 )
   END_RUNG
   RUNG wire#w1
      I_Contact( #EstadoVI_M01.Etapas_Descarga_S3 )
      I_Contact( #EstadoVI_M02.Etapas_Descarga_S3 )
      Not()
      Coil( #EstadoVI.Etapas_Descarga_S4 )
   END_RUNG
   // the same network as SCL:
   #EstadoVI.Etapas_Reset := "ON" AND #EstadoVI_M01.Etapas_Reset AND #EstadoVI_M02.Etapas_Reset;
   #EstadoVI.Etapa_Vacia := "ON" AND #EstadoVI_M01.Etapa_Vacia AND #EstadoVI_M02.Etapa_Vacia;
   #EstadoVI.Etapa_Cargada := NOT ("ON" AND NOT #EstadoVI_M01.Etapa_Cargada AND NOT #EstadoVI_M02.Etapa_Cargada);
   #EstadoVI.Etapas_Carga_E1 := NOT ("ON" AND NOT #EstadoVI_M01.Etapas_Carga_E1 AND NOT #EstadoVI_M02.Etapas_Carga_E1);
   #EstadoVI.Etapas_Descarga_S3 := NOT ("ON" AND NOT #EstadoVI_M01.Etapas_Descarga_S3 AND NOT #EstadoVI_M02.Etapas_Descarga_S3);
   #EstadoVI.Etapas_Descarga_S2 := NOT ("ON" AND NOT #EstadoVI_M01.Etapas_Descarga_S3 AND NOT #EstadoVI_M02.Etapas_Descarga_S3);
   #EstadoVI.Etapas_Descarga_S4 := NOT ("ON" AND NOT #EstadoVI_M01.Etapas_Descarga_S3 AND NOT #EstadoVI_M02.Etapas_Descarga_S3);
END_REGION

REGION Network 37: ENTRADAS DE LA MESA
   // Estados de las mesas
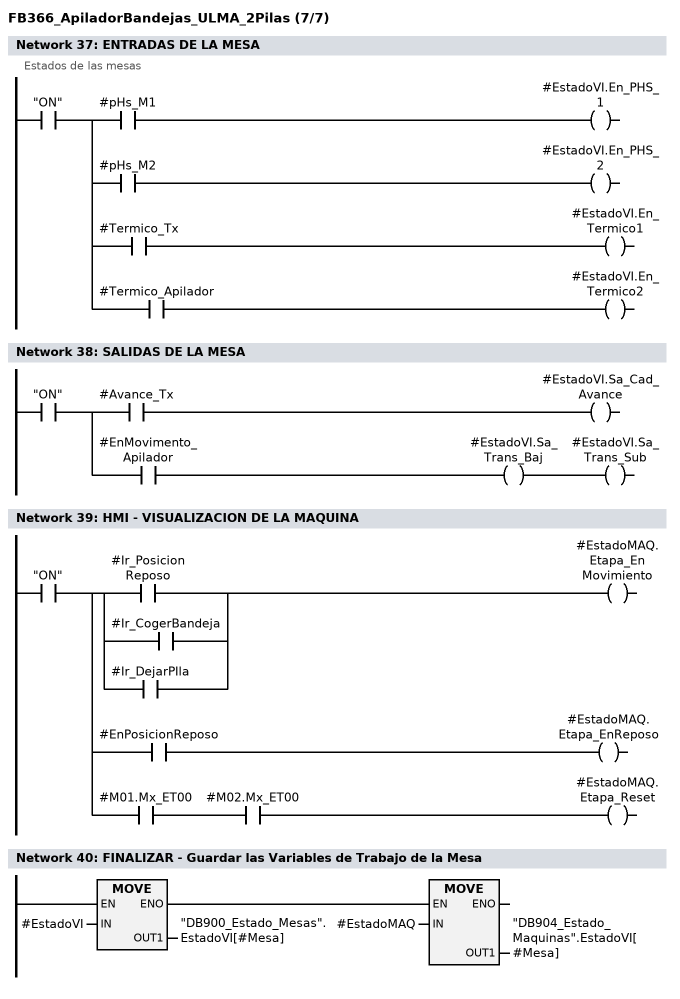
   RUNG wire#powerrail
      Contact( "ON" )
      wire#w1
      Contact( #pHs_M1 )
      Coil( #EstadoVI.En_PHS_1 )
   END_RUNG
   RUNG wire#w1
      Contact( #pHs_M2 )
      Coil( #EstadoVI.En_PHS_2 )
   END_RUNG
   RUNG wire#w1
      Contact( #Termico_Tx )
      Coil( #EstadoVI.En_Termico1 )
   END_RUNG
   RUNG wire#w1
      Contact( #Termico_Apilador )
      Coil( #EstadoVI.En_Termico2 )
   END_RUNG
   // the same network as SCL:
   #EstadoVI.En_PHS_1 := "ON" AND #pHs_M1;
   #EstadoVI.En_PHS_2 := "ON" AND #pHs_M2;
   #EstadoVI.En_Termico1 := "ON" AND #Termico_Tx;
   #EstadoVI.En_Termico2 := "ON" AND #Termico_Apilador;
END_REGION

REGION Network 38: SALIDAS DE LA MESA
   RUNG wire#powerrail
      Contact( "ON" )
      wire#w1
      Contact( #Avance_Tx )
      Coil( #EstadoVI.Sa_Cad_Avance )
   END_RUNG
   RUNG wire#w1
      Contact( #EnMovimento_Apilador )
      Coil( #EstadoVI.Sa_Trans_Baj )
      Coil( #EstadoVI.Sa_Trans_Sub )
   END_RUNG
   // the same network as SCL:
   #EstadoVI.Sa_Cad_Avance := "ON" AND #Avance_Tx;
   #EstadoVI.Sa_Trans_Baj := "ON" AND #EnMovimento_Apilador;
   #EstadoVI.Sa_Trans_Sub := #EstadoVI.Sa_Trans_Baj;
END_REGION

REGION Network 39: HMI - VISUALIZACION DE LA MAQUINA
   RUNG wire#powerrail
      Contact( "ON" )
      wire#w1
      Contact( #Ir_PosicionReposo )
      wire#w2
      Coil( #EstadoMAQ.Etapa_EnMovimiento )
   END_RUNG
   RUNG wire#w1
      Contact( #Ir_CogerBandeja )
   END_RUNG wire#w2
   RUNG wire#w1
      Contact( #Ir_DejarPIla )
   END_RUNG wire#w2
   RUNG wire#w1
      Contact( #EnPosicionReposo )
      Coil( #EstadoMAQ.Etapa_EnReposo )
   END_RUNG
   RUNG wire#w1
      Contact( #M01.Mx_ET00 )
      Contact( #M02.Mx_ET00 )
      Coil( #EstadoMAQ.Etapa_Reset )
   END_RUNG
   // the same network as SCL:
   #EstadoMAQ.Etapa_EnMovimiento := "ON" AND (#Ir_PosicionReposo OR #Ir_CogerBandeja OR #Ir_DejarPIla);
   #EstadoMAQ.Etapa_EnReposo := "ON" AND #EnPosicionReposo;
   #EstadoMAQ.Etapa_Reset := "ON" AND #M01.Mx_ET00 AND #M02.Mx_ET00;
END_REGION

REGION Network 40: FINALIZAR - Guardar las Variables de Trabajo de la Mesa
   RUNG wire#powerrail
      Move(in := #EstadoVI, out1 => "DB900_Estado_Mesas".EstadoVI[#Mesa])
      Move(in := #EstadoMAQ, out1 => "DB904_Estado_Maquinas".EstadoVI[#Mesa])
   END_RUNG
   // the same network as SCL:
   "DB900_Estado_Mesas".EstadoVI[#Mesa] := #EstadoVI;
   "DB904_Estado_Maquinas".EstadoVI[#Mesa] := #EstadoMAQ;
END_REGION
END_FUNCTION_BLOCK

FUNCTION_BLOCK "FB376_DesPaletizador_Manual"   // FB376, LAD
TITLE = DesPaletizador Manual (Capas)
{ S7_Optimized_Access := 'FALSE' }
// stored: AutoNumber false, SetENOAutomatically false
   VAR_INPUT
      Maquina : UInt;   // Numero de Maquina
      ConfigDesPaletizador : "UDT_ConfigDesPaletizador";   // DB de Config de Velocidadad
      Robot_Habilitado : Bool;   // ROBOT >> Habilitado
      Robot_OutElevador : Bool;   // ROBOT >> Fuera de la Zona del Elevador
      Robot_PeticionSubir : Bool;   // ROBOT >> Peticion de Subir
      Robot_PeticionBajar : Bool;   // ROBOT >> Peticion de Bajar
      Robot_VelocidadElevador : Int;   // ROBOT >> Velocidad del Elevador
      ByteInicial : Int;   // Byte Inicial del Variador LENZE
      NodoNoPresente : Bool;   // Nodo No Presenye del Variador LENZE
      EnTension : Bool;   // Existe Tension en la Mesa
      Mantenimiento : Bool;   // Llave de Mantenimiento
      TermicoFreno : Bool;   // Termico del Freno
      Seg_UP : Bool;   // Seguridad Abajo de la Elevacion
      Seg_DOWN : Bool;   // Seguridad Abajo de la Elevacion
      pHsPisoCarga : Bool;   // Posicion del Piso de Carga
      pHsPisoDesCarga : Bool;   // Posicion del Piso de DesCarga
      Protrusion : Bool;   // pHs de Protrusion
      P_NuevaCapa : Bool;   // Peticion de Nueva Capa
      P_Subir : Bool;   // Pulsador de Subir
      P_Bajar : Bool;   // Pulsador de Bajar
      BarreraUp : Bool;   // Barrera del Nivel Superior
      pHsAnchura_01 : Bool;
      pHsAnchura_02 : Bool;
      pHsGalibo_01 : Bool;   // pHs de Control de Hueco Superior
      pHsGalibo_02 : Bool;   // pHs de Control de Hueco Superior
      pHsGalibo_03 : Bool;   // pHs de Control de Hueco Superior
      pHsGalibo_04 : Bool;   // pHs de Control de Hueco Superior
      pHsAlturaCota_01 : Bool;
      pHsAlturaCota_02 : Bool;
      pHsAlturaMax_01 : Bool;
      pHsAlturaMax_02 : Bool;
      RoturaCadena_01 : Bool;   // Rotura de Cadena
      RoturaCadena_02 : Bool;   // Rotura de Cadena
      RoturaCadena_03 : Bool;   // Rotura de Cadena
      RoturaCadena_04 : Bool;   // Rotura de Cadena
      FinDesPaletizado : Bool;   // Fin del Paletizado
      SubirManual : Bool;   // Subir en Manual
      BajarManual : Bool;   // Bajar en Manual
      Homming : Bool;
      EncoderIncremental : Bool;
      pHsReferenciaCero : Bool;   // phs de Referencia Cero
      V_TIM_Galibo : Time := T#1S;   // Morgan 14/02/19 500ms ->1s
      V_TIM_Protrusion : Int := 200;
      V_TOut_Elevacion : Int := 15000;
   END_VAR
   VAR_OUTPUT
      DesHabilitarBarreraUp : Bool;   // DesHabilitar Barrerra superior
      H_Puesto : Bool;   // Baliza de Paleta en Puesto
      DI3VarElev_pHsReferenciaCero : Bool;
   END_VAR
   VAR
      PosicionActual : Int;   // Posicion Actual
      PosicionDOWN : Int;   // Interna >> Posicion Abajo
      PosicionUP : Int;   // Interna >> Posicion Arriba
      PosicionOrden : Int;   // Orden >> Posicion A Ejecutar
      PosicionUltima : Int;   // Orden >> Ultima Posicion Enviada
      MemoPosicionActual : Int;   // Memoria >> Altura de la Carga
      MemoEventoDesPaletizado : Int;   // Memoria >> Evento Paletizado
      ConsignaFR : Int;   // Variador >> Consigna
      EstadoElevador : Word;   // Variador >> Estado
      Subject_Area : Word;   // Variador >> Subjet Area
      ID_Area : Word;   // Variador >> ID Area
      Orden : Bool;   // Orden >> Ejecutar
      FinOrden : Bool;   // Orden >> Fin Ejecucion
      PaletaEnPuesto : Bool;   // Interna >> Paleta En el Puesto
      MAQx_SinCapa : Bool;
      MemoCapaDinamico : Bool;
      FP_CapaDinamico : Bool;
      FN_CapaDinamico : Bool;
      InicioCapa : Int;
      FinalCapa : Int;
      MAQx_SinCota : Bool;
      MemoCotaDinamico : Bool;
      FP_CotaDinamico : Bool;
      MA_SubirPuesto : Bool;   // PUESTO >> Subir la Carga
      MA_BajarPuesto : Bool;   // PUESTO >> Bajar la Carga
      MA_Baliza : Bool;   // PUESTO >> Baliza
      PermisoMovElevador : Bool;   // Permiso Mover el Elevador
      PosCarga_OK : Bool;   // Posicionado en Carga
      PosDesCarga_OK : Bool;   // Posicionado en DesCargaCarga
      VarElev_MemoHomingAuto : Bool;   // Variador >>
      VarElev_ReferenciaOK : Bool;   // Variador >>
      VarElev_Error : Bool;   // Variador >>
      EventoInicioDesPaletizado : Bool;   // Evento >> Inicio DesPaletizado
      EventoFinalDesPaletizado : Bool;   // Evento >> Final DesPaletizado
      TIM_EsperaOrden { S7_SetPoint := 'True'} : TON_TIME;   // Orden >> TIM de Espera para Ejecutar
      TMPEnPisoCarga { S7_SetPoint := 'True'} : TON_TIME;
      TMPEnPisoDesCarga { S7_SetPoint := 'True'} : TON_TIME;
      TMP_EnTension { S7_SetPoint := 'True'} : "FB910_CNT_UHS";
      TOut_Elevacion { S7_SetPoint := 'True'} : "FB910_CNT_UHS";
      TIM_Protrusion { S7_SetPoint := 'True'} : "FB910_CNT_UHS";
      TIM_Galibo { S7_SetPoint := 'True'} : TON_TIME;
      TIM_EsperaErrorPosicion { S7_SetPoint := 'True'} : TON_TIME;
   END_VAR
   VAR_TEMP
      EstadoZonaMesa : "EstadoZona";
      EstadoZonaMaquina : "EstadoZona";
      EstadoVI : "EstadosMesa";
      EstadoMAQ : "EstadoMaquina_DesPaletizadoManual";
      DatosScada : "UDT_ScadaDatosMaquina";
      ConfigMAQ : "UDT_ConfigDesPaletizador";
      Auxiliares : Struct
         PosicionAbajo : Int;   // Posicion Abajo del Elevador
         AuxPosMax : Int;
         AuxPosMin : Int;
         Margen : Int;
         AuxAlturaMax : Int;
         AuxAlturaMin : Int;
      END_STRUCT;
      UT_Datos : Struct
         NumeroUT : UInt;
         CotaUT : Int;
         CapaUT : Int;
         SinUT : Bool;
         Con_DestinoUT : Bool;
         OK_DestinoUT : Bool;
      END_STRUCT;
      MovElevador : Struct
         NuevaPosicion : Int;
         AlturaVeloLentisima : Int;
         DestinoDOWN : Bool;   // Moviendose el elevador hacia la posicion de DOWN
         LentaDOWN : Bool;   // Activar velocidad lenta en el moviento hacia la posicion DOWN
         DestinoUP : Bool;   // Moviendose el elevador hacia la posicion de UP
         LentaUP : Bool;   // Activar velocidad lenta en el moviento hacia la posicion UP
         EnPisoAbajo : Bool;
         AlturaMax_OK : Bool;
         AlturaMin_OK : Bool;
      END_STRUCT;
      ZonaEnMarcha : Bool;
      ZonaEnReset : Bool;
      MAQ_Cargada : Bool;
      MAQ_Vacia : Bool;
      AlturaControlBarrerra : Int;
      AlturaCotaDefecto : Int;
      AlturaCapaDefecto : Int;
      AlturaCapaMinima : Int;
      AlturaCapaMaxima : Int;
      TempInt : Int;
   END_VAR
   VAR_TEMP   // added for the SCL form of the ladder/FBD networks
      _w1 : Bool;
      _w2 : Bool;
      _w3 : Bool;
   END_VAR
BEGIN

REGION Network 1: PARAMETROS ESPECIALES
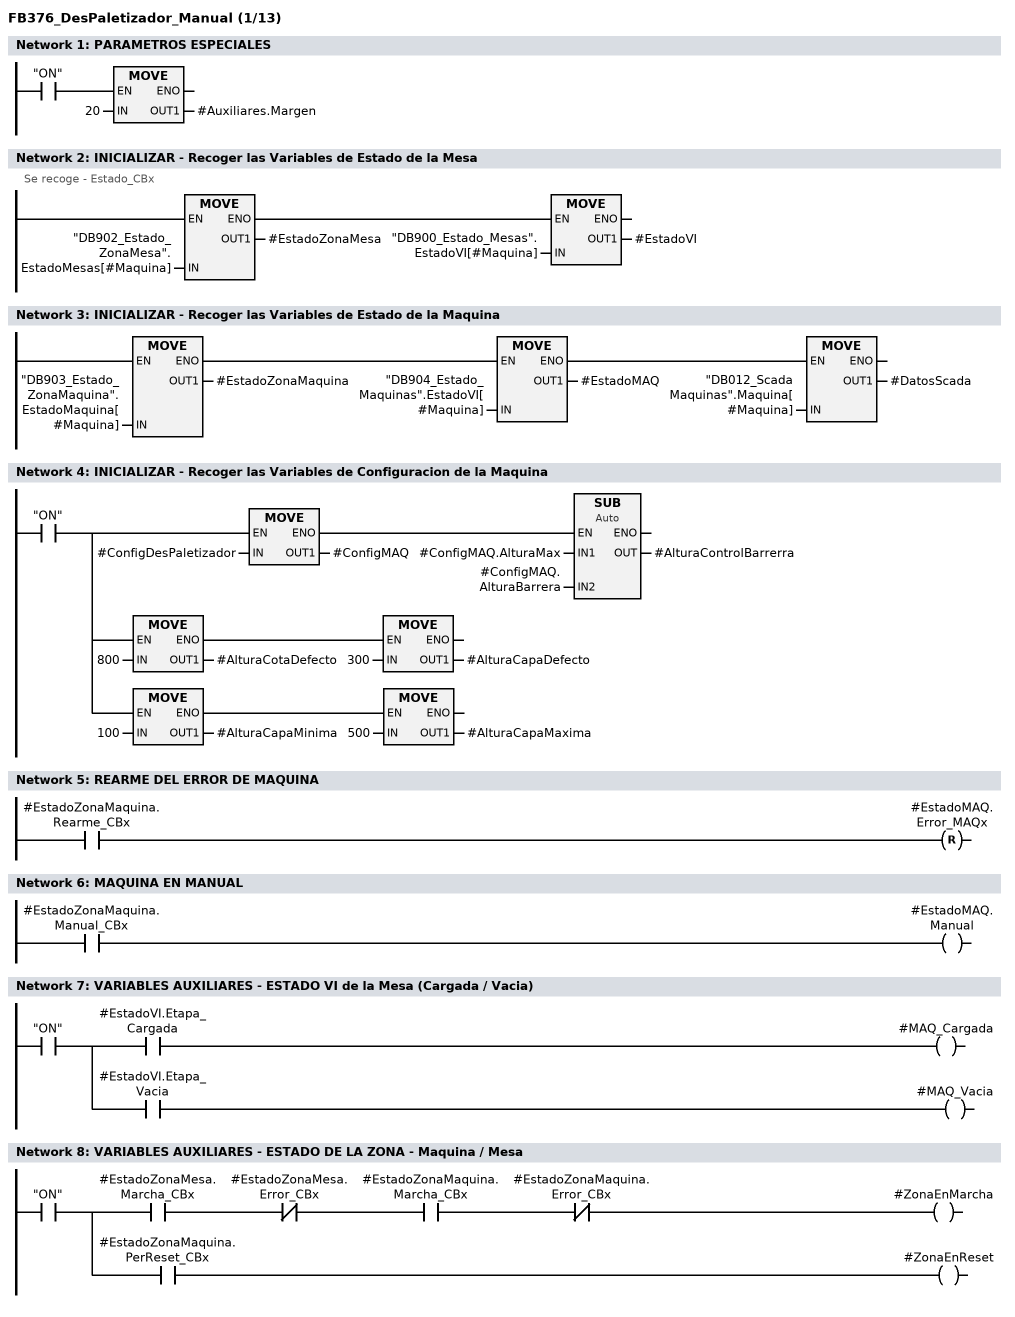
   RUNG wire#powerrail
      Contact( "ON" )
      { S7_GenerateENO := "TRUE" } Move(in := 20, out1 => #Auxiliares.Margen)
   END_RUNG
   // the same network as SCL:
   IF "ON" THEN #Auxiliares.Margen := 20; END_IF;
END_REGION

REGION Network 2: INICIALIZAR - Recoger las Variables de Estado de la Mesa
   // Se recoge - Estado_CBx
   RUNG wire#powerrail
      Move(in := "DB902_Estado_ZonaMesa".EstadoMesas[#Maquina], out1 => #EstadoZonaMesa)
      Move(in := "DB900_Estado_Mesas".EstadoVI[#Maquina], out1 => #EstadoVI)
   END_RUNG
   // the same network as SCL:
   #EstadoZonaMesa := "DB902_Estado_ZonaMesa".EstadoMesas[#Maquina];
   #EstadoVI := "DB900_Estado_Mesas".EstadoVI[#Maquina];
END_REGION

REGION Network 3: INICIALIZAR - Recoger las Variables de Estado de la Maquina
   RUNG wire#powerrail
      Move(in := "DB903_Estado_ZonaMaquina".EstadoMaquina[#Maquina], out1 => #EstadoZonaMaquina)
      Move(in := "DB904_Estado_Maquinas".EstadoVI[#Maquina], out1 => #EstadoMAQ)
      Move(in := "DB012_ScadaMaquinas".Maquina[#Maquina], out1 => #DatosScada)
   END_RUNG
   // the same network as SCL:
   #EstadoZonaMaquina := "DB903_Estado_ZonaMaquina".EstadoMaquina[#Maquina];
   #EstadoMAQ := "DB904_Estado_Maquinas".EstadoVI[#Maquina];
   #DatosScada := "DB012_ScadaMaquinas".Maquina[#Maquina];
END_REGION

REGION Network 4: INICIALIZAR - Recoger las Variables de Configuracion de la Maquina
   RUNG wire#powerrail
      Contact( "ON" )
      wire#w1
      Move(in := #ConfigDesPaletizador, out1 => #ConfigMAQ)
      Sub(in1 := #ConfigMAQ.AlturaMax, in2 := #ConfigMAQ.AlturaBarrera, out => #AlturaControlBarrerra)
   END_RUNG
   RUNG wire#w1
      Move(in := 800, out1 => #AlturaCotaDefecto)
      Move(in := 300, out1 => #AlturaCapaDefecto)
   END_RUNG
   RUNG wire#w1
      Move(in := 100, out1 => #AlturaCapaMinima)
      Move(in := 500, out1 => #AlturaCapaMaxima)
   END_RUNG
   // the same network as SCL:
   IF "ON" THEN
       #ConfigMAQ := #ConfigDesPaletizador;
       #AlturaControlBarrerra := #ConfigMAQ.AlturaMax - #ConfigMAQ.AlturaBarrera;
       #AlturaCotaDefecto := 800;
       #AlturaCapaDefecto := 300;
       #AlturaCapaMinima := 100;
       #AlturaCapaMaxima := 500;
   END_IF;
END_REGION

REGION Network 5: REARME DEL ERROR DE MAQUINA
   RUNG wire#powerrail
      Contact( #EstadoZonaMaquina.Rearme_CBx )
      R_Coil( #EstadoMAQ.Error_MAQx )
   END_RUNG
   // the same network as SCL:
   IF #EstadoZonaMaquina.Rearme_CBx THEN #EstadoMAQ.Error_MAQx := FALSE; END_IF;
END_REGION

